// TIA Portal V17 export
// export: Created 2025-03-07T09:17:31.2731089Z, ExportSetting WithDefaults, DisplayName Totally Integrated Automation Portal, DisplayVersion V17 Update 8, DisplayName TIA Portal Openness, DisplayVersion V17 Update 8, DisplayName TIA Portal Version Control Interface, DisplayVersion V17, DisplayName SINAMICS Startdrive Advanced, DisplayVersion V17 SP2, DisplayName SINAMICS Startdrive G110M, G120, G120C, G120D, G120P, G115D, DisplayVersion V17 SP2, DisplayName SINAMICS Startdrive G130, G150, S120, S150, SINAMICS MV, S210, DisplayVersion V17 SP2, DisplayName STEP 7 Professional, DisplayVersion V17 Update 8, DisplayName SINUMERIK ONE STEP 7 Toolbox, DisplayVersion V17 Update 12, DisplayName SINUMERIK 840D sl STEP 7 Toolbox, DisplayVersion V17 Update 12, DisplayName STEP 7 Safety, DisplayVersion V17 Update 6, DisplayName WinCC Advanced, DisplayVersion V17 Update 8
FUNCTION "FC373_NCK_M_CH9_SPARE" : Void   // FC373, LAD
TITLE = Channel 1 data
{ S7_Optimized_Access := 'FALSE' }
AUTHOR : ETXETAR
VERSION : 1.0
// stored: AutoNumber false, IsIECCheckEnabled false, SetENOAutomatically false, UDAEnableTagReadback false
BEGIN

REGION Network 1: ACKNOWLEDGE M700-FIXTURE 4 CLAMP SEQUENCE (READ-IN DISABLE) / ACKNOWLEDGE M100-CLAMP SEQUENCE FIXTURE 1
   // NOTE: WHEN THERE IS NOT INDEXING TABLE AVAILABLE IN THE MACHINE DELETE 
   // DB2171.DBX5.0 AND DB2171.DBX2.0
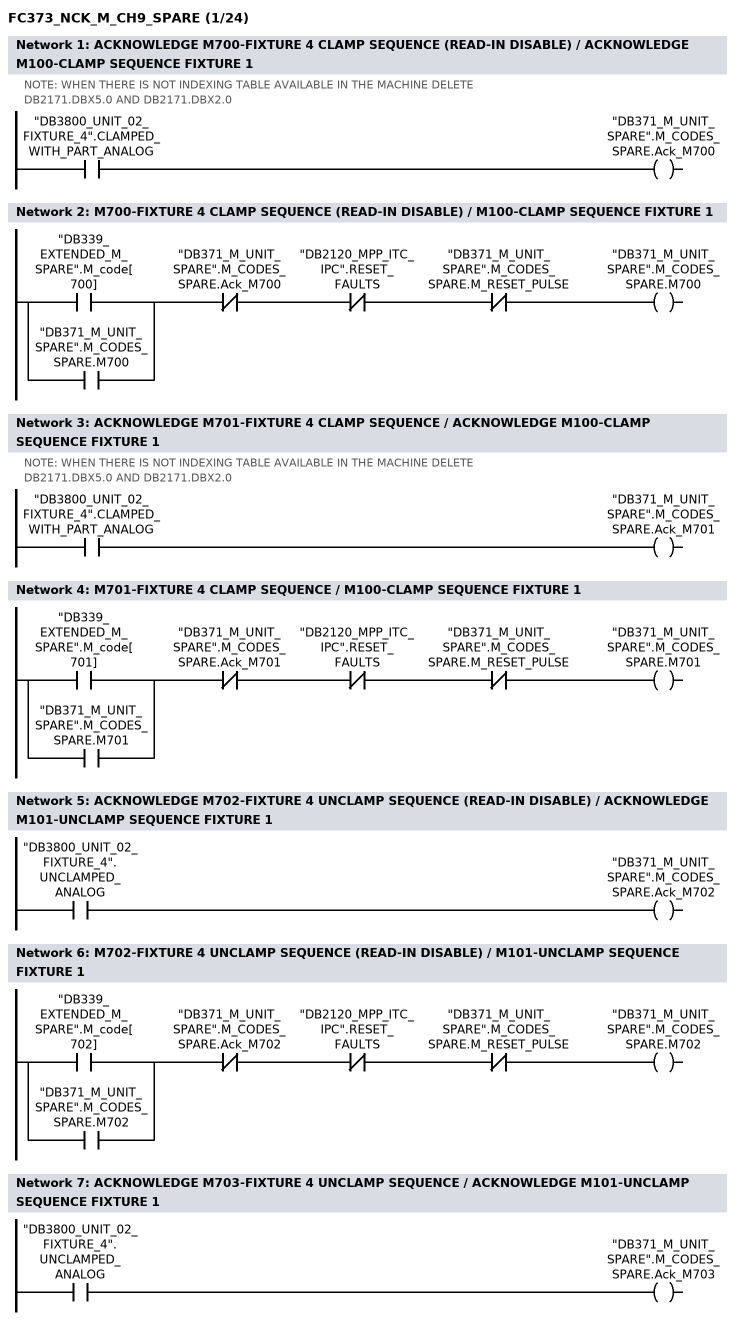
   RUNG wire#powerrail
      Contact( "DB3800_UNIT_02_FIXTURE_4".CLAMPED_WITH_PART_ANALOG )
      Coil( "DB371_M_UNIT_SPARE".M_CODES_SPARE.Ack_M700 )
   END_RUNG
   // the same network as SCL:
   "DB371_M_UNIT_SPARE".M_CODES_SPARE.Ack_M700 := "DB3800_UNIT_02_FIXTURE_4".CLAMPED_WITH_PART_ANALOG;
END_REGION

REGION Network 2: M700-FIXTURE 4 CLAMP SEQUENCE (READ-IN DISABLE) / M100-CLAMP SEQUENCE FIXTURE 1
   RUNG wire#powerrail
      Contact( "DB339_EXTENDED_M_SPARE".M_code[700] )
      wire#w1
      I_Contact( "DB371_M_UNIT_SPARE".M_CODES_SPARE.Ack_M700 )
      I_Contact( "DB2120_MPP_ITC_IPC".RESET_FAULTS )
      I_Contact( "DB371_M_UNIT_SPARE".M_CODES_SPARE.M_RESET_PULSE )
      Coil( "DB371_M_UNIT_SPARE".M_CODES_SPARE.M700 )
   END_RUNG
   RUNG wire#powerrail
      Contact( "DB371_M_UNIT_SPARE".M_CODES_SPARE.M700 )
   END_RUNG wire#w1
   // the same network as SCL:
   "DB371_M_UNIT_SPARE".M_CODES_SPARE.M700 := ("DB339_EXTENDED_M_SPARE".M_code[700] OR "DB371_M_UNIT_SPARE".M_CODES_SPARE.M700) AND NOT "DB371_M_UNIT_SPARE".M_CODES_SPARE.Ack_M700 AND NOT "DB2120_MPP_ITC_IPC".RESET_FAULTS AND NOT "DB371_M_UNIT_SPARE".M_CODES_SPARE.M_RESET_PULSE;
END_REGION

REGION Network 3: ACKNOWLEDGE M701-FIXTURE 4 CLAMP SEQUENCE / ACKNOWLEDGE M100-CLAMP SEQUENCE FIXTURE 1
   // NOTE: WHEN THERE IS NOT INDEXING TABLE AVAILABLE IN THE MACHINE DELETE 
   // DB2171.DBX5.0 AND DB2171.DBX2.0
   RUNG wire#powerrail
      Contact( "DB3800_UNIT_02_FIXTURE_4".CLAMPED_WITH_PART_ANALOG )
      Coil( "DB371_M_UNIT_SPARE".M_CODES_SPARE.Ack_M701 )
   END_RUNG
   // the same network as SCL:
   "DB371_M_UNIT_SPARE".M_CODES_SPARE.Ack_M701 := "DB3800_UNIT_02_FIXTURE_4".CLAMPED_WITH_PART_ANALOG;
END_REGION

REGION Network 4: M701-FIXTURE 4 CLAMP SEQUENCE / M100-CLAMP SEQUENCE FIXTURE 1
   RUNG wire#powerrail
      Contact( "DB339_EXTENDED_M_SPARE".M_code[701] )
      wire#w1
      I_Contact( "DB371_M_UNIT_SPARE".M_CODES_SPARE.Ack_M701 )
      I_Contact( "DB2120_MPP_ITC_IPC".RESET_FAULTS )
      I_Contact( "DB371_M_UNIT_SPARE".M_CODES_SPARE.M_RESET_PULSE )
      Coil( "DB371_M_UNIT_SPARE".M_CODES_SPARE.M701 )
   END_RUNG
   RUNG wire#powerrail
      Contact( "DB371_M_UNIT_SPARE".M_CODES_SPARE.M701 )
   END_RUNG wire#w1
   // the same network as SCL:
   "DB371_M_UNIT_SPARE".M_CODES_SPARE.M701 := ("DB339_EXTENDED_M_SPARE".M_code[701] OR "DB371_M_UNIT_SPARE".M_CODES_SPARE.M701) AND NOT "DB371_M_UNIT_SPARE".M_CODES_SPARE.Ack_M701 AND NOT "DB2120_MPP_ITC_IPC".RESET_FAULTS AND NOT "DB371_M_UNIT_SPARE".M_CODES_SPARE.M_RESET_PULSE;
END_REGION

REGION Network 5: ACKNOWLEDGE M702-FIXTURE 4 UNCLAMP SEQUENCE (READ-IN DISABLE) / ACKNOWLEDGE M101-UNCLAMP SEQUENCE FIXTURE 1
   RUNG wire#powerrail
      Contact( "DB3800_UNIT_02_FIXTURE_4".UNCLAMPED_ANALOG )
      Coil( "DB371_M_UNIT_SPARE".M_CODES_SPARE.Ack_M702 )
   END_RUNG
   // the same network as SCL:
   "DB371_M_UNIT_SPARE".M_CODES_SPARE.Ack_M702 := "DB3800_UNIT_02_FIXTURE_4".UNCLAMPED_ANALOG;
END_REGION

REGION Network 6: M702-FIXTURE 4 UNCLAMP SEQUENCE (READ-IN DISABLE) / M101-UNCLAMP SEQUENCE FIXTURE 1
   RUNG wire#powerrail
      Contact( "DB339_EXTENDED_M_SPARE".M_code[702] )
      wire#w1
      I_Contact( "DB371_M_UNIT_SPARE".M_CODES_SPARE.Ack_M702 )
      I_Contact( "DB2120_MPP_ITC_IPC".RESET_FAULTS )
      I_Contact( "DB371_M_UNIT_SPARE".M_CODES_SPARE.M_RESET_PULSE )
      Coil( "DB371_M_UNIT_SPARE".M_CODES_SPARE.M702 )
   END_RUNG
   RUNG wire#powerrail
      Contact( "DB371_M_UNIT_SPARE".M_CODES_SPARE.M702 )
   END_RUNG wire#w1
   // the same network as SCL:
   "DB371_M_UNIT_SPARE".M_CODES_SPARE.M702 := ("DB339_EXTENDED_M_SPARE".M_code[702] OR "DB371_M_UNIT_SPARE".M_CODES_SPARE.M702) AND NOT "DB371_M_UNIT_SPARE".M_CODES_SPARE.Ack_M702 AND NOT "DB2120_MPP_ITC_IPC".RESET_FAULTS AND NOT "DB371_M_UNIT_SPARE".M_CODES_SPARE.M_RESET_PULSE;
END_REGION

REGION Network 7: ACKNOWLEDGE M703-FIXTURE 4 UNCLAMP SEQUENCE / ACKNOWLEDGE M101-UNCLAMP SEQUENCE FIXTURE 1
   RUNG wire#powerrail
      Contact( "DB3800_UNIT_02_FIXTURE_4".UNCLAMPED_ANALOG )
      Coil( "DB371_M_UNIT_SPARE".M_CODES_SPARE.Ack_M703 )
   END_RUNG
   // the same network as SCL:
   "DB371_M_UNIT_SPARE".M_CODES_SPARE.Ack_M703 := "DB3800_UNIT_02_FIXTURE_4".UNCLAMPED_ANALOG;
END_REGION

REGION Network 8: M703-FIXTURE 4 UNCLAMP SEQUENCE / M101-UNCLAMP SEQUENCE FIXTURE 1
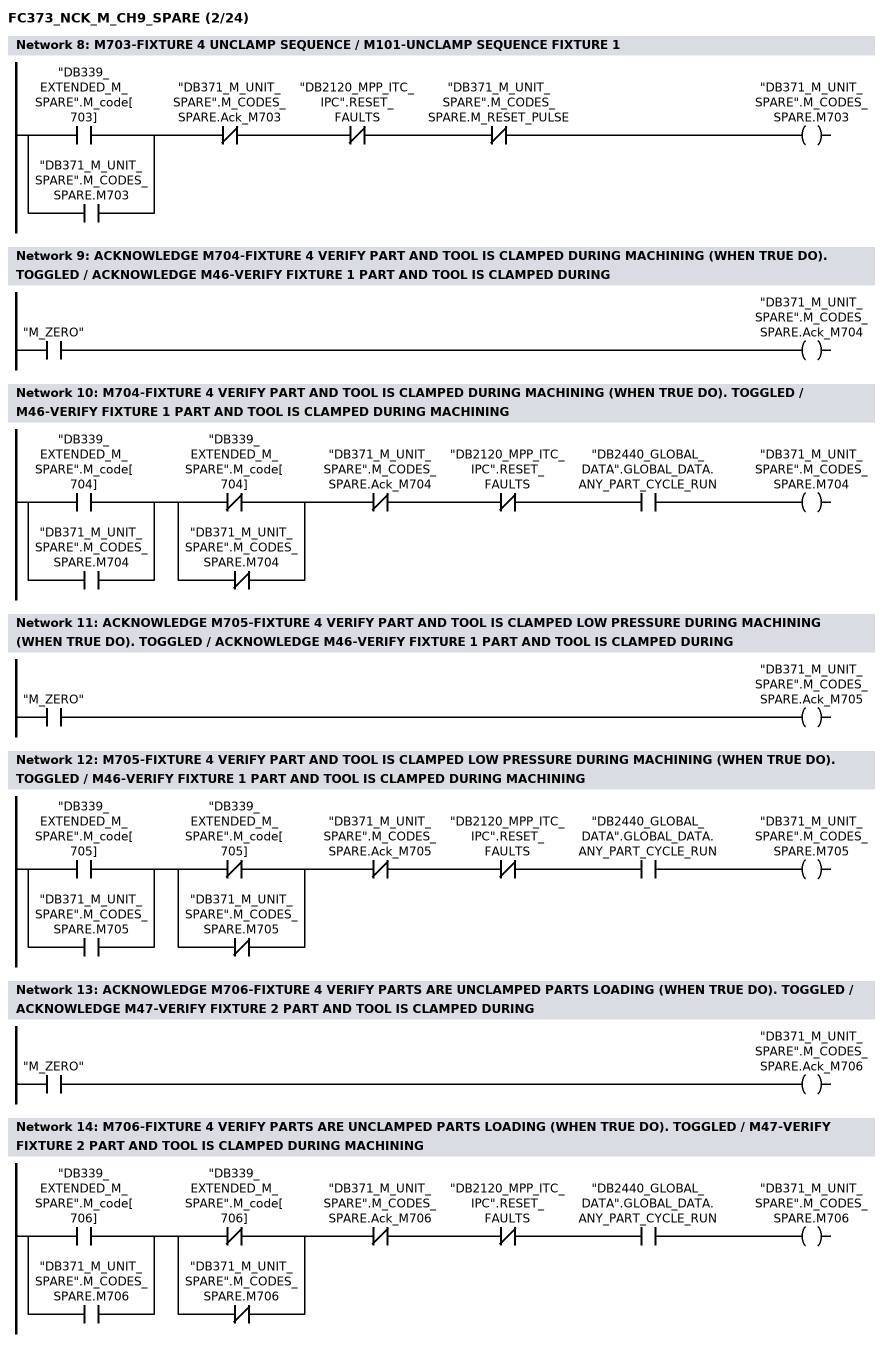
   RUNG wire#powerrail
      Contact( "DB339_EXTENDED_M_SPARE".M_code[703] )
      wire#w1
      I_Contact( "DB371_M_UNIT_SPARE".M_CODES_SPARE.Ack_M703 )
      I_Contact( "DB2120_MPP_ITC_IPC".RESET_FAULTS )
      I_Contact( "DB371_M_UNIT_SPARE".M_CODES_SPARE.M_RESET_PULSE )
      Coil( "DB371_M_UNIT_SPARE".M_CODES_SPARE.M703 )
   END_RUNG
   RUNG wire#powerrail
      Contact( "DB371_M_UNIT_SPARE".M_CODES_SPARE.M703 )
   END_RUNG wire#w1
   // the same network as SCL:
   "DB371_M_UNIT_SPARE".M_CODES_SPARE.M703 := ("DB339_EXTENDED_M_SPARE".M_code[703] OR "DB371_M_UNIT_SPARE".M_CODES_SPARE.M703) AND NOT "DB371_M_UNIT_SPARE".M_CODES_SPARE.Ack_M703 AND NOT "DB2120_MPP_ITC_IPC".RESET_FAULTS AND NOT "DB371_M_UNIT_SPARE".M_CODES_SPARE.M_RESET_PULSE;
END_REGION

REGION Network 9: ACKNOWLEDGE M704-FIXTURE 4 VERIFY PART AND TOOL IS CLAMPED DURING MACHINING (WHEN TRUE DO). TOGGLED / ACKNOWLEDGE M46-VERIFY FIXTURE 1 PART AND TOOL IS CLAMPED DURING
   RUNG wire#powerrail
      Contact( "M_ZERO" )
      Coil( "DB371_M_UNIT_SPARE".M_CODES_SPARE.Ack_M704 )
   END_RUNG
   // the same network as SCL:
   "DB371_M_UNIT_SPARE".M_CODES_SPARE.Ack_M704 := "M_ZERO";
END_REGION

REGION Network 10: M704-FIXTURE 4 VERIFY PART AND TOOL IS CLAMPED DURING MACHINING (WHEN TRUE DO). TOGGLED / M46-VERIFY FIXTURE 1 PART AND TOOL IS CLAMPED DURING MACHINING
   RUNG wire#powerrail
      Contact( "DB339_EXTENDED_M_SPARE".M_code[704] )
      wire#w1
      I_Contact( "DB339_EXTENDED_M_SPARE".M_code[704] )
      wire#w2
      I_Contact( "DB371_M_UNIT_SPARE".M_CODES_SPARE.Ack_M704 )
      I_Contact( "DB2120_MPP_ITC_IPC".RESET_FAULTS )
      Contact( "DB2440_GLOBAL_DATA".GLOBAL_DATA.ANY_PART_CYCLE_RUN )
      Coil( "DB371_M_UNIT_SPARE".M_CODES_SPARE.M704 )
   END_RUNG
   RUNG wire#powerrail
      Contact( "DB371_M_UNIT_SPARE".M_CODES_SPARE.M704 )
   END_RUNG wire#w1
   RUNG wire#w1
      I_Contact( "DB371_M_UNIT_SPARE".M_CODES_SPARE.M704 )
   END_RUNG wire#w2
   // the same network as SCL:
   "DB371_M_UNIT_SPARE".M_CODES_SPARE.M704 := ("DB339_EXTENDED_M_SPARE".M_code[704] OR "DB371_M_UNIT_SPARE".M_CODES_SPARE.M704) AND (NOT "DB339_EXTENDED_M_SPARE".M_code[704] OR NOT "DB371_M_UNIT_SPARE".M_CODES_SPARE.M704) AND NOT "DB371_M_UNIT_SPARE".M_CODES_SPARE.Ack_M704 AND NOT "DB2120_MPP_ITC_IPC".RESET_FAULTS AND "DB2440_GLOBAL_DATA".GLOBAL_DATA.ANY_PART_CYCLE_RUN;
END_REGION

REGION Network 11: ACKNOWLEDGE M705-FIXTURE 4 VERIFY PART AND TOOL IS CLAMPED LOW PRESSURE DURING MACHINING (WHEN TRUE DO). TOGGLED / ACKNOWLEDGE M46-VERIFY FIXTURE 1 PART AND TOOL IS CLAMPED DURING
   RUNG wire#powerrail
      Contact( "M_ZERO" )
      Coil( "DB371_M_UNIT_SPARE".M_CODES_SPARE.Ack_M705 )
   END_RUNG
   // the same network as SCL:
   "DB371_M_UNIT_SPARE".M_CODES_SPARE.Ack_M705 := "M_ZERO";
END_REGION

REGION Network 12: M705-FIXTURE 4 VERIFY PART AND TOOL IS CLAMPED LOW PRESSURE DURING MACHINING (WHEN TRUE DO). TOGGLED / M46-VERIFY FIXTURE 1 PART AND TOOL IS CLAMPED DURING MACHINING
   RUNG wire#powerrail
      Contact( "DB339_EXTENDED_M_SPARE".M_code[705] )
      wire#w1
      I_Contact( "DB339_EXTENDED_M_SPARE".M_code[705] )
      wire#w2
      I_Contact( "DB371_M_UNIT_SPARE".M_CODES_SPARE.Ack_M705 )
      I_Contact( "DB2120_MPP_ITC_IPC".RESET_FAULTS )
      Contact( "DB2440_GLOBAL_DATA".GLOBAL_DATA.ANY_PART_CYCLE_RUN )
      Coil( "DB371_M_UNIT_SPARE".M_CODES_SPARE.M705 )
   END_RUNG
   RUNG wire#powerrail
      Contact( "DB371_M_UNIT_SPARE".M_CODES_SPARE.M705 )
   END_RUNG wire#w1
   RUNG wire#w1
      I_Contact( "DB371_M_UNIT_SPARE".M_CODES_SPARE.M705 )
   END_RUNG wire#w2
   // the same network as SCL:
   "DB371_M_UNIT_SPARE".M_CODES_SPARE.M705 := ("DB339_EXTENDED_M_SPARE".M_code[705] OR "DB371_M_UNIT_SPARE".M_CODES_SPARE.M705) AND (NOT "DB339_EXTENDED_M_SPARE".M_code[705] OR NOT "DB371_M_UNIT_SPARE".M_CODES_SPARE.M705) AND NOT "DB371_M_UNIT_SPARE".M_CODES_SPARE.Ack_M705 AND NOT "DB2120_MPP_ITC_IPC".RESET_FAULTS AND "DB2440_GLOBAL_DATA".GLOBAL_DATA.ANY_PART_CYCLE_RUN;
END_REGION

REGION Network 13: ACKNOWLEDGE M706-FIXTURE 4 VERIFY PARTS ARE UNCLAMPED PARTS LOADING (WHEN TRUE DO). TOGGLED / ACKNOWLEDGE M47-VERIFY FIXTURE 2 PART AND TOOL IS CLAMPED DURING
   RUNG wire#powerrail
      Contact( "M_ZERO" )
      Coil( "DB371_M_UNIT_SPARE".M_CODES_SPARE.Ack_M706 )
   END_RUNG
   // the same network as SCL:
   "DB371_M_UNIT_SPARE".M_CODES_SPARE.Ack_M706 := "M_ZERO";
END_REGION

REGION Network 14: M706-FIXTURE 4 VERIFY PARTS ARE UNCLAMPED PARTS LOADING (WHEN TRUE DO). TOGGLED / M47-VERIFY FIXTURE 2 PART AND TOOL IS CLAMPED DURING MACHINING
   RUNG wire#powerrail
      Contact( "DB339_EXTENDED_M_SPARE".M_code[706] )
      wire#w1
      I_Contact( "DB339_EXTENDED_M_SPARE".M_code[706] )
      wire#w2
      I_Contact( "DB371_M_UNIT_SPARE".M_CODES_SPARE.Ack_M706 )
      I_Contact( "DB2120_MPP_ITC_IPC".RESET_FAULTS )
      Contact( "DB2440_GLOBAL_DATA".GLOBAL_DATA.ANY_PART_CYCLE_RUN )
      Coil( "DB371_M_UNIT_SPARE".M_CODES_SPARE.M706 )
   END_RUNG
   RUNG wire#powerrail
      Contact( "DB371_M_UNIT_SPARE".M_CODES_SPARE.M706 )
   END_RUNG wire#w1
   RUNG wire#w1
      I_Contact( "DB371_M_UNIT_SPARE".M_CODES_SPARE.M706 )
   END_RUNG wire#w2
   // the same network as SCL:
   "DB371_M_UNIT_SPARE".M_CODES_SPARE.M706 := ("DB339_EXTENDED_M_SPARE".M_code[706] OR "DB371_M_UNIT_SPARE".M_CODES_SPARE.M706) AND (NOT "DB339_EXTENDED_M_SPARE".M_code[706] OR NOT "DB371_M_UNIT_SPARE".M_CODES_SPARE.M706) AND NOT "DB371_M_UNIT_SPARE".M_CODES_SPARE.Ack_M706 AND NOT "DB2120_MPP_ITC_IPC".RESET_FAULTS AND "DB2440_GLOBAL_DATA".GLOBAL_DATA.ANY_PART_CYCLE_RUN;
END_REGION

REGION Network 15: ACKNOWLEDGE M707-FIXTURE 4 VERIFY FIXTURE REMAINS CLAMPED
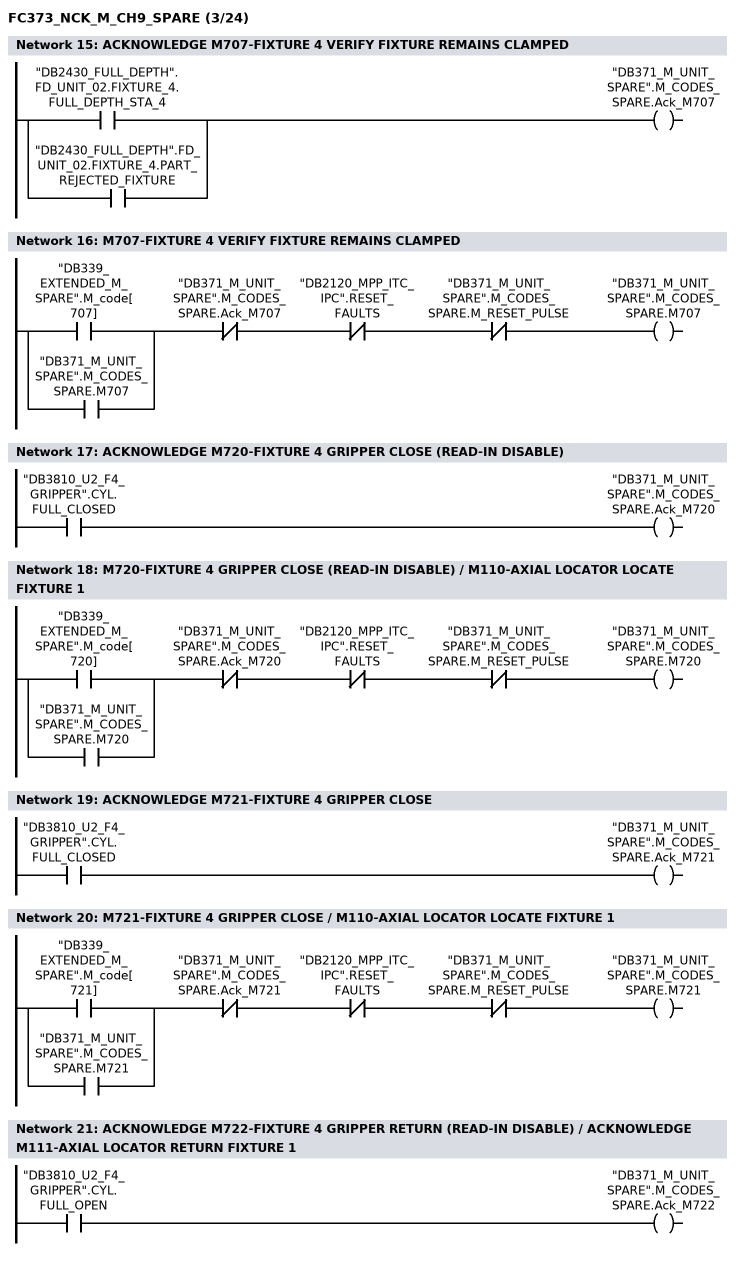
   RUNG wire#powerrail
      Contact( "DB2430_FULL_DEPTH".FD_UNIT_02.FIXTURE_4.FULL_DEPTH_STA_4 )
      wire#w1
      Coil( "DB371_M_UNIT_SPARE".M_CODES_SPARE.Ack_M707 )
   END_RUNG
   RUNG wire#powerrail
      Contact( "DB2430_FULL_DEPTH".FD_UNIT_02.FIXTURE_4.PART_REJECTED_FIXTURE )
   END_RUNG wire#w1
   // the same network as SCL:
   "DB371_M_UNIT_SPARE".M_CODES_SPARE.Ack_M707 := "DB2430_FULL_DEPTH".FD_UNIT_02.FIXTURE_4.FULL_DEPTH_STA_4 OR "DB2430_FULL_DEPTH".FD_UNIT_02.FIXTURE_4.PART_REJECTED_FIXTURE;
END_REGION

REGION Network 16: M707-FIXTURE 4 VERIFY FIXTURE REMAINS CLAMPED
   RUNG wire#powerrail
      Contact( "DB339_EXTENDED_M_SPARE".M_code[707] )
      wire#w1
      I_Contact( "DB371_M_UNIT_SPARE".M_CODES_SPARE.Ack_M707 )
      I_Contact( "DB2120_MPP_ITC_IPC".RESET_FAULTS )
      I_Contact( "DB371_M_UNIT_SPARE".M_CODES_SPARE.M_RESET_PULSE )
      Coil( "DB371_M_UNIT_SPARE".M_CODES_SPARE.M707 )
   END_RUNG
   RUNG wire#powerrail
      Contact( "DB371_M_UNIT_SPARE".M_CODES_SPARE.M707 )
   END_RUNG wire#w1
   // the same network as SCL:
   "DB371_M_UNIT_SPARE".M_CODES_SPARE.M707 := ("DB339_EXTENDED_M_SPARE".M_code[707] OR "DB371_M_UNIT_SPARE".M_CODES_SPARE.M707) AND NOT "DB371_M_UNIT_SPARE".M_CODES_SPARE.Ack_M707 AND NOT "DB2120_MPP_ITC_IPC".RESET_FAULTS AND NOT "DB371_M_UNIT_SPARE".M_CODES_SPARE.M_RESET_PULSE;
END_REGION

REGION Network 17: ACKNOWLEDGE M720-FIXTURE 4 GRIPPER CLOSE (READ-IN DISABLE)
   RUNG wire#powerrail
      Contact( "DB3810_U2_F4_GRIPPER".CYL.FULL_CLOSED )
      Coil( "DB371_M_UNIT_SPARE".M_CODES_SPARE.Ack_M720 )
   END_RUNG
   // the same network as SCL:
   "DB371_M_UNIT_SPARE".M_CODES_SPARE.Ack_M720 := "DB3810_U2_F4_GRIPPER".CYL.FULL_CLOSED;
END_REGION

REGION Network 18: M720-FIXTURE 4 GRIPPER CLOSE (READ-IN DISABLE) / M110-AXIAL LOCATOR LOCATE FIXTURE 1
   RUNG wire#powerrail
      Contact( "DB339_EXTENDED_M_SPARE".M_code[720] )
      wire#w1
      I_Contact( "DB371_M_UNIT_SPARE".M_CODES_SPARE.Ack_M720 )
      I_Contact( "DB2120_MPP_ITC_IPC".RESET_FAULTS )
      I_Contact( "DB371_M_UNIT_SPARE".M_CODES_SPARE.M_RESET_PULSE )
      Coil( "DB371_M_UNIT_SPARE".M_CODES_SPARE.M720 )
   END_RUNG
   RUNG wire#powerrail
      Contact( "DB371_M_UNIT_SPARE".M_CODES_SPARE.M720 )
   END_RUNG wire#w1
   // the same network as SCL:
   "DB371_M_UNIT_SPARE".M_CODES_SPARE.M720 := ("DB339_EXTENDED_M_SPARE".M_code[720] OR "DB371_M_UNIT_SPARE".M_CODES_SPARE.M720) AND NOT "DB371_M_UNIT_SPARE".M_CODES_SPARE.Ack_M720 AND NOT "DB2120_MPP_ITC_IPC".RESET_FAULTS AND NOT "DB371_M_UNIT_SPARE".M_CODES_SPARE.M_RESET_PULSE;
END_REGION

REGION Network 19: ACKNOWLEDGE M721-FIXTURE 4 GRIPPER CLOSE
   RUNG wire#powerrail
      Contact( "DB3810_U2_F4_GRIPPER".CYL.FULL_CLOSED )
      Coil( "DB371_M_UNIT_SPARE".M_CODES_SPARE.Ack_M721 )
   END_RUNG
   // the same network as SCL:
   "DB371_M_UNIT_SPARE".M_CODES_SPARE.Ack_M721 := "DB3810_U2_F4_GRIPPER".CYL.FULL_CLOSED;
END_REGION

REGION Network 20: M721-FIXTURE 4 GRIPPER CLOSE / M110-AXIAL LOCATOR LOCATE FIXTURE 1
   RUNG wire#powerrail
      Contact( "DB339_EXTENDED_M_SPARE".M_code[721] )
      wire#w1
      I_Contact( "DB371_M_UNIT_SPARE".M_CODES_SPARE.Ack_M721 )
      I_Contact( "DB2120_MPP_ITC_IPC".RESET_FAULTS )
      I_Contact( "DB371_M_UNIT_SPARE".M_CODES_SPARE.M_RESET_PULSE )
      Coil( "DB371_M_UNIT_SPARE".M_CODES_SPARE.M721 )
   END_RUNG
   RUNG wire#powerrail
      Contact( "DB371_M_UNIT_SPARE".M_CODES_SPARE.M721 )
   END_RUNG wire#w1
   // the same network as SCL:
   "DB371_M_UNIT_SPARE".M_CODES_SPARE.M721 := ("DB339_EXTENDED_M_SPARE".M_code[721] OR "DB371_M_UNIT_SPARE".M_CODES_SPARE.M721) AND NOT "DB371_M_UNIT_SPARE".M_CODES_SPARE.Ack_M721 AND NOT "DB2120_MPP_ITC_IPC".RESET_FAULTS AND NOT "DB371_M_UNIT_SPARE".M_CODES_SPARE.M_RESET_PULSE;
END_REGION

REGION Network 21: ACKNOWLEDGE M722-FIXTURE 4 GRIPPER RETURN (READ-IN DISABLE) / ACKNOWLEDGE M111-AXIAL LOCATOR RETURN FIXTURE 1
   RUNG wire#powerrail
      Contact( "DB3810_U2_F4_GRIPPER".CYL.FULL_OPEN )
      Coil( "DB371_M_UNIT_SPARE".M_CODES_SPARE.Ack_M722 )
   END_RUNG
   // the same network as SCL:
   "DB371_M_UNIT_SPARE".M_CODES_SPARE.Ack_M722 := "DB3810_U2_F4_GRIPPER".CYL.FULL_OPEN;
END_REGION

REGION Network 22: M722-FIXTURE 4 GRIPPER RETURN (READ-IN DISABLE) / M111-AXIAL LOCATOR RETURN FIXTURE 1
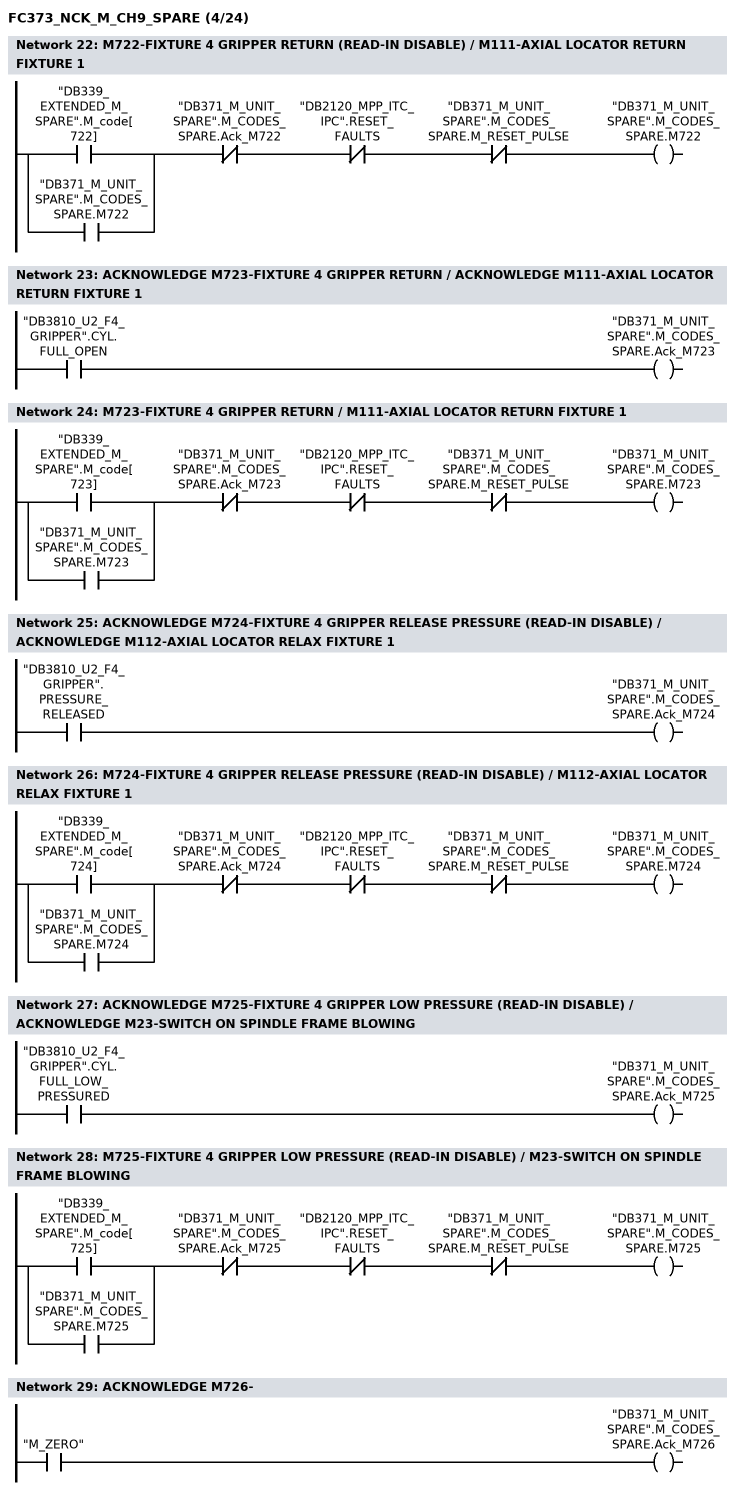
   RUNG wire#powerrail
      Contact( "DB339_EXTENDED_M_SPARE".M_code[722] )
      wire#w1
      I_Contact( "DB371_M_UNIT_SPARE".M_CODES_SPARE.Ack_M722 )
      I_Contact( "DB2120_MPP_ITC_IPC".RESET_FAULTS )
      I_Contact( "DB371_M_UNIT_SPARE".M_CODES_SPARE.M_RESET_PULSE )
      Coil( "DB371_M_UNIT_SPARE".M_CODES_SPARE.M722 )
   END_RUNG
   RUNG wire#powerrail
      Contact( "DB371_M_UNIT_SPARE".M_CODES_SPARE.M722 )
   END_RUNG wire#w1
   // the same network as SCL:
   "DB371_M_UNIT_SPARE".M_CODES_SPARE.M722 := ("DB339_EXTENDED_M_SPARE".M_code[722] OR "DB371_M_UNIT_SPARE".M_CODES_SPARE.M722) AND NOT "DB371_M_UNIT_SPARE".M_CODES_SPARE.Ack_M722 AND NOT "DB2120_MPP_ITC_IPC".RESET_FAULTS AND NOT "DB371_M_UNIT_SPARE".M_CODES_SPARE.M_RESET_PULSE;
END_REGION

REGION Network 23: ACKNOWLEDGE M723-FIXTURE 4 GRIPPER RETURN / ACKNOWLEDGE M111-AXIAL LOCATOR RETURN FIXTURE 1
   RUNG wire#powerrail
      Contact( "DB3810_U2_F4_GRIPPER".CYL.FULL_OPEN )
      Coil( "DB371_M_UNIT_SPARE".M_CODES_SPARE.Ack_M723 )
   END_RUNG
   // the same network as SCL:
   "DB371_M_UNIT_SPARE".M_CODES_SPARE.Ack_M723 := "DB3810_U2_F4_GRIPPER".CYL.FULL_OPEN;
END_REGION

REGION Network 24: M723-FIXTURE 4 GRIPPER RETURN / M111-AXIAL LOCATOR RETURN FIXTURE 1
   RUNG wire#powerrail
      Contact( "DB339_EXTENDED_M_SPARE".M_code[723] )
      wire#w1
      I_Contact( "DB371_M_UNIT_SPARE".M_CODES_SPARE.Ack_M723 )
      I_Contact( "DB2120_MPP_ITC_IPC".RESET_FAULTS )
      I_Contact( "DB371_M_UNIT_SPARE".M_CODES_SPARE.M_RESET_PULSE )
      Coil( "DB371_M_UNIT_SPARE".M_CODES_SPARE.M723 )
   END_RUNG
   RUNG wire#powerrail
      Contact( "DB371_M_UNIT_SPARE".M_CODES_SPARE.M723 )
   END_RUNG wire#w1
   // the same network as SCL:
   "DB371_M_UNIT_SPARE".M_CODES_SPARE.M723 := ("DB339_EXTENDED_M_SPARE".M_code[723] OR "DB371_M_UNIT_SPARE".M_CODES_SPARE.M723) AND NOT "DB371_M_UNIT_SPARE".M_CODES_SPARE.Ack_M723 AND NOT "DB2120_MPP_ITC_IPC".RESET_FAULTS AND NOT "DB371_M_UNIT_SPARE".M_CODES_SPARE.M_RESET_PULSE;
END_REGION

REGION Network 25: ACKNOWLEDGE M724-FIXTURE 4 GRIPPER RELEASE PRESSURE (READ-IN DISABLE) / ACKNOWLEDGE M112-AXIAL LOCATOR RELAX FIXTURE 1
   RUNG wire#powerrail
      Contact( "DB3810_U2_F4_GRIPPER".PRESSURE_RELEASED )
      Coil( "DB371_M_UNIT_SPARE".M_CODES_SPARE.Ack_M724 )
   END_RUNG
   // the same network as SCL:
   "DB371_M_UNIT_SPARE".M_CODES_SPARE.Ack_M724 := "DB3810_U2_F4_GRIPPER".PRESSURE_RELEASED;
END_REGION

REGION Network 26: M724-FIXTURE 4 GRIPPER RELEASE PRESSURE (READ-IN DISABLE) / M112-AXIAL LOCATOR RELAX FIXTURE 1
   RUNG wire#powerrail
      Contact( "DB339_EXTENDED_M_SPARE".M_code[724] )
      wire#w1
      I_Contact( "DB371_M_UNIT_SPARE".M_CODES_SPARE.Ack_M724 )
      I_Contact( "DB2120_MPP_ITC_IPC".RESET_FAULTS )
      I_Contact( "DB371_M_UNIT_SPARE".M_CODES_SPARE.M_RESET_PULSE )
      Coil( "DB371_M_UNIT_SPARE".M_CODES_SPARE.M724 )
   END_RUNG
   RUNG wire#powerrail
      Contact( "DB371_M_UNIT_SPARE".M_CODES_SPARE.M724 )
   END_RUNG wire#w1
   // the same network as SCL:
   "DB371_M_UNIT_SPARE".M_CODES_SPARE.M724 := ("DB339_EXTENDED_M_SPARE".M_code[724] OR "DB371_M_UNIT_SPARE".M_CODES_SPARE.M724) AND NOT "DB371_M_UNIT_SPARE".M_CODES_SPARE.Ack_M724 AND NOT "DB2120_MPP_ITC_IPC".RESET_FAULTS AND NOT "DB371_M_UNIT_SPARE".M_CODES_SPARE.M_RESET_PULSE;
END_REGION

REGION Network 27: ACKNOWLEDGE M725-FIXTURE 4 GRIPPER LOW PRESSURE (READ-IN DISABLE) / ACKNOWLEDGE M23-SWITCH ON SPINDLE FRAME BLOWING
   RUNG wire#powerrail
      Contact( "DB3810_U2_F4_GRIPPER".CYL.FULL_LOW_PRESSURED )
      Coil( "DB371_M_UNIT_SPARE".M_CODES_SPARE.Ack_M725 )
   END_RUNG
   // the same network as SCL:
   "DB371_M_UNIT_SPARE".M_CODES_SPARE.Ack_M725 := "DB3810_U2_F4_GRIPPER".CYL.FULL_LOW_PRESSURED;
END_REGION

REGION Network 28: M725-FIXTURE 4 GRIPPER LOW PRESSURE (READ-IN DISABLE) / M23-SWITCH ON SPINDLE FRAME BLOWING
   RUNG wire#powerrail
      Contact( "DB339_EXTENDED_M_SPARE".M_code[725] )
      wire#w1
      I_Contact( "DB371_M_UNIT_SPARE".M_CODES_SPARE.Ack_M725 )
      I_Contact( "DB2120_MPP_ITC_IPC".RESET_FAULTS )
      I_Contact( "DB371_M_UNIT_SPARE".M_CODES_SPARE.M_RESET_PULSE )
      Coil( "DB371_M_UNIT_SPARE".M_CODES_SPARE.M725 )
   END_RUNG
   RUNG wire#powerrail
      Contact( "DB371_M_UNIT_SPARE".M_CODES_SPARE.M725 )
   END_RUNG wire#w1
   // the same network as SCL:
   "DB371_M_UNIT_SPARE".M_CODES_SPARE.M725 := ("DB339_EXTENDED_M_SPARE".M_code[725] OR "DB371_M_UNIT_SPARE".M_CODES_SPARE.M725) AND NOT "DB371_M_UNIT_SPARE".M_CODES_SPARE.Ack_M725 AND NOT "DB2120_MPP_ITC_IPC".RESET_FAULTS AND NOT "DB371_M_UNIT_SPARE".M_CODES_SPARE.M_RESET_PULSE;
END_REGION

REGION Network 29: ACKNOWLEDGE M726-
   RUNG wire#powerrail
      Contact( "M_ZERO" )
      Coil( "DB371_M_UNIT_SPARE".M_CODES_SPARE.Ack_M726 )
   END_RUNG
   // the same network as SCL:
   "DB371_M_UNIT_SPARE".M_CODES_SPARE.Ack_M726 := "M_ZERO";
END_REGION

REGION Network 30: M726-
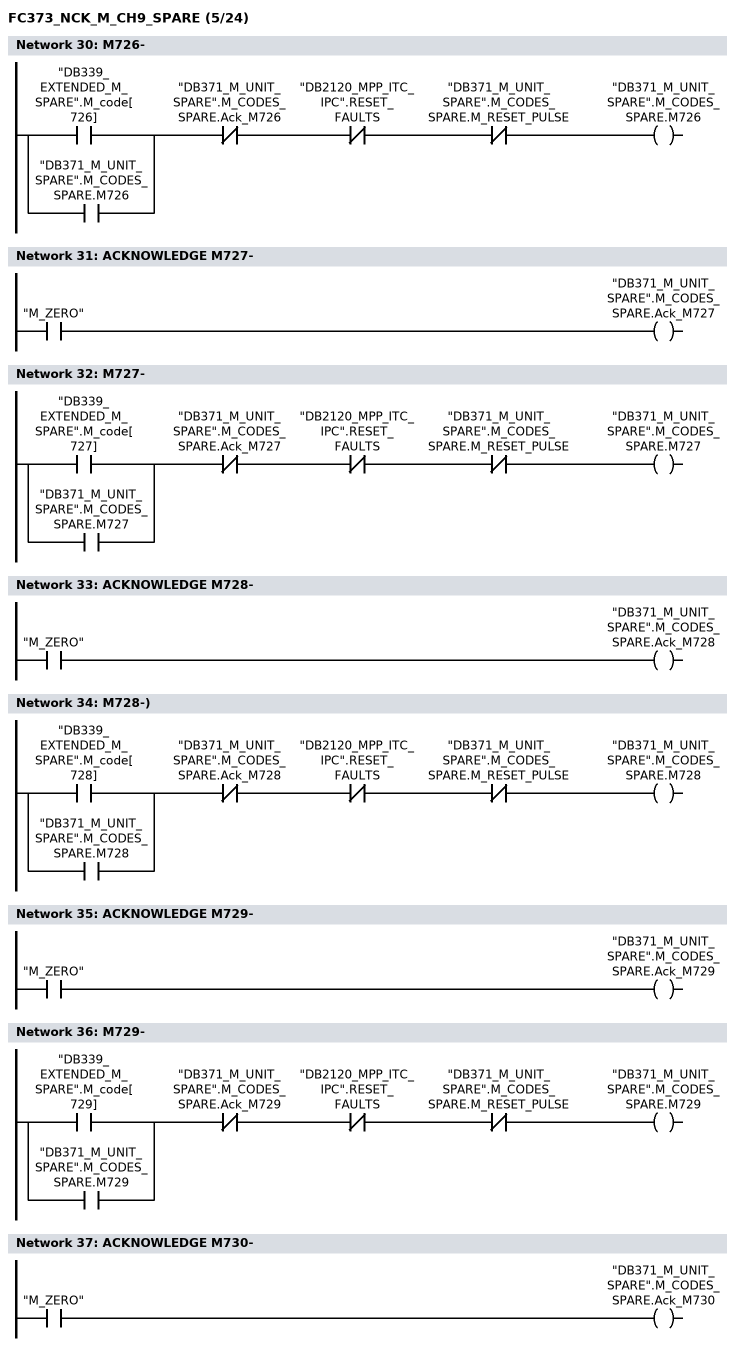
   RUNG wire#powerrail
      Contact( "DB339_EXTENDED_M_SPARE".M_code[726] )
      wire#w1
      I_Contact( "DB371_M_UNIT_SPARE".M_CODES_SPARE.Ack_M726 )
      I_Contact( "DB2120_MPP_ITC_IPC".RESET_FAULTS )
      I_Contact( "DB371_M_UNIT_SPARE".M_CODES_SPARE.M_RESET_PULSE )
      Coil( "DB371_M_UNIT_SPARE".M_CODES_SPARE.M726 )
   END_RUNG
   RUNG wire#powerrail
      Contact( "DB371_M_UNIT_SPARE".M_CODES_SPARE.M726 )
   END_RUNG wire#w1
   // the same network as SCL:
   "DB371_M_UNIT_SPARE".M_CODES_SPARE.M726 := ("DB339_EXTENDED_M_SPARE".M_code[726] OR "DB371_M_UNIT_SPARE".M_CODES_SPARE.M726) AND NOT "DB371_M_UNIT_SPARE".M_CODES_SPARE.Ack_M726 AND NOT "DB2120_MPP_ITC_IPC".RESET_FAULTS AND NOT "DB371_M_UNIT_SPARE".M_CODES_SPARE.M_RESET_PULSE;
END_REGION

REGION Network 31: ACKNOWLEDGE M727-
   RUNG wire#powerrail
      Contact( "M_ZERO" )
      Coil( "DB371_M_UNIT_SPARE".M_CODES_SPARE.Ack_M727 )
   END_RUNG
   // the same network as SCL:
   "DB371_M_UNIT_SPARE".M_CODES_SPARE.Ack_M727 := "M_ZERO";
END_REGION

REGION Network 32: M727-
   RUNG wire#powerrail
      Contact( "DB339_EXTENDED_M_SPARE".M_code[727] )
      wire#w1
      I_Contact( "DB371_M_UNIT_SPARE".M_CODES_SPARE.Ack_M727 )
      I_Contact( "DB2120_MPP_ITC_IPC".RESET_FAULTS )
      I_Contact( "DB371_M_UNIT_SPARE".M_CODES_SPARE.M_RESET_PULSE )
      Coil( "DB371_M_UNIT_SPARE".M_CODES_SPARE.M727 )
   END_RUNG
   RUNG wire#powerrail
      Contact( "DB371_M_UNIT_SPARE".M_CODES_SPARE.M727 )
   END_RUNG wire#w1
   // the same network as SCL:
   "DB371_M_UNIT_SPARE".M_CODES_SPARE.M727 := ("DB339_EXTENDED_M_SPARE".M_code[727] OR "DB371_M_UNIT_SPARE".M_CODES_SPARE.M727) AND NOT "DB371_M_UNIT_SPARE".M_CODES_SPARE.Ack_M727 AND NOT "DB2120_MPP_ITC_IPC".RESET_FAULTS AND NOT "DB371_M_UNIT_SPARE".M_CODES_SPARE.M_RESET_PULSE;
END_REGION

REGION Network 33: ACKNOWLEDGE M728-
   RUNG wire#powerrail
      Contact( "M_ZERO" )
      Coil( "DB371_M_UNIT_SPARE".M_CODES_SPARE.Ack_M728 )
   END_RUNG
   // the same network as SCL:
   "DB371_M_UNIT_SPARE".M_CODES_SPARE.Ack_M728 := "M_ZERO";
END_REGION

REGION Network 34: M728-)
   RUNG wire#powerrail
      Contact( "DB339_EXTENDED_M_SPARE".M_code[728] )
      wire#w1
      I_Contact( "DB371_M_UNIT_SPARE".M_CODES_SPARE.Ack_M728 )
      I_Contact( "DB2120_MPP_ITC_IPC".RESET_FAULTS )
      I_Contact( "DB371_M_UNIT_SPARE".M_CODES_SPARE.M_RESET_PULSE )
      Coil( "DB371_M_UNIT_SPARE".M_CODES_SPARE.M728 )
   END_RUNG
   RUNG wire#powerrail
      Contact( "DB371_M_UNIT_SPARE".M_CODES_SPARE.M728 )
   END_RUNG wire#w1
   // the same network as SCL:
   "DB371_M_UNIT_SPARE".M_CODES_SPARE.M728 := ("DB339_EXTENDED_M_SPARE".M_code[728] OR "DB371_M_UNIT_SPARE".M_CODES_SPARE.M728) AND NOT "DB371_M_UNIT_SPARE".M_CODES_SPARE.Ack_M728 AND NOT "DB2120_MPP_ITC_IPC".RESET_FAULTS AND NOT "DB371_M_UNIT_SPARE".M_CODES_SPARE.M_RESET_PULSE;
END_REGION

REGION Network 35: ACKNOWLEDGE M729-
   RUNG wire#powerrail
      Contact( "M_ZERO" )
      Coil( "DB371_M_UNIT_SPARE".M_CODES_SPARE.Ack_M729 )
   END_RUNG
   // the same network as SCL:
   "DB371_M_UNIT_SPARE".M_CODES_SPARE.Ack_M729 := "M_ZERO";
END_REGION

REGION Network 36: M729-
   RUNG wire#powerrail
      Contact( "DB339_EXTENDED_M_SPARE".M_code[729] )
      wire#w1
      I_Contact( "DB371_M_UNIT_SPARE".M_CODES_SPARE.Ack_M729 )
      I_Contact( "DB2120_MPP_ITC_IPC".RESET_FAULTS )
      I_Contact( "DB371_M_UNIT_SPARE".M_CODES_SPARE.M_RESET_PULSE )
      Coil( "DB371_M_UNIT_SPARE".M_CODES_SPARE.M729 )
   END_RUNG
   RUNG wire#powerrail
      Contact( "DB371_M_UNIT_SPARE".M_CODES_SPARE.M729 )
   END_RUNG wire#w1
   // the same network as SCL:
   "DB371_M_UNIT_SPARE".M_CODES_SPARE.M729 := ("DB339_EXTENDED_M_SPARE".M_code[729] OR "DB371_M_UNIT_SPARE".M_CODES_SPARE.M729) AND NOT "DB371_M_UNIT_SPARE".M_CODES_SPARE.Ack_M729 AND NOT "DB2120_MPP_ITC_IPC".RESET_FAULTS AND NOT "DB371_M_UNIT_SPARE".M_CODES_SPARE.M_RESET_PULSE;
END_REGION

REGION Network 37: ACKNOWLEDGE M730-
   RUNG wire#powerrail
      Contact( "M_ZERO" )
      Coil( "DB371_M_UNIT_SPARE".M_CODES_SPARE.Ack_M730 )
   END_RUNG
   // the same network as SCL:
   "DB371_M_UNIT_SPARE".M_CODES_SPARE.Ack_M730 := "M_ZERO";
END_REGION

REGION Network 38: M730-
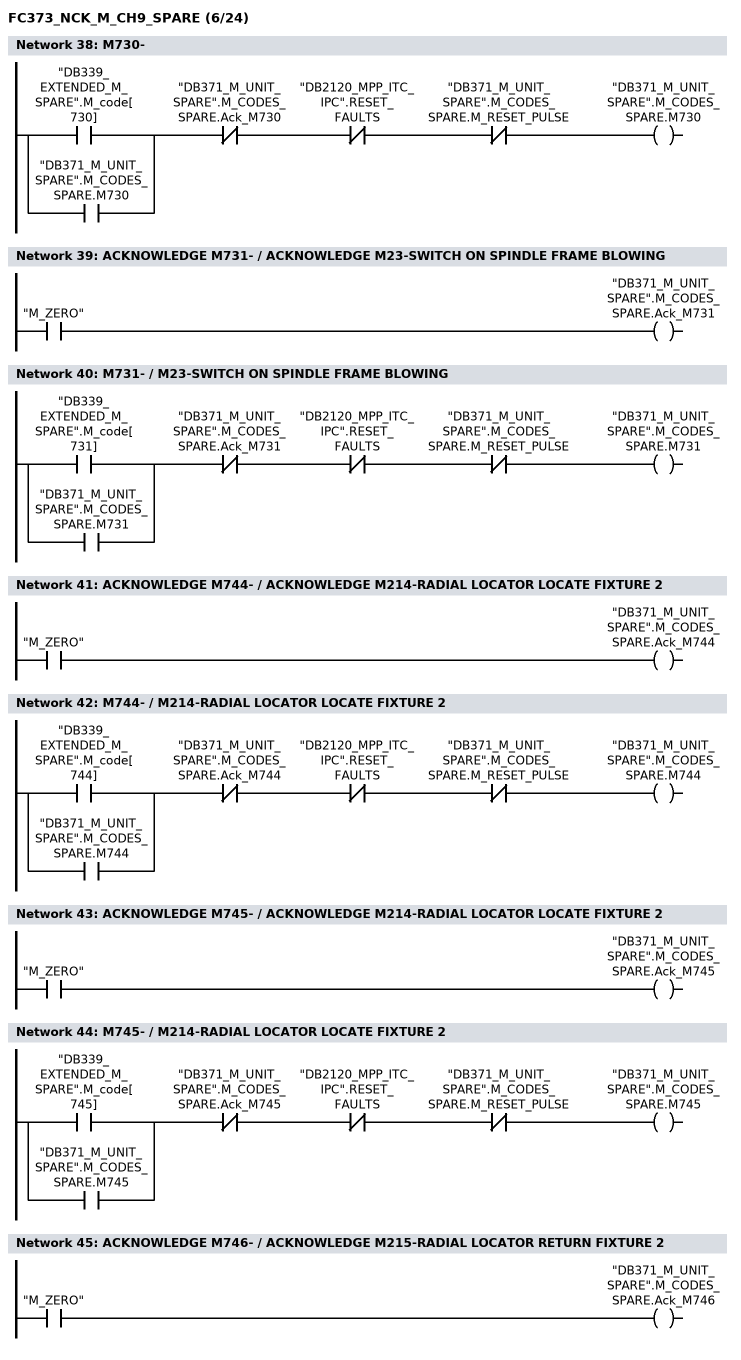
   RUNG wire#powerrail
      Contact( "DB339_EXTENDED_M_SPARE".M_code[730] )
      wire#w1
      I_Contact( "DB371_M_UNIT_SPARE".M_CODES_SPARE.Ack_M730 )
      I_Contact( "DB2120_MPP_ITC_IPC".RESET_FAULTS )
      I_Contact( "DB371_M_UNIT_SPARE".M_CODES_SPARE.M_RESET_PULSE )
      Coil( "DB371_M_UNIT_SPARE".M_CODES_SPARE.M730 )
   END_RUNG
   RUNG wire#powerrail
      Contact( "DB371_M_UNIT_SPARE".M_CODES_SPARE.M730 )
   END_RUNG wire#w1
   // the same network as SCL:
   "DB371_M_UNIT_SPARE".M_CODES_SPARE.M730 := ("DB339_EXTENDED_M_SPARE".M_code[730] OR "DB371_M_UNIT_SPARE".M_CODES_SPARE.M730) AND NOT "DB371_M_UNIT_SPARE".M_CODES_SPARE.Ack_M730 AND NOT "DB2120_MPP_ITC_IPC".RESET_FAULTS AND NOT "DB371_M_UNIT_SPARE".M_CODES_SPARE.M_RESET_PULSE;
END_REGION

REGION Network 39: ACKNOWLEDGE M731- / ACKNOWLEDGE M23-SWITCH ON SPINDLE FRAME BLOWING
   RUNG wire#powerrail
      Contact( "M_ZERO" )
      Coil( "DB371_M_UNIT_SPARE".M_CODES_SPARE.Ack_M731 )
   END_RUNG
   // the same network as SCL:
   "DB371_M_UNIT_SPARE".M_CODES_SPARE.Ack_M731 := "M_ZERO";
END_REGION

REGION Network 40: M731- / M23-SWITCH ON SPINDLE FRAME BLOWING
   RUNG wire#powerrail
      Contact( "DB339_EXTENDED_M_SPARE".M_code[731] )
      wire#w1
      I_Contact( "DB371_M_UNIT_SPARE".M_CODES_SPARE.Ack_M731 )
      I_Contact( "DB2120_MPP_ITC_IPC".RESET_FAULTS )
      I_Contact( "DB371_M_UNIT_SPARE".M_CODES_SPARE.M_RESET_PULSE )
      Coil( "DB371_M_UNIT_SPARE".M_CODES_SPARE.M731 )
   END_RUNG
   RUNG wire#powerrail
      Contact( "DB371_M_UNIT_SPARE".M_CODES_SPARE.M731 )
   END_RUNG wire#w1
   // the same network as SCL:
   "DB371_M_UNIT_SPARE".M_CODES_SPARE.M731 := ("DB339_EXTENDED_M_SPARE".M_code[731] OR "DB371_M_UNIT_SPARE".M_CODES_SPARE.M731) AND NOT "DB371_M_UNIT_SPARE".M_CODES_SPARE.Ack_M731 AND NOT "DB2120_MPP_ITC_IPC".RESET_FAULTS AND NOT "DB371_M_UNIT_SPARE".M_CODES_SPARE.M_RESET_PULSE;
END_REGION

REGION Network 41: ACKNOWLEDGE M744- / ACKNOWLEDGE M214-RADIAL LOCATOR LOCATE FIXTURE 2
   RUNG wire#powerrail
      Contact( "M_ZERO" )
      Coil( "DB371_M_UNIT_SPARE".M_CODES_SPARE.Ack_M744 )
   END_RUNG
   // the same network as SCL:
   "DB371_M_UNIT_SPARE".M_CODES_SPARE.Ack_M744 := "M_ZERO";
END_REGION

REGION Network 42: M744- / M214-RADIAL LOCATOR LOCATE FIXTURE 2
   RUNG wire#powerrail
      Contact( "DB339_EXTENDED_M_SPARE".M_code[744] )
      wire#w1
      I_Contact( "DB371_M_UNIT_SPARE".M_CODES_SPARE.Ack_M744 )
      I_Contact( "DB2120_MPP_ITC_IPC".RESET_FAULTS )
      I_Contact( "DB371_M_UNIT_SPARE".M_CODES_SPARE.M_RESET_PULSE )
      Coil( "DB371_M_UNIT_SPARE".M_CODES_SPARE.M744 )
   END_RUNG
   RUNG wire#powerrail
      Contact( "DB371_M_UNIT_SPARE".M_CODES_SPARE.M744 )
   END_RUNG wire#w1
   // the same network as SCL:
   "DB371_M_UNIT_SPARE".M_CODES_SPARE.M744 := ("DB339_EXTENDED_M_SPARE".M_code[744] OR "DB371_M_UNIT_SPARE".M_CODES_SPARE.M744) AND NOT "DB371_M_UNIT_SPARE".M_CODES_SPARE.Ack_M744 AND NOT "DB2120_MPP_ITC_IPC".RESET_FAULTS AND NOT "DB371_M_UNIT_SPARE".M_CODES_SPARE.M_RESET_PULSE;
END_REGION

REGION Network 43: ACKNOWLEDGE M745- / ACKNOWLEDGE M214-RADIAL LOCATOR LOCATE FIXTURE 2
   RUNG wire#powerrail
      Contact( "M_ZERO" )
      Coil( "DB371_M_UNIT_SPARE".M_CODES_SPARE.Ack_M745 )
   END_RUNG
   // the same network as SCL:
   "DB371_M_UNIT_SPARE".M_CODES_SPARE.Ack_M745 := "M_ZERO";
END_REGION

REGION Network 44: M745- / M214-RADIAL LOCATOR LOCATE FIXTURE 2
   RUNG wire#powerrail
      Contact( "DB339_EXTENDED_M_SPARE".M_code[745] )
      wire#w1
      I_Contact( "DB371_M_UNIT_SPARE".M_CODES_SPARE.Ack_M745 )
      I_Contact( "DB2120_MPP_ITC_IPC".RESET_FAULTS )
      I_Contact( "DB371_M_UNIT_SPARE".M_CODES_SPARE.M_RESET_PULSE )
      Coil( "DB371_M_UNIT_SPARE".M_CODES_SPARE.M745 )
   END_RUNG
   RUNG wire#powerrail
      Contact( "DB371_M_UNIT_SPARE".M_CODES_SPARE.M745 )
   END_RUNG wire#w1
   // the same network as SCL:
   "DB371_M_UNIT_SPARE".M_CODES_SPARE.M745 := ("DB339_EXTENDED_M_SPARE".M_code[745] OR "DB371_M_UNIT_SPARE".M_CODES_SPARE.M745) AND NOT "DB371_M_UNIT_SPARE".M_CODES_SPARE.Ack_M745 AND NOT "DB2120_MPP_ITC_IPC".RESET_FAULTS AND NOT "DB371_M_UNIT_SPARE".M_CODES_SPARE.M_RESET_PULSE;
END_REGION

REGION Network 45: ACKNOWLEDGE M746- / ACKNOWLEDGE M215-RADIAL LOCATOR RETURN FIXTURE 2
   RUNG wire#powerrail
      Contact( "M_ZERO" )
      Coil( "DB371_M_UNIT_SPARE".M_CODES_SPARE.Ack_M746 )
   END_RUNG
   // the same network as SCL:
   "DB371_M_UNIT_SPARE".M_CODES_SPARE.Ack_M746 := "M_ZERO";
END_REGION

REGION Network 46: M746- / M215-RADIAL LOCATOR RETURN FIXTURE 2
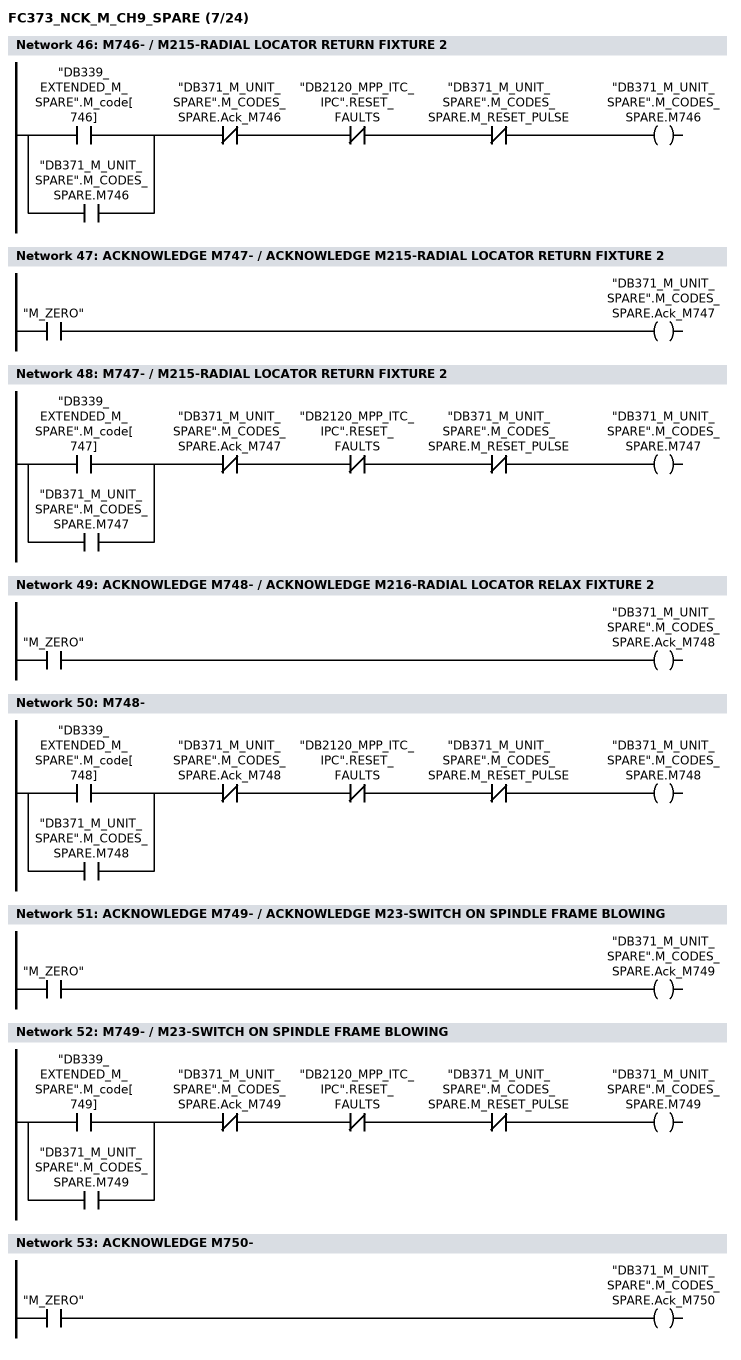
   RUNG wire#powerrail
      Contact( "DB339_EXTENDED_M_SPARE".M_code[746] )
      wire#w1
      I_Contact( "DB371_M_UNIT_SPARE".M_CODES_SPARE.Ack_M746 )
      I_Contact( "DB2120_MPP_ITC_IPC".RESET_FAULTS )
      I_Contact( "DB371_M_UNIT_SPARE".M_CODES_SPARE.M_RESET_PULSE )
      Coil( "DB371_M_UNIT_SPARE".M_CODES_SPARE.M746 )
   END_RUNG
   RUNG wire#powerrail
      Contact( "DB371_M_UNIT_SPARE".M_CODES_SPARE.M746 )
   END_RUNG wire#w1
   // the same network as SCL:
   "DB371_M_UNIT_SPARE".M_CODES_SPARE.M746 := ("DB339_EXTENDED_M_SPARE".M_code[746] OR "DB371_M_UNIT_SPARE".M_CODES_SPARE.M746) AND NOT "DB371_M_UNIT_SPARE".M_CODES_SPARE.Ack_M746 AND NOT "DB2120_MPP_ITC_IPC".RESET_FAULTS AND NOT "DB371_M_UNIT_SPARE".M_CODES_SPARE.M_RESET_PULSE;
END_REGION

REGION Network 47: ACKNOWLEDGE M747- / ACKNOWLEDGE M215-RADIAL LOCATOR RETURN FIXTURE 2
   RUNG wire#powerrail
      Contact( "M_ZERO" )
      Coil( "DB371_M_UNIT_SPARE".M_CODES_SPARE.Ack_M747 )
   END_RUNG
   // the same network as SCL:
   "DB371_M_UNIT_SPARE".M_CODES_SPARE.Ack_M747 := "M_ZERO";
END_REGION

REGION Network 48: M747- / M215-RADIAL LOCATOR RETURN FIXTURE 2
   RUNG wire#powerrail
      Contact( "DB339_EXTENDED_M_SPARE".M_code[747] )
      wire#w1
      I_Contact( "DB371_M_UNIT_SPARE".M_CODES_SPARE.Ack_M747 )
      I_Contact( "DB2120_MPP_ITC_IPC".RESET_FAULTS )
      I_Contact( "DB371_M_UNIT_SPARE".M_CODES_SPARE.M_RESET_PULSE )
      Coil( "DB371_M_UNIT_SPARE".M_CODES_SPARE.M747 )
   END_RUNG
   RUNG wire#powerrail
      Contact( "DB371_M_UNIT_SPARE".M_CODES_SPARE.M747 )
   END_RUNG wire#w1
   // the same network as SCL:
   "DB371_M_UNIT_SPARE".M_CODES_SPARE.M747 := ("DB339_EXTENDED_M_SPARE".M_code[747] OR "DB371_M_UNIT_SPARE".M_CODES_SPARE.M747) AND NOT "DB371_M_UNIT_SPARE".M_CODES_SPARE.Ack_M747 AND NOT "DB2120_MPP_ITC_IPC".RESET_FAULTS AND NOT "DB371_M_UNIT_SPARE".M_CODES_SPARE.M_RESET_PULSE;
END_REGION

REGION Network 49: ACKNOWLEDGE M748- / ACKNOWLEDGE M216-RADIAL LOCATOR RELAX FIXTURE 2
   RUNG wire#powerrail
      Contact( "M_ZERO" )
      Coil( "DB371_M_UNIT_SPARE".M_CODES_SPARE.Ack_M748 )
   END_RUNG
   // the same network as SCL:
   "DB371_M_UNIT_SPARE".M_CODES_SPARE.Ack_M748 := "M_ZERO";
END_REGION

REGION Network 50: M748-
   RUNG wire#powerrail
      Contact( "DB339_EXTENDED_M_SPARE".M_code[748] )
      wire#w1
      I_Contact( "DB371_M_UNIT_SPARE".M_CODES_SPARE.Ack_M748 )
      I_Contact( "DB2120_MPP_ITC_IPC".RESET_FAULTS )
      I_Contact( "DB371_M_UNIT_SPARE".M_CODES_SPARE.M_RESET_PULSE )
      Coil( "DB371_M_UNIT_SPARE".M_CODES_SPARE.M748 )
   END_RUNG
   RUNG wire#powerrail
      Contact( "DB371_M_UNIT_SPARE".M_CODES_SPARE.M748 )
   END_RUNG wire#w1
   // the same network as SCL:
   "DB371_M_UNIT_SPARE".M_CODES_SPARE.M748 := ("DB339_EXTENDED_M_SPARE".M_code[748] OR "DB371_M_UNIT_SPARE".M_CODES_SPARE.M748) AND NOT "DB371_M_UNIT_SPARE".M_CODES_SPARE.Ack_M748 AND NOT "DB2120_MPP_ITC_IPC".RESET_FAULTS AND NOT "DB371_M_UNIT_SPARE".M_CODES_SPARE.M_RESET_PULSE;
END_REGION

REGION Network 51: ACKNOWLEDGE M749- / ACKNOWLEDGE M23-SWITCH ON SPINDLE FRAME BLOWING
   RUNG wire#powerrail
      Contact( "M_ZERO" )
      Coil( "DB371_M_UNIT_SPARE".M_CODES_SPARE.Ack_M749 )
   END_RUNG
   // the same network as SCL:
   "DB371_M_UNIT_SPARE".M_CODES_SPARE.Ack_M749 := "M_ZERO";
END_REGION

REGION Network 52: M749- / M23-SWITCH ON SPINDLE FRAME BLOWING
   RUNG wire#powerrail
      Contact( "DB339_EXTENDED_M_SPARE".M_code[749] )
      wire#w1
      I_Contact( "DB371_M_UNIT_SPARE".M_CODES_SPARE.Ack_M749 )
      I_Contact( "DB2120_MPP_ITC_IPC".RESET_FAULTS )
      I_Contact( "DB371_M_UNIT_SPARE".M_CODES_SPARE.M_RESET_PULSE )
      Coil( "DB371_M_UNIT_SPARE".M_CODES_SPARE.M749 )
   END_RUNG
   RUNG wire#powerrail
      Contact( "DB371_M_UNIT_SPARE".M_CODES_SPARE.M749 )
   END_RUNG wire#w1
   // the same network as SCL:
   "DB371_M_UNIT_SPARE".M_CODES_SPARE.M749 := ("DB339_EXTENDED_M_SPARE".M_code[749] OR "DB371_M_UNIT_SPARE".M_CODES_SPARE.M749) AND NOT "DB371_M_UNIT_SPARE".M_CODES_SPARE.Ack_M749 AND NOT "DB2120_MPP_ITC_IPC".RESET_FAULTS AND NOT "DB371_M_UNIT_SPARE".M_CODES_SPARE.M_RESET_PULSE;
END_REGION

REGION Network 53: ACKNOWLEDGE M750-
   RUNG wire#powerrail
      Contact( "M_ZERO" )
      Coil( "DB371_M_UNIT_SPARE".M_CODES_SPARE.Ack_M750 )
   END_RUNG
   // the same network as SCL:
   "DB371_M_UNIT_SPARE".M_CODES_SPARE.Ack_M750 := "M_ZERO";
END_REGION

REGION Network 54: M750-
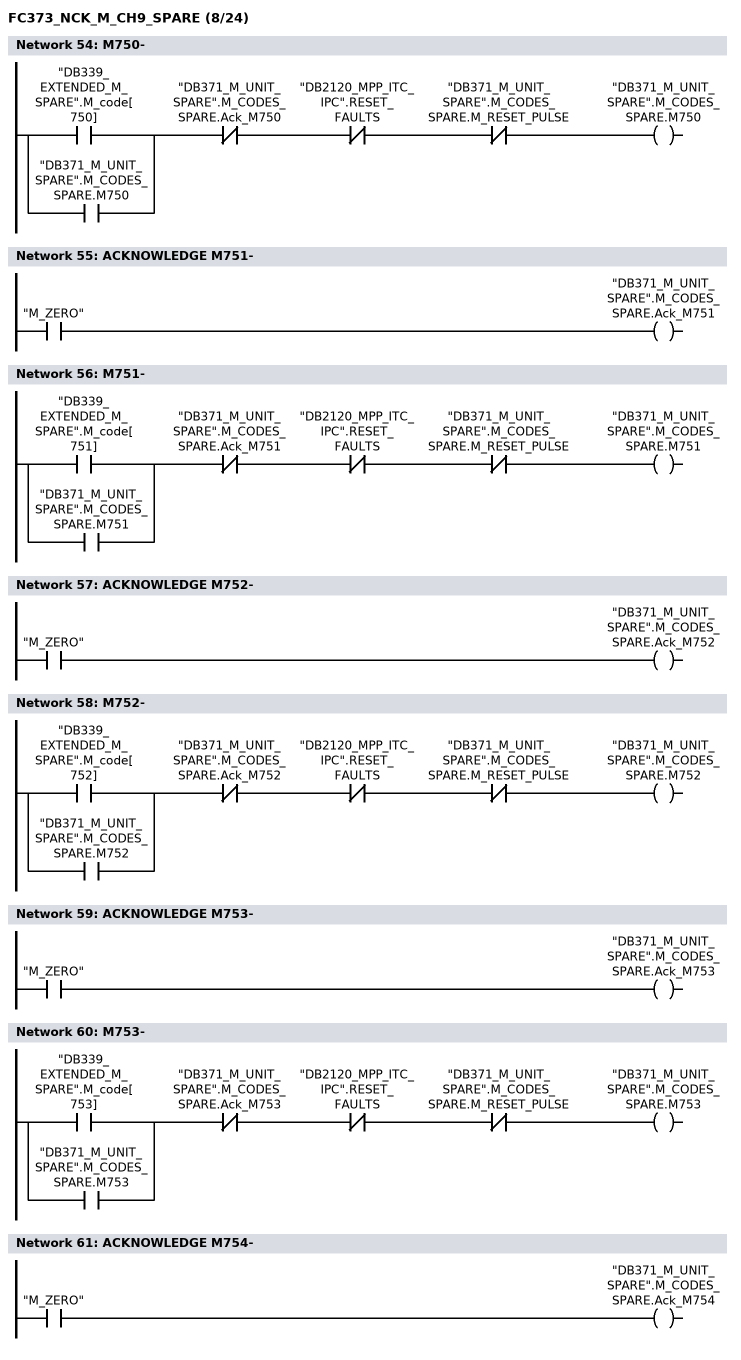
   RUNG wire#powerrail
      Contact( "DB339_EXTENDED_M_SPARE".M_code[750] )
      wire#w1
      I_Contact( "DB371_M_UNIT_SPARE".M_CODES_SPARE.Ack_M750 )
      I_Contact( "DB2120_MPP_ITC_IPC".RESET_FAULTS )
      I_Contact( "DB371_M_UNIT_SPARE".M_CODES_SPARE.M_RESET_PULSE )
      Coil( "DB371_M_UNIT_SPARE".M_CODES_SPARE.M750 )
   END_RUNG
   RUNG wire#powerrail
      Contact( "DB371_M_UNIT_SPARE".M_CODES_SPARE.M750 )
   END_RUNG wire#w1
   // the same network as SCL:
   "DB371_M_UNIT_SPARE".M_CODES_SPARE.M750 := ("DB339_EXTENDED_M_SPARE".M_code[750] OR "DB371_M_UNIT_SPARE".M_CODES_SPARE.M750) AND NOT "DB371_M_UNIT_SPARE".M_CODES_SPARE.Ack_M750 AND NOT "DB2120_MPP_ITC_IPC".RESET_FAULTS AND NOT "DB371_M_UNIT_SPARE".M_CODES_SPARE.M_RESET_PULSE;
END_REGION

REGION Network 55: ACKNOWLEDGE M751-
   RUNG wire#powerrail
      Contact( "M_ZERO" )
      Coil( "DB371_M_UNIT_SPARE".M_CODES_SPARE.Ack_M751 )
   END_RUNG
   // the same network as SCL:
   "DB371_M_UNIT_SPARE".M_CODES_SPARE.Ack_M751 := "M_ZERO";
END_REGION

REGION Network 56: M751-
   RUNG wire#powerrail
      Contact( "DB339_EXTENDED_M_SPARE".M_code[751] )
      wire#w1
      I_Contact( "DB371_M_UNIT_SPARE".M_CODES_SPARE.Ack_M751 )
      I_Contact( "DB2120_MPP_ITC_IPC".RESET_FAULTS )
      I_Contact( "DB371_M_UNIT_SPARE".M_CODES_SPARE.M_RESET_PULSE )
      Coil( "DB371_M_UNIT_SPARE".M_CODES_SPARE.M751 )
   END_RUNG
   RUNG wire#powerrail
      Contact( "DB371_M_UNIT_SPARE".M_CODES_SPARE.M751 )
   END_RUNG wire#w1
   // the same network as SCL:
   "DB371_M_UNIT_SPARE".M_CODES_SPARE.M751 := ("DB339_EXTENDED_M_SPARE".M_code[751] OR "DB371_M_UNIT_SPARE".M_CODES_SPARE.M751) AND NOT "DB371_M_UNIT_SPARE".M_CODES_SPARE.Ack_M751 AND NOT "DB2120_MPP_ITC_IPC".RESET_FAULTS AND NOT "DB371_M_UNIT_SPARE".M_CODES_SPARE.M_RESET_PULSE;
END_REGION

REGION Network 57: ACKNOWLEDGE M752-
   RUNG wire#powerrail
      Contact( "M_ZERO" )
      Coil( "DB371_M_UNIT_SPARE".M_CODES_SPARE.Ack_M752 )
   END_RUNG
   // the same network as SCL:
   "DB371_M_UNIT_SPARE".M_CODES_SPARE.Ack_M752 := "M_ZERO";
END_REGION

REGION Network 58: M752-
   RUNG wire#powerrail
      Contact( "DB339_EXTENDED_M_SPARE".M_code[752] )
      wire#w1
      I_Contact( "DB371_M_UNIT_SPARE".M_CODES_SPARE.Ack_M752 )
      I_Contact( "DB2120_MPP_ITC_IPC".RESET_FAULTS )
      I_Contact( "DB371_M_UNIT_SPARE".M_CODES_SPARE.M_RESET_PULSE )
      Coil( "DB371_M_UNIT_SPARE".M_CODES_SPARE.M752 )
   END_RUNG
   RUNG wire#powerrail
      Contact( "DB371_M_UNIT_SPARE".M_CODES_SPARE.M752 )
   END_RUNG wire#w1
   // the same network as SCL:
   "DB371_M_UNIT_SPARE".M_CODES_SPARE.M752 := ("DB339_EXTENDED_M_SPARE".M_code[752] OR "DB371_M_UNIT_SPARE".M_CODES_SPARE.M752) AND NOT "DB371_M_UNIT_SPARE".M_CODES_SPARE.Ack_M752 AND NOT "DB2120_MPP_ITC_IPC".RESET_FAULTS AND NOT "DB371_M_UNIT_SPARE".M_CODES_SPARE.M_RESET_PULSE;
END_REGION

REGION Network 59: ACKNOWLEDGE M753-
   RUNG wire#powerrail
      Contact( "M_ZERO" )
      Coil( "DB371_M_UNIT_SPARE".M_CODES_SPARE.Ack_M753 )
   END_RUNG
   // the same network as SCL:
   "DB371_M_UNIT_SPARE".M_CODES_SPARE.Ack_M753 := "M_ZERO";
END_REGION

REGION Network 60: M753-
   RUNG wire#powerrail
      Contact( "DB339_EXTENDED_M_SPARE".M_code[753] )
      wire#w1
      I_Contact( "DB371_M_UNIT_SPARE".M_CODES_SPARE.Ack_M753 )
      I_Contact( "DB2120_MPP_ITC_IPC".RESET_FAULTS )
      I_Contact( "DB371_M_UNIT_SPARE".M_CODES_SPARE.M_RESET_PULSE )
      Coil( "DB371_M_UNIT_SPARE".M_CODES_SPARE.M753 )
   END_RUNG
   RUNG wire#powerrail
      Contact( "DB371_M_UNIT_SPARE".M_CODES_SPARE.M753 )
   END_RUNG wire#w1
   // the same network as SCL:
   "DB371_M_UNIT_SPARE".M_CODES_SPARE.M753 := ("DB339_EXTENDED_M_SPARE".M_code[753] OR "DB371_M_UNIT_SPARE".M_CODES_SPARE.M753) AND NOT "DB371_M_UNIT_SPARE".M_CODES_SPARE.Ack_M753 AND NOT "DB2120_MPP_ITC_IPC".RESET_FAULTS AND NOT "DB371_M_UNIT_SPARE".M_CODES_SPARE.M_RESET_PULSE;
END_REGION

REGION Network 61: ACKNOWLEDGE M754-
   RUNG wire#powerrail
      Contact( "M_ZERO" )
      Coil( "DB371_M_UNIT_SPARE".M_CODES_SPARE.Ack_M754 )
   END_RUNG
   // the same network as SCL:
   "DB371_M_UNIT_SPARE".M_CODES_SPARE.Ack_M754 := "M_ZERO";
END_REGION

REGION Network 62: M754-
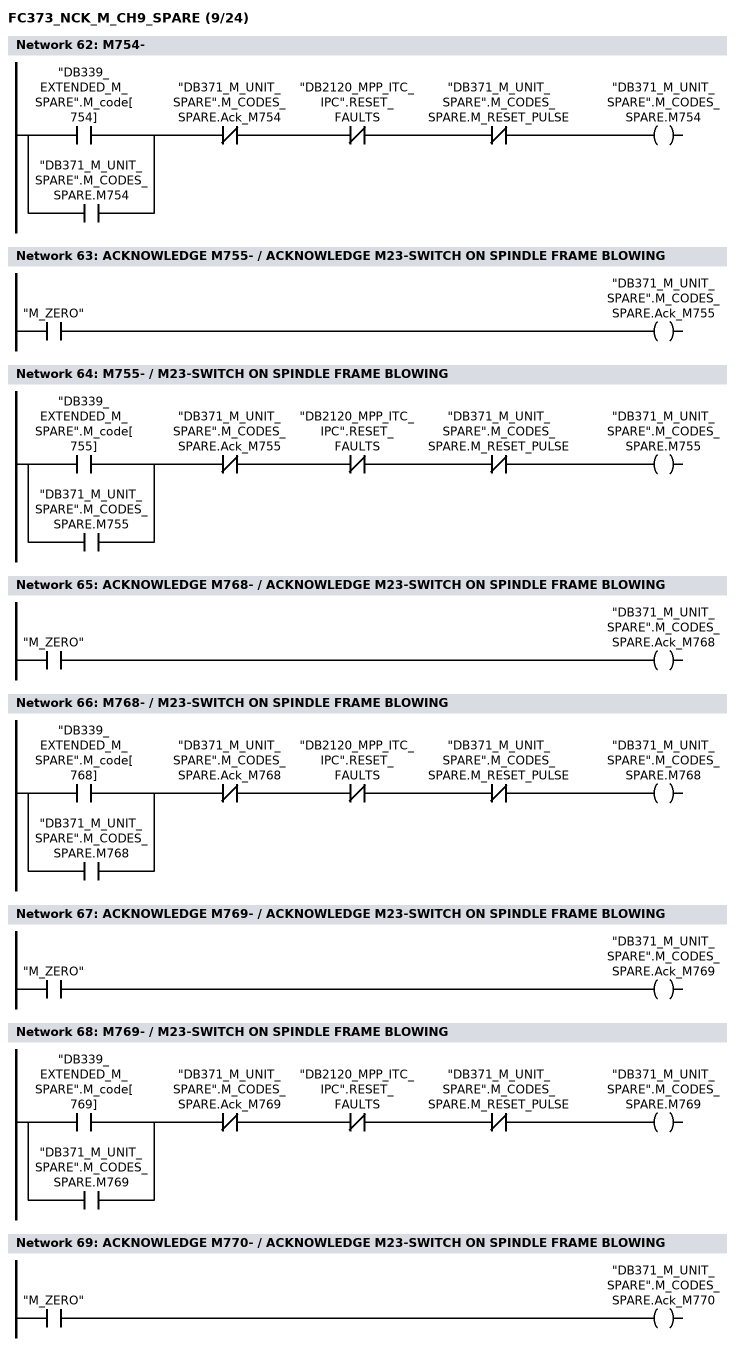
   RUNG wire#powerrail
      Contact( "DB339_EXTENDED_M_SPARE".M_code[754] )
      wire#w1
      I_Contact( "DB371_M_UNIT_SPARE".M_CODES_SPARE.Ack_M754 )
      I_Contact( "DB2120_MPP_ITC_IPC".RESET_FAULTS )
      I_Contact( "DB371_M_UNIT_SPARE".M_CODES_SPARE.M_RESET_PULSE )
      Coil( "DB371_M_UNIT_SPARE".M_CODES_SPARE.M754 )
   END_RUNG
   RUNG wire#powerrail
      Contact( "DB371_M_UNIT_SPARE".M_CODES_SPARE.M754 )
   END_RUNG wire#w1
   // the same network as SCL:
   "DB371_M_UNIT_SPARE".M_CODES_SPARE.M754 := ("DB339_EXTENDED_M_SPARE".M_code[754] OR "DB371_M_UNIT_SPARE".M_CODES_SPARE.M754) AND NOT "DB371_M_UNIT_SPARE".M_CODES_SPARE.Ack_M754 AND NOT "DB2120_MPP_ITC_IPC".RESET_FAULTS AND NOT "DB371_M_UNIT_SPARE".M_CODES_SPARE.M_RESET_PULSE;
END_REGION

REGION Network 63: ACKNOWLEDGE M755- / ACKNOWLEDGE M23-SWITCH ON SPINDLE FRAME BLOWING
   RUNG wire#powerrail
      Contact( "M_ZERO" )
      Coil( "DB371_M_UNIT_SPARE".M_CODES_SPARE.Ack_M755 )
   END_RUNG
   // the same network as SCL:
   "DB371_M_UNIT_SPARE".M_CODES_SPARE.Ack_M755 := "M_ZERO";
END_REGION

REGION Network 64: M755- / M23-SWITCH ON SPINDLE FRAME BLOWING
   RUNG wire#powerrail
      Contact( "DB339_EXTENDED_M_SPARE".M_code[755] )
      wire#w1
      I_Contact( "DB371_M_UNIT_SPARE".M_CODES_SPARE.Ack_M755 )
      I_Contact( "DB2120_MPP_ITC_IPC".RESET_FAULTS )
      I_Contact( "DB371_M_UNIT_SPARE".M_CODES_SPARE.M_RESET_PULSE )
      Coil( "DB371_M_UNIT_SPARE".M_CODES_SPARE.M755 )
   END_RUNG
   RUNG wire#powerrail
      Contact( "DB371_M_UNIT_SPARE".M_CODES_SPARE.M755 )
   END_RUNG wire#w1
   // the same network as SCL:
   "DB371_M_UNIT_SPARE".M_CODES_SPARE.M755 := ("DB339_EXTENDED_M_SPARE".M_code[755] OR "DB371_M_UNIT_SPARE".M_CODES_SPARE.M755) AND NOT "DB371_M_UNIT_SPARE".M_CODES_SPARE.Ack_M755 AND NOT "DB2120_MPP_ITC_IPC".RESET_FAULTS AND NOT "DB371_M_UNIT_SPARE".M_CODES_SPARE.M_RESET_PULSE;
END_REGION

REGION Network 65: ACKNOWLEDGE M768- / ACKNOWLEDGE M23-SWITCH ON SPINDLE FRAME BLOWING
   RUNG wire#powerrail
      Contact( "M_ZERO" )
      Coil( "DB371_M_UNIT_SPARE".M_CODES_SPARE.Ack_M768 )
   END_RUNG
   // the same network as SCL:
   "DB371_M_UNIT_SPARE".M_CODES_SPARE.Ack_M768 := "M_ZERO";
END_REGION

REGION Network 66: M768- / M23-SWITCH ON SPINDLE FRAME BLOWING
   RUNG wire#powerrail
      Contact( "DB339_EXTENDED_M_SPARE".M_code[768] )
      wire#w1
      I_Contact( "DB371_M_UNIT_SPARE".M_CODES_SPARE.Ack_M768 )
      I_Contact( "DB2120_MPP_ITC_IPC".RESET_FAULTS )
      I_Contact( "DB371_M_UNIT_SPARE".M_CODES_SPARE.M_RESET_PULSE )
      Coil( "DB371_M_UNIT_SPARE".M_CODES_SPARE.M768 )
   END_RUNG
   RUNG wire#powerrail
      Contact( "DB371_M_UNIT_SPARE".M_CODES_SPARE.M768 )
   END_RUNG wire#w1
   // the same network as SCL:
   "DB371_M_UNIT_SPARE".M_CODES_SPARE.M768 := ("DB339_EXTENDED_M_SPARE".M_code[768] OR "DB371_M_UNIT_SPARE".M_CODES_SPARE.M768) AND NOT "DB371_M_UNIT_SPARE".M_CODES_SPARE.Ack_M768 AND NOT "DB2120_MPP_ITC_IPC".RESET_FAULTS AND NOT "DB371_M_UNIT_SPARE".M_CODES_SPARE.M_RESET_PULSE;
END_REGION

REGION Network 67: ACKNOWLEDGE M769- / ACKNOWLEDGE M23-SWITCH ON SPINDLE FRAME BLOWING
   RUNG wire#powerrail
      Contact( "M_ZERO" )
      Coil( "DB371_M_UNIT_SPARE".M_CODES_SPARE.Ack_M769 )
   END_RUNG
   // the same network as SCL:
   "DB371_M_UNIT_SPARE".M_CODES_SPARE.Ack_M769 := "M_ZERO";
END_REGION

REGION Network 68: M769- / M23-SWITCH ON SPINDLE FRAME BLOWING
   RUNG wire#powerrail
      Contact( "DB339_EXTENDED_M_SPARE".M_code[769] )
      wire#w1
      I_Contact( "DB371_M_UNIT_SPARE".M_CODES_SPARE.Ack_M769 )
      I_Contact( "DB2120_MPP_ITC_IPC".RESET_FAULTS )
      I_Contact( "DB371_M_UNIT_SPARE".M_CODES_SPARE.M_RESET_PULSE )
      Coil( "DB371_M_UNIT_SPARE".M_CODES_SPARE.M769 )
   END_RUNG
   RUNG wire#powerrail
      Contact( "DB371_M_UNIT_SPARE".M_CODES_SPARE.M769 )
   END_RUNG wire#w1
   // the same network as SCL:
   "DB371_M_UNIT_SPARE".M_CODES_SPARE.M769 := ("DB339_EXTENDED_M_SPARE".M_code[769] OR "DB371_M_UNIT_SPARE".M_CODES_SPARE.M769) AND NOT "DB371_M_UNIT_SPARE".M_CODES_SPARE.Ack_M769 AND NOT "DB2120_MPP_ITC_IPC".RESET_FAULTS AND NOT "DB371_M_UNIT_SPARE".M_CODES_SPARE.M_RESET_PULSE;
END_REGION

REGION Network 69: ACKNOWLEDGE M770- / ACKNOWLEDGE M23-SWITCH ON SPINDLE FRAME BLOWING
   RUNG wire#powerrail
      Contact( "M_ZERO" )
      Coil( "DB371_M_UNIT_SPARE".M_CODES_SPARE.Ack_M770 )
   END_RUNG
   // the same network as SCL:
   "DB371_M_UNIT_SPARE".M_CODES_SPARE.Ack_M770 := "M_ZERO";
END_REGION

REGION Network 70: M770- / M23-SWITCH ON SPINDLE FRAME BLOWING
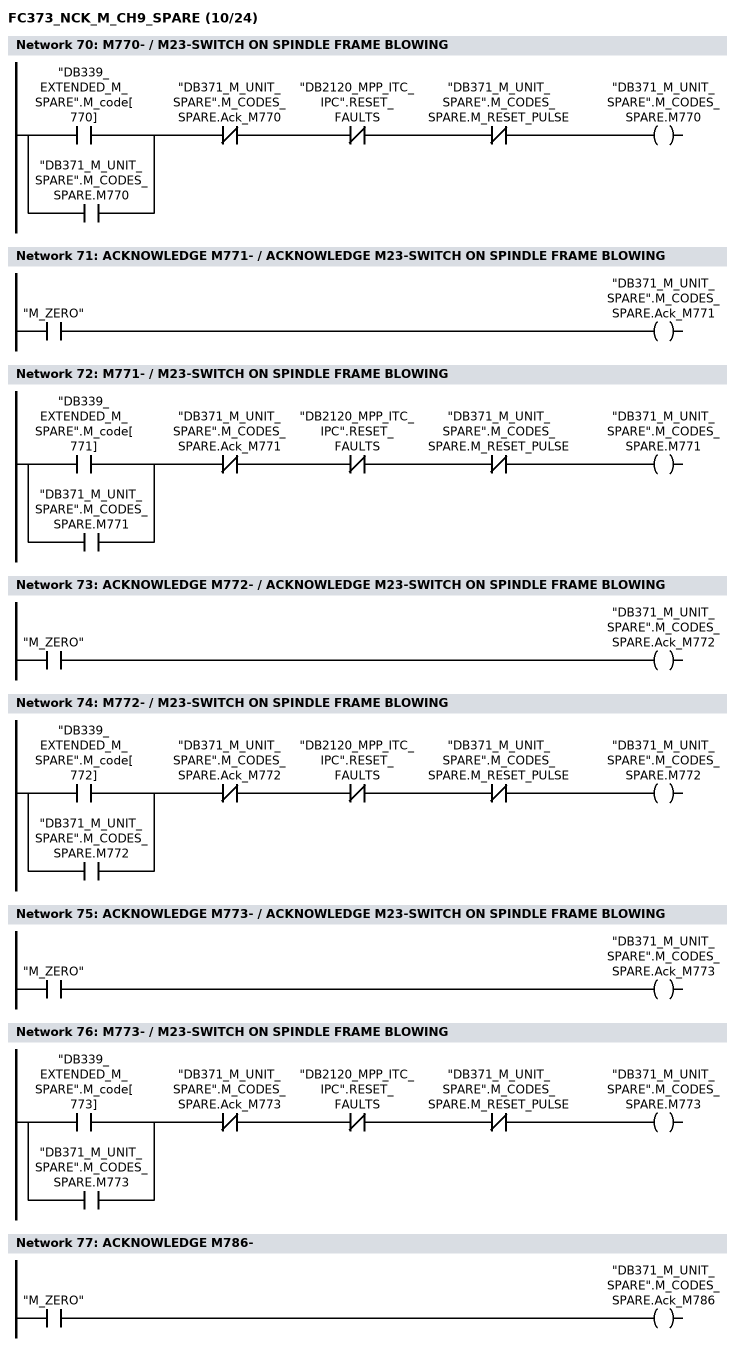
   RUNG wire#powerrail
      Contact( "DB339_EXTENDED_M_SPARE".M_code[770] )
      wire#w1
      I_Contact( "DB371_M_UNIT_SPARE".M_CODES_SPARE.Ack_M770 )
      I_Contact( "DB2120_MPP_ITC_IPC".RESET_FAULTS )
      I_Contact( "DB371_M_UNIT_SPARE".M_CODES_SPARE.M_RESET_PULSE )
      Coil( "DB371_M_UNIT_SPARE".M_CODES_SPARE.M770 )
   END_RUNG
   RUNG wire#powerrail
      Contact( "DB371_M_UNIT_SPARE".M_CODES_SPARE.M770 )
   END_RUNG wire#w1
   // the same network as SCL:
   "DB371_M_UNIT_SPARE".M_CODES_SPARE.M770 := ("DB339_EXTENDED_M_SPARE".M_code[770] OR "DB371_M_UNIT_SPARE".M_CODES_SPARE.M770) AND NOT "DB371_M_UNIT_SPARE".M_CODES_SPARE.Ack_M770 AND NOT "DB2120_MPP_ITC_IPC".RESET_FAULTS AND NOT "DB371_M_UNIT_SPARE".M_CODES_SPARE.M_RESET_PULSE;
END_REGION

REGION Network 71: ACKNOWLEDGE M771- / ACKNOWLEDGE M23-SWITCH ON SPINDLE FRAME BLOWING
   RUNG wire#powerrail
      Contact( "M_ZERO" )
      Coil( "DB371_M_UNIT_SPARE".M_CODES_SPARE.Ack_M771 )
   END_RUNG
   // the same network as SCL:
   "DB371_M_UNIT_SPARE".M_CODES_SPARE.Ack_M771 := "M_ZERO";
END_REGION

REGION Network 72: M771- / M23-SWITCH ON SPINDLE FRAME BLOWING
   RUNG wire#powerrail
      Contact( "DB339_EXTENDED_M_SPARE".M_code[771] )
      wire#w1
      I_Contact( "DB371_M_UNIT_SPARE".M_CODES_SPARE.Ack_M771 )
      I_Contact( "DB2120_MPP_ITC_IPC".RESET_FAULTS )
      I_Contact( "DB371_M_UNIT_SPARE".M_CODES_SPARE.M_RESET_PULSE )
      Coil( "DB371_M_UNIT_SPARE".M_CODES_SPARE.M771 )
   END_RUNG
   RUNG wire#powerrail
      Contact( "DB371_M_UNIT_SPARE".M_CODES_SPARE.M771 )
   END_RUNG wire#w1
   // the same network as SCL:
   "DB371_M_UNIT_SPARE".M_CODES_SPARE.M771 := ("DB339_EXTENDED_M_SPARE".M_code[771] OR "DB371_M_UNIT_SPARE".M_CODES_SPARE.M771) AND NOT "DB371_M_UNIT_SPARE".M_CODES_SPARE.Ack_M771 AND NOT "DB2120_MPP_ITC_IPC".RESET_FAULTS AND NOT "DB371_M_UNIT_SPARE".M_CODES_SPARE.M_RESET_PULSE;
END_REGION

REGION Network 73: ACKNOWLEDGE M772- / ACKNOWLEDGE M23-SWITCH ON SPINDLE FRAME BLOWING
   RUNG wire#powerrail
      Contact( "M_ZERO" )
      Coil( "DB371_M_UNIT_SPARE".M_CODES_SPARE.Ack_M772 )
   END_RUNG
   // the same network as SCL:
   "DB371_M_UNIT_SPARE".M_CODES_SPARE.Ack_M772 := "M_ZERO";
END_REGION

REGION Network 74: M772- / M23-SWITCH ON SPINDLE FRAME BLOWING
   RUNG wire#powerrail
      Contact( "DB339_EXTENDED_M_SPARE".M_code[772] )
      wire#w1
      I_Contact( "DB371_M_UNIT_SPARE".M_CODES_SPARE.Ack_M772 )
      I_Contact( "DB2120_MPP_ITC_IPC".RESET_FAULTS )
      I_Contact( "DB371_M_UNIT_SPARE".M_CODES_SPARE.M_RESET_PULSE )
      Coil( "DB371_M_UNIT_SPARE".M_CODES_SPARE.M772 )
   END_RUNG
   RUNG wire#powerrail
      Contact( "DB371_M_UNIT_SPARE".M_CODES_SPARE.M772 )
   END_RUNG wire#w1
   // the same network as SCL:
   "DB371_M_UNIT_SPARE".M_CODES_SPARE.M772 := ("DB339_EXTENDED_M_SPARE".M_code[772] OR "DB371_M_UNIT_SPARE".M_CODES_SPARE.M772) AND NOT "DB371_M_UNIT_SPARE".M_CODES_SPARE.Ack_M772 AND NOT "DB2120_MPP_ITC_IPC".RESET_FAULTS AND NOT "DB371_M_UNIT_SPARE".M_CODES_SPARE.M_RESET_PULSE;
END_REGION

REGION Network 75: ACKNOWLEDGE M773- / ACKNOWLEDGE M23-SWITCH ON SPINDLE FRAME BLOWING
   RUNG wire#powerrail
      Contact( "M_ZERO" )
      Coil( "DB371_M_UNIT_SPARE".M_CODES_SPARE.Ack_M773 )
   END_RUNG
   // the same network as SCL:
   "DB371_M_UNIT_SPARE".M_CODES_SPARE.Ack_M773 := "M_ZERO";
END_REGION

REGION Network 76: M773- / M23-SWITCH ON SPINDLE FRAME BLOWING
   RUNG wire#powerrail
      Contact( "DB339_EXTENDED_M_SPARE".M_code[773] )
      wire#w1
      I_Contact( "DB371_M_UNIT_SPARE".M_CODES_SPARE.Ack_M773 )
      I_Contact( "DB2120_MPP_ITC_IPC".RESET_FAULTS )
      I_Contact( "DB371_M_UNIT_SPARE".M_CODES_SPARE.M_RESET_PULSE )
      Coil( "DB371_M_UNIT_SPARE".M_CODES_SPARE.M773 )
   END_RUNG
   RUNG wire#powerrail
      Contact( "DB371_M_UNIT_SPARE".M_CODES_SPARE.M773 )
   END_RUNG wire#w1
   // the same network as SCL:
   "DB371_M_UNIT_SPARE".M_CODES_SPARE.M773 := ("DB339_EXTENDED_M_SPARE".M_code[773] OR "DB371_M_UNIT_SPARE".M_CODES_SPARE.M773) AND NOT "DB371_M_UNIT_SPARE".M_CODES_SPARE.Ack_M773 AND NOT "DB2120_MPP_ITC_IPC".RESET_FAULTS AND NOT "DB371_M_UNIT_SPARE".M_CODES_SPARE.M_RESET_PULSE;
END_REGION

REGION Network 77: ACKNOWLEDGE M786-
   RUNG wire#powerrail
      Contact( "M_ZERO" )
      Coil( "DB371_M_UNIT_SPARE".M_CODES_SPARE.Ack_M786 )
   END_RUNG
   // the same network as SCL:
   "DB371_M_UNIT_SPARE".M_CODES_SPARE.Ack_M786 := "M_ZERO";
END_REGION

REGION Network 78: M786-
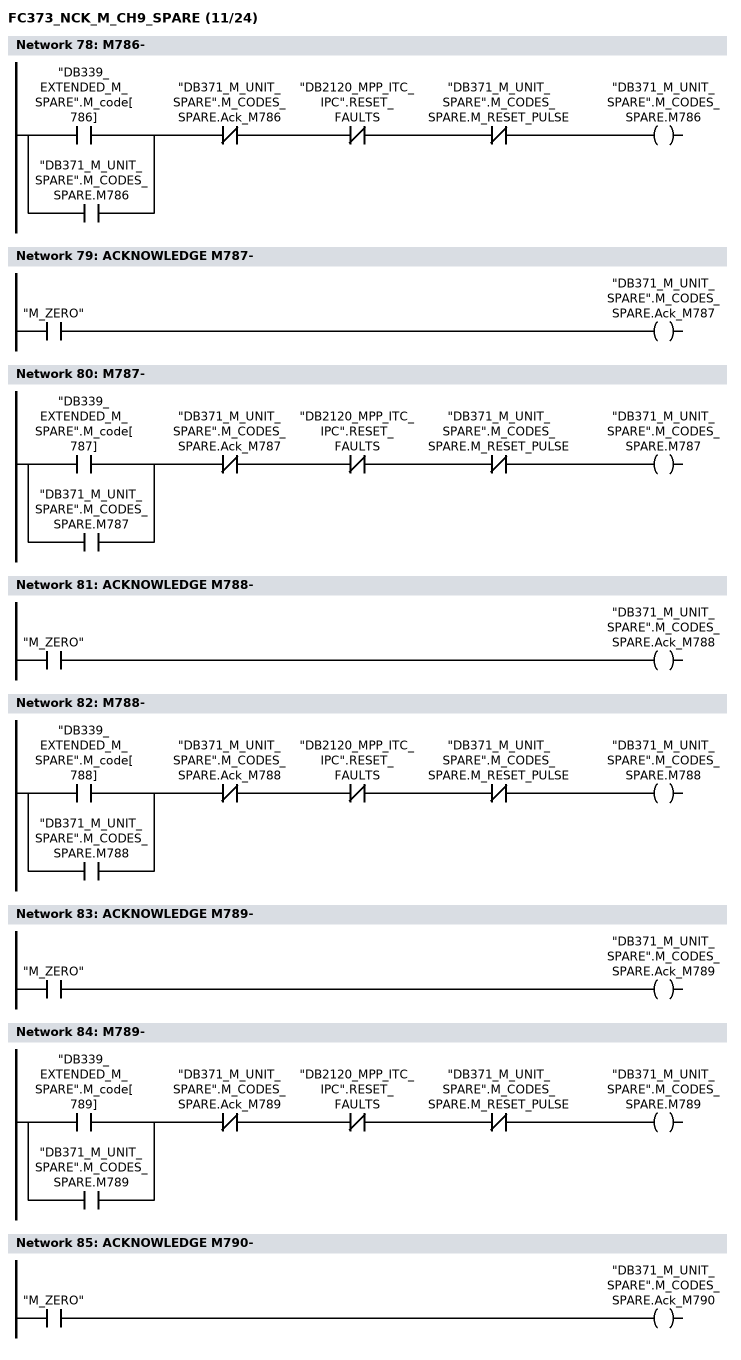
   RUNG wire#powerrail
      Contact( "DB339_EXTENDED_M_SPARE".M_code[786] )
      wire#w1
      I_Contact( "DB371_M_UNIT_SPARE".M_CODES_SPARE.Ack_M786 )
      I_Contact( "DB2120_MPP_ITC_IPC".RESET_FAULTS )
      I_Contact( "DB371_M_UNIT_SPARE".M_CODES_SPARE.M_RESET_PULSE )
      Coil( "DB371_M_UNIT_SPARE".M_CODES_SPARE.M786 )
   END_RUNG
   RUNG wire#powerrail
      Contact( "DB371_M_UNIT_SPARE".M_CODES_SPARE.M786 )
   END_RUNG wire#w1
   // the same network as SCL:
   "DB371_M_UNIT_SPARE".M_CODES_SPARE.M786 := ("DB339_EXTENDED_M_SPARE".M_code[786] OR "DB371_M_UNIT_SPARE".M_CODES_SPARE.M786) AND NOT "DB371_M_UNIT_SPARE".M_CODES_SPARE.Ack_M786 AND NOT "DB2120_MPP_ITC_IPC".RESET_FAULTS AND NOT "DB371_M_UNIT_SPARE".M_CODES_SPARE.M_RESET_PULSE;
END_REGION

REGION Network 79: ACKNOWLEDGE M787-
   RUNG wire#powerrail
      Contact( "M_ZERO" )
      Coil( "DB371_M_UNIT_SPARE".M_CODES_SPARE.Ack_M787 )
   END_RUNG
   // the same network as SCL:
   "DB371_M_UNIT_SPARE".M_CODES_SPARE.Ack_M787 := "M_ZERO";
END_REGION

REGION Network 80: M787-
   RUNG wire#powerrail
      Contact( "DB339_EXTENDED_M_SPARE".M_code[787] )
      wire#w1
      I_Contact( "DB371_M_UNIT_SPARE".M_CODES_SPARE.Ack_M787 )
      I_Contact( "DB2120_MPP_ITC_IPC".RESET_FAULTS )
      I_Contact( "DB371_M_UNIT_SPARE".M_CODES_SPARE.M_RESET_PULSE )
      Coil( "DB371_M_UNIT_SPARE".M_CODES_SPARE.M787 )
   END_RUNG
   RUNG wire#powerrail
      Contact( "DB371_M_UNIT_SPARE".M_CODES_SPARE.M787 )
   END_RUNG wire#w1
   // the same network as SCL:
   "DB371_M_UNIT_SPARE".M_CODES_SPARE.M787 := ("DB339_EXTENDED_M_SPARE".M_code[787] OR "DB371_M_UNIT_SPARE".M_CODES_SPARE.M787) AND NOT "DB371_M_UNIT_SPARE".M_CODES_SPARE.Ack_M787 AND NOT "DB2120_MPP_ITC_IPC".RESET_FAULTS AND NOT "DB371_M_UNIT_SPARE".M_CODES_SPARE.M_RESET_PULSE;
END_REGION

REGION Network 81: ACKNOWLEDGE M788-
   RUNG wire#powerrail
      Contact( "M_ZERO" )
      Coil( "DB371_M_UNIT_SPARE".M_CODES_SPARE.Ack_M788 )
   END_RUNG
   // the same network as SCL:
   "DB371_M_UNIT_SPARE".M_CODES_SPARE.Ack_M788 := "M_ZERO";
END_REGION

REGION Network 82: M788-
   RUNG wire#powerrail
      Contact( "DB339_EXTENDED_M_SPARE".M_code[788] )
      wire#w1
      I_Contact( "DB371_M_UNIT_SPARE".M_CODES_SPARE.Ack_M788 )
      I_Contact( "DB2120_MPP_ITC_IPC".RESET_FAULTS )
      I_Contact( "DB371_M_UNIT_SPARE".M_CODES_SPARE.M_RESET_PULSE )
      Coil( "DB371_M_UNIT_SPARE".M_CODES_SPARE.M788 )
   END_RUNG
   RUNG wire#powerrail
      Contact( "DB371_M_UNIT_SPARE".M_CODES_SPARE.M788 )
   END_RUNG wire#w1
   // the same network as SCL:
   "DB371_M_UNIT_SPARE".M_CODES_SPARE.M788 := ("DB339_EXTENDED_M_SPARE".M_code[788] OR "DB371_M_UNIT_SPARE".M_CODES_SPARE.M788) AND NOT "DB371_M_UNIT_SPARE".M_CODES_SPARE.Ack_M788 AND NOT "DB2120_MPP_ITC_IPC".RESET_FAULTS AND NOT "DB371_M_UNIT_SPARE".M_CODES_SPARE.M_RESET_PULSE;
END_REGION

REGION Network 83: ACKNOWLEDGE M789-
   RUNG wire#powerrail
      Contact( "M_ZERO" )
      Coil( "DB371_M_UNIT_SPARE".M_CODES_SPARE.Ack_M789 )
   END_RUNG
   // the same network as SCL:
   "DB371_M_UNIT_SPARE".M_CODES_SPARE.Ack_M789 := "M_ZERO";
END_REGION

REGION Network 84: M789-
   RUNG wire#powerrail
      Contact( "DB339_EXTENDED_M_SPARE".M_code[789] )
      wire#w1
      I_Contact( "DB371_M_UNIT_SPARE".M_CODES_SPARE.Ack_M789 )
      I_Contact( "DB2120_MPP_ITC_IPC".RESET_FAULTS )
      I_Contact( "DB371_M_UNIT_SPARE".M_CODES_SPARE.M_RESET_PULSE )
      Coil( "DB371_M_UNIT_SPARE".M_CODES_SPARE.M789 )
   END_RUNG
   RUNG wire#powerrail
      Contact( "DB371_M_UNIT_SPARE".M_CODES_SPARE.M789 )
   END_RUNG wire#w1
   // the same network as SCL:
   "DB371_M_UNIT_SPARE".M_CODES_SPARE.M789 := ("DB339_EXTENDED_M_SPARE".M_code[789] OR "DB371_M_UNIT_SPARE".M_CODES_SPARE.M789) AND NOT "DB371_M_UNIT_SPARE".M_CODES_SPARE.Ack_M789 AND NOT "DB2120_MPP_ITC_IPC".RESET_FAULTS AND NOT "DB371_M_UNIT_SPARE".M_CODES_SPARE.M_RESET_PULSE;
END_REGION

REGION Network 85: ACKNOWLEDGE M790-
   RUNG wire#powerrail
      Contact( "M_ZERO" )
      Coil( "DB371_M_UNIT_SPARE".M_CODES_SPARE.Ack_M790 )
   END_RUNG
   // the same network as SCL:
   "DB371_M_UNIT_SPARE".M_CODES_SPARE.Ack_M790 := "M_ZERO";
END_REGION

REGION Network 86: M790-
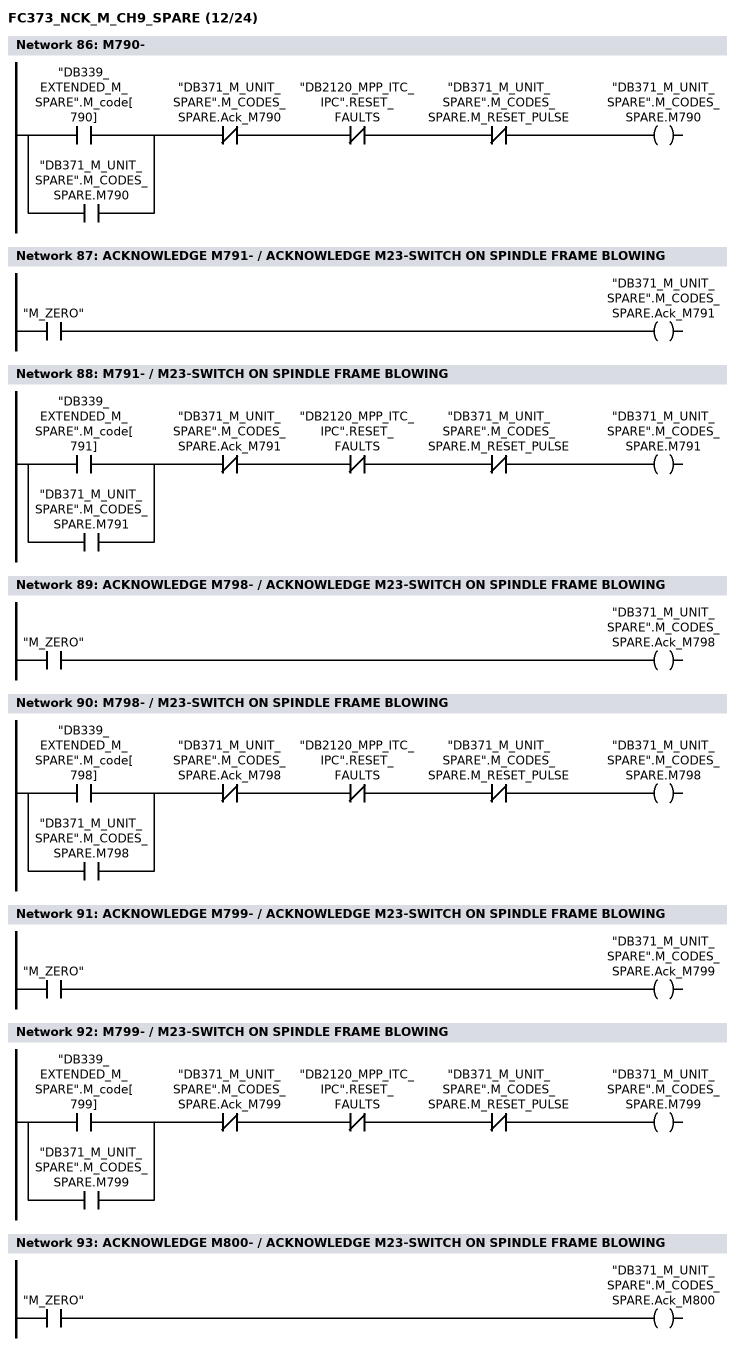
   RUNG wire#powerrail
      Contact( "DB339_EXTENDED_M_SPARE".M_code[790] )
      wire#w1
      I_Contact( "DB371_M_UNIT_SPARE".M_CODES_SPARE.Ack_M790 )
      I_Contact( "DB2120_MPP_ITC_IPC".RESET_FAULTS )
      I_Contact( "DB371_M_UNIT_SPARE".M_CODES_SPARE.M_RESET_PULSE )
      Coil( "DB371_M_UNIT_SPARE".M_CODES_SPARE.M790 )
   END_RUNG
   RUNG wire#powerrail
      Contact( "DB371_M_UNIT_SPARE".M_CODES_SPARE.M790 )
   END_RUNG wire#w1
   // the same network as SCL:
   "DB371_M_UNIT_SPARE".M_CODES_SPARE.M790 := ("DB339_EXTENDED_M_SPARE".M_code[790] OR "DB371_M_UNIT_SPARE".M_CODES_SPARE.M790) AND NOT "DB371_M_UNIT_SPARE".M_CODES_SPARE.Ack_M790 AND NOT "DB2120_MPP_ITC_IPC".RESET_FAULTS AND NOT "DB371_M_UNIT_SPARE".M_CODES_SPARE.M_RESET_PULSE;
END_REGION

REGION Network 87: ACKNOWLEDGE M791- / ACKNOWLEDGE M23-SWITCH ON SPINDLE FRAME BLOWING
   RUNG wire#powerrail
      Contact( "M_ZERO" )
      Coil( "DB371_M_UNIT_SPARE".M_CODES_SPARE.Ack_M791 )
   END_RUNG
   // the same network as SCL:
   "DB371_M_UNIT_SPARE".M_CODES_SPARE.Ack_M791 := "M_ZERO";
END_REGION

REGION Network 88: M791- / M23-SWITCH ON SPINDLE FRAME BLOWING
   RUNG wire#powerrail
      Contact( "DB339_EXTENDED_M_SPARE".M_code[791] )
      wire#w1
      I_Contact( "DB371_M_UNIT_SPARE".M_CODES_SPARE.Ack_M791 )
      I_Contact( "DB2120_MPP_ITC_IPC".RESET_FAULTS )
      I_Contact( "DB371_M_UNIT_SPARE".M_CODES_SPARE.M_RESET_PULSE )
      Coil( "DB371_M_UNIT_SPARE".M_CODES_SPARE.M791 )
   END_RUNG
   RUNG wire#powerrail
      Contact( "DB371_M_UNIT_SPARE".M_CODES_SPARE.M791 )
   END_RUNG wire#w1
   // the same network as SCL:
   "DB371_M_UNIT_SPARE".M_CODES_SPARE.M791 := ("DB339_EXTENDED_M_SPARE".M_code[791] OR "DB371_M_UNIT_SPARE".M_CODES_SPARE.M791) AND NOT "DB371_M_UNIT_SPARE".M_CODES_SPARE.Ack_M791 AND NOT "DB2120_MPP_ITC_IPC".RESET_FAULTS AND NOT "DB371_M_UNIT_SPARE".M_CODES_SPARE.M_RESET_PULSE;
END_REGION

REGION Network 89: ACKNOWLEDGE M798- / ACKNOWLEDGE M23-SWITCH ON SPINDLE FRAME BLOWING
   RUNG wire#powerrail
      Contact( "M_ZERO" )
      Coil( "DB371_M_UNIT_SPARE".M_CODES_SPARE.Ack_M798 )
   END_RUNG
   // the same network as SCL:
   "DB371_M_UNIT_SPARE".M_CODES_SPARE.Ack_M798 := "M_ZERO";
END_REGION

REGION Network 90: M798- / M23-SWITCH ON SPINDLE FRAME BLOWING
   RUNG wire#powerrail
      Contact( "DB339_EXTENDED_M_SPARE".M_code[798] )
      wire#w1
      I_Contact( "DB371_M_UNIT_SPARE".M_CODES_SPARE.Ack_M798 )
      I_Contact( "DB2120_MPP_ITC_IPC".RESET_FAULTS )
      I_Contact( "DB371_M_UNIT_SPARE".M_CODES_SPARE.M_RESET_PULSE )
      Coil( "DB371_M_UNIT_SPARE".M_CODES_SPARE.M798 )
   END_RUNG
   RUNG wire#powerrail
      Contact( "DB371_M_UNIT_SPARE".M_CODES_SPARE.M798 )
   END_RUNG wire#w1
   // the same network as SCL:
   "DB371_M_UNIT_SPARE".M_CODES_SPARE.M798 := ("DB339_EXTENDED_M_SPARE".M_code[798] OR "DB371_M_UNIT_SPARE".M_CODES_SPARE.M798) AND NOT "DB371_M_UNIT_SPARE".M_CODES_SPARE.Ack_M798 AND NOT "DB2120_MPP_ITC_IPC".RESET_FAULTS AND NOT "DB371_M_UNIT_SPARE".M_CODES_SPARE.M_RESET_PULSE;
END_REGION

REGION Network 91: ACKNOWLEDGE M799- / ACKNOWLEDGE M23-SWITCH ON SPINDLE FRAME BLOWING
   RUNG wire#powerrail
      Contact( "M_ZERO" )
      Coil( "DB371_M_UNIT_SPARE".M_CODES_SPARE.Ack_M799 )
   END_RUNG
   // the same network as SCL:
   "DB371_M_UNIT_SPARE".M_CODES_SPARE.Ack_M799 := "M_ZERO";
END_REGION

REGION Network 92: M799- / M23-SWITCH ON SPINDLE FRAME BLOWING
   RUNG wire#powerrail
      Contact( "DB339_EXTENDED_M_SPARE".M_code[799] )
      wire#w1
      I_Contact( "DB371_M_UNIT_SPARE".M_CODES_SPARE.Ack_M799 )
      I_Contact( "DB2120_MPP_ITC_IPC".RESET_FAULTS )
      I_Contact( "DB371_M_UNIT_SPARE".M_CODES_SPARE.M_RESET_PULSE )
      Coil( "DB371_M_UNIT_SPARE".M_CODES_SPARE.M799 )
   END_RUNG
   RUNG wire#powerrail
      Contact( "DB371_M_UNIT_SPARE".M_CODES_SPARE.M799 )
   END_RUNG wire#w1
   // the same network as SCL:
   "DB371_M_UNIT_SPARE".M_CODES_SPARE.M799 := ("DB339_EXTENDED_M_SPARE".M_code[799] OR "DB371_M_UNIT_SPARE".M_CODES_SPARE.M799) AND NOT "DB371_M_UNIT_SPARE".M_CODES_SPARE.Ack_M799 AND NOT "DB2120_MPP_ITC_IPC".RESET_FAULTS AND NOT "DB371_M_UNIT_SPARE".M_CODES_SPARE.M_RESET_PULSE;
END_REGION

REGION Network 93: ACKNOWLEDGE M800- / ACKNOWLEDGE M23-SWITCH ON SPINDLE FRAME BLOWING
   RUNG wire#powerrail
      Contact( "M_ZERO" )
      Coil( "DB371_M_UNIT_SPARE".M_CODES_SPARE.Ack_M800 )
   END_RUNG
   // the same network as SCL:
   "DB371_M_UNIT_SPARE".M_CODES_SPARE.Ack_M800 := "M_ZERO";
END_REGION

REGION Network 94: M800- / M23-SWITCH ON SPINDLE FRAME BLOWING
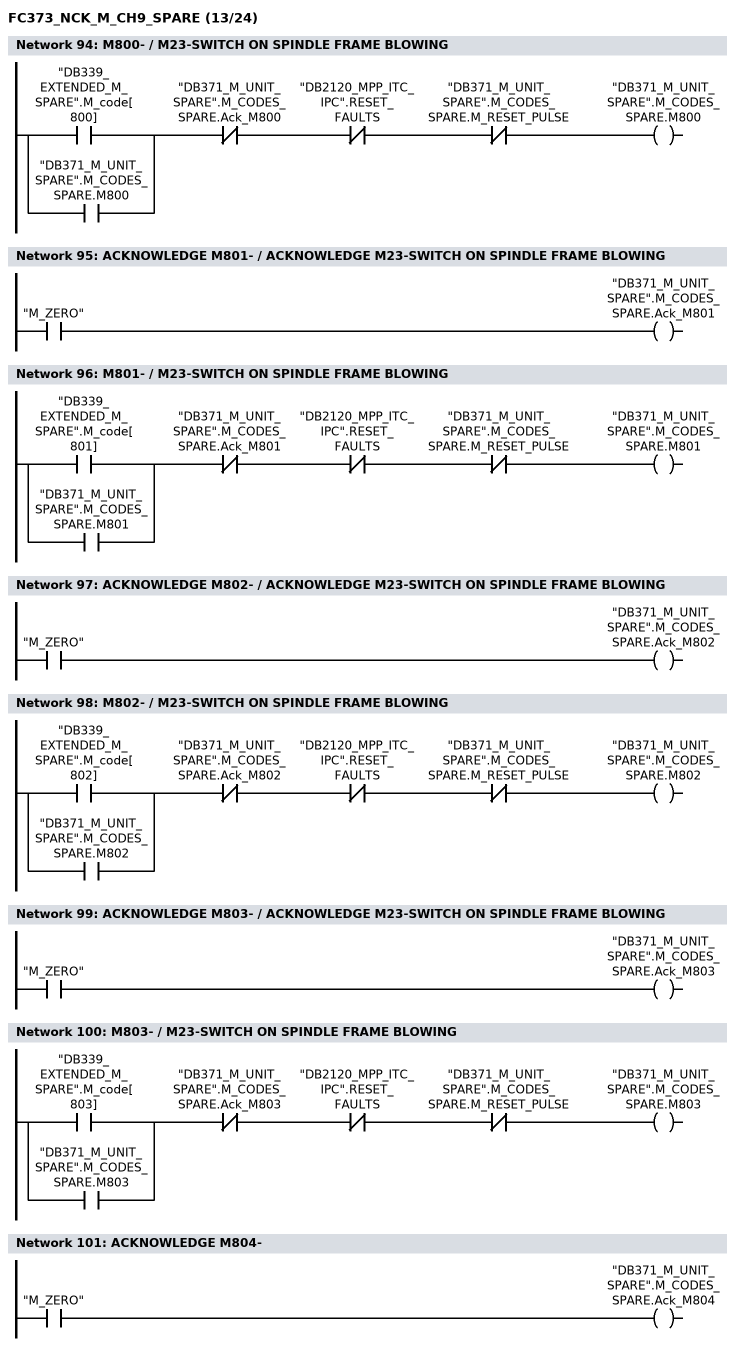
   RUNG wire#powerrail
      Contact( "DB339_EXTENDED_M_SPARE".M_code[800] )
      wire#w1
      I_Contact( "DB371_M_UNIT_SPARE".M_CODES_SPARE.Ack_M800 )
      I_Contact( "DB2120_MPP_ITC_IPC".RESET_FAULTS )
      I_Contact( "DB371_M_UNIT_SPARE".M_CODES_SPARE.M_RESET_PULSE )
      Coil( "DB371_M_UNIT_SPARE".M_CODES_SPARE.M800 )
   END_RUNG
   RUNG wire#powerrail
      Contact( "DB371_M_UNIT_SPARE".M_CODES_SPARE.M800 )
   END_RUNG wire#w1
   // the same network as SCL:
   "DB371_M_UNIT_SPARE".M_CODES_SPARE.M800 := ("DB339_EXTENDED_M_SPARE".M_code[800] OR "DB371_M_UNIT_SPARE".M_CODES_SPARE.M800) AND NOT "DB371_M_UNIT_SPARE".M_CODES_SPARE.Ack_M800 AND NOT "DB2120_MPP_ITC_IPC".RESET_FAULTS AND NOT "DB371_M_UNIT_SPARE".M_CODES_SPARE.M_RESET_PULSE;
END_REGION

REGION Network 95: ACKNOWLEDGE M801- / ACKNOWLEDGE M23-SWITCH ON SPINDLE FRAME BLOWING
   RUNG wire#powerrail
      Contact( "M_ZERO" )
      Coil( "DB371_M_UNIT_SPARE".M_CODES_SPARE.Ack_M801 )
   END_RUNG
   // the same network as SCL:
   "DB371_M_UNIT_SPARE".M_CODES_SPARE.Ack_M801 := "M_ZERO";
END_REGION

REGION Network 96: M801- / M23-SWITCH ON SPINDLE FRAME BLOWING
   RUNG wire#powerrail
      Contact( "DB339_EXTENDED_M_SPARE".M_code[801] )
      wire#w1
      I_Contact( "DB371_M_UNIT_SPARE".M_CODES_SPARE.Ack_M801 )
      I_Contact( "DB2120_MPP_ITC_IPC".RESET_FAULTS )
      I_Contact( "DB371_M_UNIT_SPARE".M_CODES_SPARE.M_RESET_PULSE )
      Coil( "DB371_M_UNIT_SPARE".M_CODES_SPARE.M801 )
   END_RUNG
   RUNG wire#powerrail
      Contact( "DB371_M_UNIT_SPARE".M_CODES_SPARE.M801 )
   END_RUNG wire#w1
   // the same network as SCL:
   "DB371_M_UNIT_SPARE".M_CODES_SPARE.M801 := ("DB339_EXTENDED_M_SPARE".M_code[801] OR "DB371_M_UNIT_SPARE".M_CODES_SPARE.M801) AND NOT "DB371_M_UNIT_SPARE".M_CODES_SPARE.Ack_M801 AND NOT "DB2120_MPP_ITC_IPC".RESET_FAULTS AND NOT "DB371_M_UNIT_SPARE".M_CODES_SPARE.M_RESET_PULSE;
END_REGION

REGION Network 97: ACKNOWLEDGE M802- / ACKNOWLEDGE M23-SWITCH ON SPINDLE FRAME BLOWING
   RUNG wire#powerrail
      Contact( "M_ZERO" )
      Coil( "DB371_M_UNIT_SPARE".M_CODES_SPARE.Ack_M802 )
   END_RUNG
   // the same network as SCL:
   "DB371_M_UNIT_SPARE".M_CODES_SPARE.Ack_M802 := "M_ZERO";
END_REGION

REGION Network 98: M802- / M23-SWITCH ON SPINDLE FRAME BLOWING
   RUNG wire#powerrail
      Contact( "DB339_EXTENDED_M_SPARE".M_code[802] )
      wire#w1
      I_Contact( "DB371_M_UNIT_SPARE".M_CODES_SPARE.Ack_M802 )
      I_Contact( "DB2120_MPP_ITC_IPC".RESET_FAULTS )
      I_Contact( "DB371_M_UNIT_SPARE".M_CODES_SPARE.M_RESET_PULSE )
      Coil( "DB371_M_UNIT_SPARE".M_CODES_SPARE.M802 )
   END_RUNG
   RUNG wire#powerrail
      Contact( "DB371_M_UNIT_SPARE".M_CODES_SPARE.M802 )
   END_RUNG wire#w1
   // the same network as SCL:
   "DB371_M_UNIT_SPARE".M_CODES_SPARE.M802 := ("DB339_EXTENDED_M_SPARE".M_code[802] OR "DB371_M_UNIT_SPARE".M_CODES_SPARE.M802) AND NOT "DB371_M_UNIT_SPARE".M_CODES_SPARE.Ack_M802 AND NOT "DB2120_MPP_ITC_IPC".RESET_FAULTS AND NOT "DB371_M_UNIT_SPARE".M_CODES_SPARE.M_RESET_PULSE;
END_REGION

REGION Network 99: ACKNOWLEDGE M803- / ACKNOWLEDGE M23-SWITCH ON SPINDLE FRAME BLOWING
   RUNG wire#powerrail
      Contact( "M_ZERO" )
      Coil( "DB371_M_UNIT_SPARE".M_CODES_SPARE.Ack_M803 )
   END_RUNG
   // the same network as SCL:
   "DB371_M_UNIT_SPARE".M_CODES_SPARE.Ack_M803 := "M_ZERO";
END_REGION

REGION Network 100: M803- / M23-SWITCH ON SPINDLE FRAME BLOWING
   RUNG wire#powerrail
      Contact( "DB339_EXTENDED_M_SPARE".M_code[803] )
      wire#w1
      I_Contact( "DB371_M_UNIT_SPARE".M_CODES_SPARE.Ack_M803 )
      I_Contact( "DB2120_MPP_ITC_IPC".RESET_FAULTS )
      I_Contact( "DB371_M_UNIT_SPARE".M_CODES_SPARE.M_RESET_PULSE )
      Coil( "DB371_M_UNIT_SPARE".M_CODES_SPARE.M803 )
   END_RUNG
   RUNG wire#powerrail
      Contact( "DB371_M_UNIT_SPARE".M_CODES_SPARE.M803 )
   END_RUNG wire#w1
   // the same network as SCL:
   "DB371_M_UNIT_SPARE".M_CODES_SPARE.M803 := ("DB339_EXTENDED_M_SPARE".M_code[803] OR "DB371_M_UNIT_SPARE".M_CODES_SPARE.M803) AND NOT "DB371_M_UNIT_SPARE".M_CODES_SPARE.Ack_M803 AND NOT "DB2120_MPP_ITC_IPC".RESET_FAULTS AND NOT "DB371_M_UNIT_SPARE".M_CODES_SPARE.M_RESET_PULSE;
END_REGION

REGION Network 101: ACKNOWLEDGE M804-
   RUNG wire#powerrail
      Contact( "M_ZERO" )
      Coil( "DB371_M_UNIT_SPARE".M_CODES_SPARE.Ack_M804 )
   END_RUNG
   // the same network as SCL:
   "DB371_M_UNIT_SPARE".M_CODES_SPARE.Ack_M804 := "M_ZERO";
END_REGION

REGION Network 102: M804-
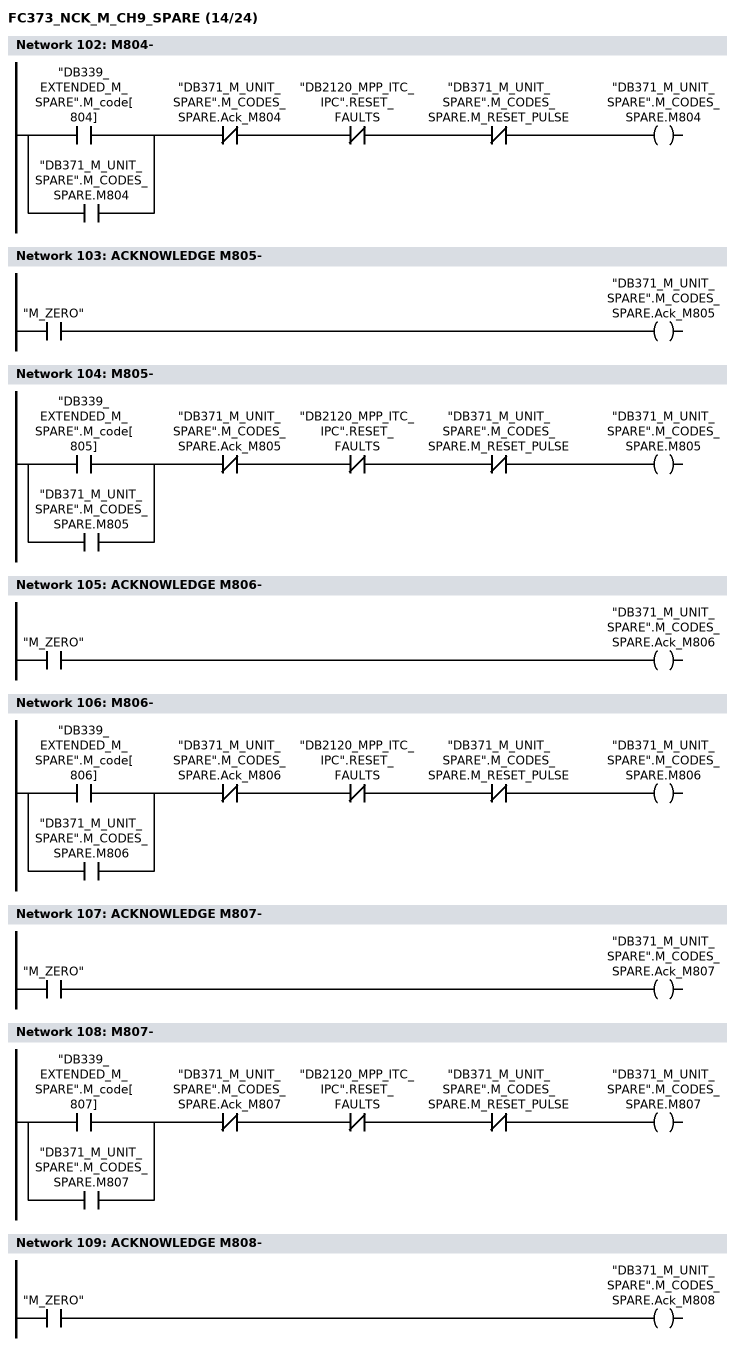
   RUNG wire#powerrail
      Contact( "DB339_EXTENDED_M_SPARE".M_code[804] )
      wire#w1
      I_Contact( "DB371_M_UNIT_SPARE".M_CODES_SPARE.Ack_M804 )
      I_Contact( "DB2120_MPP_ITC_IPC".RESET_FAULTS )
      I_Contact( "DB371_M_UNIT_SPARE".M_CODES_SPARE.M_RESET_PULSE )
      Coil( "DB371_M_UNIT_SPARE".M_CODES_SPARE.M804 )
   END_RUNG
   RUNG wire#powerrail
      Contact( "DB371_M_UNIT_SPARE".M_CODES_SPARE.M804 )
   END_RUNG wire#w1
   // the same network as SCL:
   "DB371_M_UNIT_SPARE".M_CODES_SPARE.M804 := ("DB339_EXTENDED_M_SPARE".M_code[804] OR "DB371_M_UNIT_SPARE".M_CODES_SPARE.M804) AND NOT "DB371_M_UNIT_SPARE".M_CODES_SPARE.Ack_M804 AND NOT "DB2120_MPP_ITC_IPC".RESET_FAULTS AND NOT "DB371_M_UNIT_SPARE".M_CODES_SPARE.M_RESET_PULSE;
END_REGION

REGION Network 103: ACKNOWLEDGE M805-
   RUNG wire#powerrail
      Contact( "M_ZERO" )
      Coil( "DB371_M_UNIT_SPARE".M_CODES_SPARE.Ack_M805 )
   END_RUNG
   // the same network as SCL:
   "DB371_M_UNIT_SPARE".M_CODES_SPARE.Ack_M805 := "M_ZERO";
END_REGION

REGION Network 104: M805-
   RUNG wire#powerrail
      Contact( "DB339_EXTENDED_M_SPARE".M_code[805] )
      wire#w1
      I_Contact( "DB371_M_UNIT_SPARE".M_CODES_SPARE.Ack_M805 )
      I_Contact( "DB2120_MPP_ITC_IPC".RESET_FAULTS )
      I_Contact( "DB371_M_UNIT_SPARE".M_CODES_SPARE.M_RESET_PULSE )
      Coil( "DB371_M_UNIT_SPARE".M_CODES_SPARE.M805 )
   END_RUNG
   RUNG wire#powerrail
      Contact( "DB371_M_UNIT_SPARE".M_CODES_SPARE.M805 )
   END_RUNG wire#w1
   // the same network as SCL:
   "DB371_M_UNIT_SPARE".M_CODES_SPARE.M805 := ("DB339_EXTENDED_M_SPARE".M_code[805] OR "DB371_M_UNIT_SPARE".M_CODES_SPARE.M805) AND NOT "DB371_M_UNIT_SPARE".M_CODES_SPARE.Ack_M805 AND NOT "DB2120_MPP_ITC_IPC".RESET_FAULTS AND NOT "DB371_M_UNIT_SPARE".M_CODES_SPARE.M_RESET_PULSE;
END_REGION

REGION Network 105: ACKNOWLEDGE M806-
   RUNG wire#powerrail
      Contact( "M_ZERO" )
      Coil( "DB371_M_UNIT_SPARE".M_CODES_SPARE.Ack_M806 )
   END_RUNG
   // the same network as SCL:
   "DB371_M_UNIT_SPARE".M_CODES_SPARE.Ack_M806 := "M_ZERO";
END_REGION

REGION Network 106: M806-
   RUNG wire#powerrail
      Contact( "DB339_EXTENDED_M_SPARE".M_code[806] )
      wire#w1
      I_Contact( "DB371_M_UNIT_SPARE".M_CODES_SPARE.Ack_M806 )
      I_Contact( "DB2120_MPP_ITC_IPC".RESET_FAULTS )
      I_Contact( "DB371_M_UNIT_SPARE".M_CODES_SPARE.M_RESET_PULSE )
      Coil( "DB371_M_UNIT_SPARE".M_CODES_SPARE.M806 )
   END_RUNG
   RUNG wire#powerrail
      Contact( "DB371_M_UNIT_SPARE".M_CODES_SPARE.M806 )
   END_RUNG wire#w1
   // the same network as SCL:
   "DB371_M_UNIT_SPARE".M_CODES_SPARE.M806 := ("DB339_EXTENDED_M_SPARE".M_code[806] OR "DB371_M_UNIT_SPARE".M_CODES_SPARE.M806) AND NOT "DB371_M_UNIT_SPARE".M_CODES_SPARE.Ack_M806 AND NOT "DB2120_MPP_ITC_IPC".RESET_FAULTS AND NOT "DB371_M_UNIT_SPARE".M_CODES_SPARE.M_RESET_PULSE;
END_REGION

REGION Network 107: ACKNOWLEDGE M807-
   RUNG wire#powerrail
      Contact( "M_ZERO" )
      Coil( "DB371_M_UNIT_SPARE".M_CODES_SPARE.Ack_M807 )
   END_RUNG
   // the same network as SCL:
   "DB371_M_UNIT_SPARE".M_CODES_SPARE.Ack_M807 := "M_ZERO";
END_REGION

REGION Network 108: M807-
   RUNG wire#powerrail
      Contact( "DB339_EXTENDED_M_SPARE".M_code[807] )
      wire#w1
      I_Contact( "DB371_M_UNIT_SPARE".M_CODES_SPARE.Ack_M807 )
      I_Contact( "DB2120_MPP_ITC_IPC".RESET_FAULTS )
      I_Contact( "DB371_M_UNIT_SPARE".M_CODES_SPARE.M_RESET_PULSE )
      Coil( "DB371_M_UNIT_SPARE".M_CODES_SPARE.M807 )
   END_RUNG
   RUNG wire#powerrail
      Contact( "DB371_M_UNIT_SPARE".M_CODES_SPARE.M807 )
   END_RUNG wire#w1
   // the same network as SCL:
   "DB371_M_UNIT_SPARE".M_CODES_SPARE.M807 := ("DB339_EXTENDED_M_SPARE".M_code[807] OR "DB371_M_UNIT_SPARE".M_CODES_SPARE.M807) AND NOT "DB371_M_UNIT_SPARE".M_CODES_SPARE.Ack_M807 AND NOT "DB2120_MPP_ITC_IPC".RESET_FAULTS AND NOT "DB371_M_UNIT_SPARE".M_CODES_SPARE.M_RESET_PULSE;
END_REGION

REGION Network 109: ACKNOWLEDGE M808-
   RUNG wire#powerrail
      Contact( "M_ZERO" )
      Coil( "DB371_M_UNIT_SPARE".M_CODES_SPARE.Ack_M808 )
   END_RUNG
   // the same network as SCL:
   "DB371_M_UNIT_SPARE".M_CODES_SPARE.Ack_M808 := "M_ZERO";
END_REGION

REGION Network 110: M808-
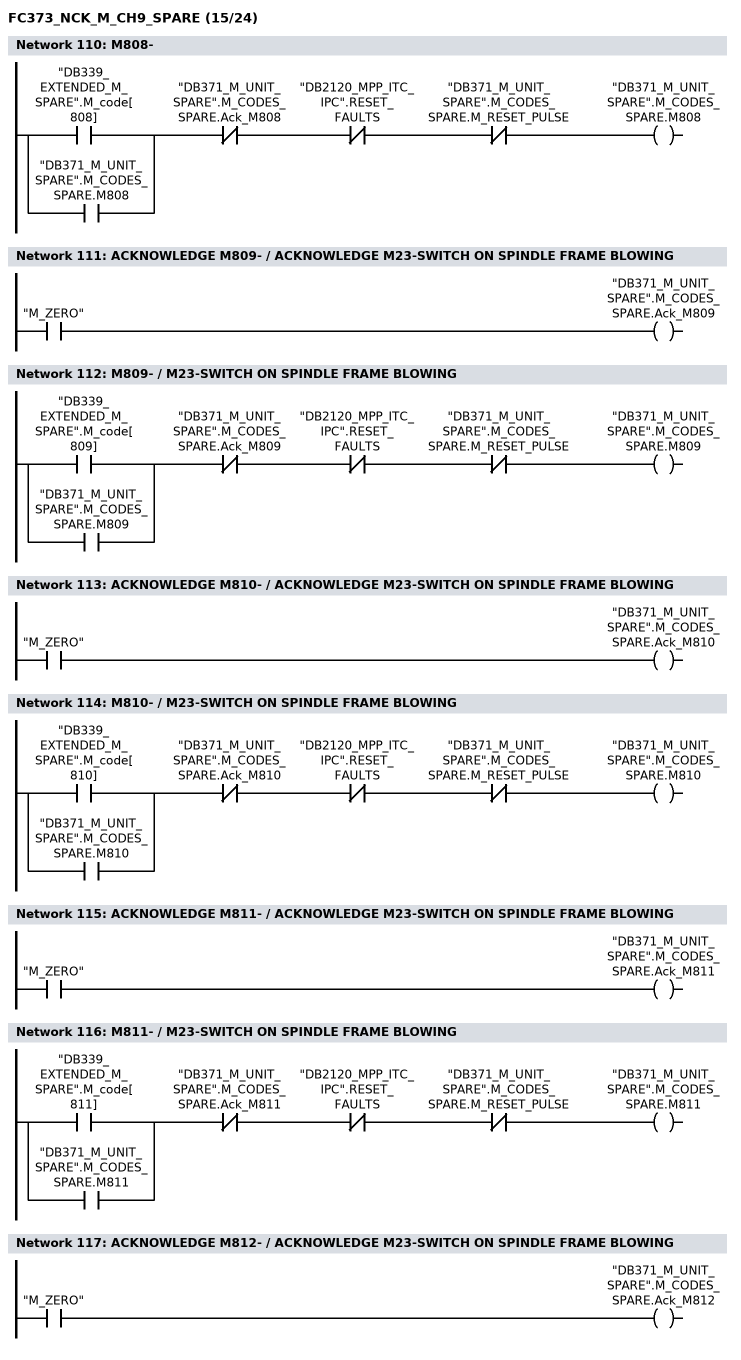
   RUNG wire#powerrail
      Contact( "DB339_EXTENDED_M_SPARE".M_code[808] )
      wire#w1
      I_Contact( "DB371_M_UNIT_SPARE".M_CODES_SPARE.Ack_M808 )
      I_Contact( "DB2120_MPP_ITC_IPC".RESET_FAULTS )
      I_Contact( "DB371_M_UNIT_SPARE".M_CODES_SPARE.M_RESET_PULSE )
      Coil( "DB371_M_UNIT_SPARE".M_CODES_SPARE.M808 )
   END_RUNG
   RUNG wire#powerrail
      Contact( "DB371_M_UNIT_SPARE".M_CODES_SPARE.M808 )
   END_RUNG wire#w1
   // the same network as SCL:
   "DB371_M_UNIT_SPARE".M_CODES_SPARE.M808 := ("DB339_EXTENDED_M_SPARE".M_code[808] OR "DB371_M_UNIT_SPARE".M_CODES_SPARE.M808) AND NOT "DB371_M_UNIT_SPARE".M_CODES_SPARE.Ack_M808 AND NOT "DB2120_MPP_ITC_IPC".RESET_FAULTS AND NOT "DB371_M_UNIT_SPARE".M_CODES_SPARE.M_RESET_PULSE;
END_REGION

REGION Network 111: ACKNOWLEDGE M809- / ACKNOWLEDGE M23-SWITCH ON SPINDLE FRAME BLOWING
   RUNG wire#powerrail
      Contact( "M_ZERO" )
      Coil( "DB371_M_UNIT_SPARE".M_CODES_SPARE.Ack_M809 )
   END_RUNG
   // the same network as SCL:
   "DB371_M_UNIT_SPARE".M_CODES_SPARE.Ack_M809 := "M_ZERO";
END_REGION

REGION Network 112: M809- / M23-SWITCH ON SPINDLE FRAME BLOWING
   RUNG wire#powerrail
      Contact( "DB339_EXTENDED_M_SPARE".M_code[809] )
      wire#w1
      I_Contact( "DB371_M_UNIT_SPARE".M_CODES_SPARE.Ack_M809 )
      I_Contact( "DB2120_MPP_ITC_IPC".RESET_FAULTS )
      I_Contact( "DB371_M_UNIT_SPARE".M_CODES_SPARE.M_RESET_PULSE )
      Coil( "DB371_M_UNIT_SPARE".M_CODES_SPARE.M809 )
   END_RUNG
   RUNG wire#powerrail
      Contact( "DB371_M_UNIT_SPARE".M_CODES_SPARE.M809 )
   END_RUNG wire#w1
   // the same network as SCL:
   "DB371_M_UNIT_SPARE".M_CODES_SPARE.M809 := ("DB339_EXTENDED_M_SPARE".M_code[809] OR "DB371_M_UNIT_SPARE".M_CODES_SPARE.M809) AND NOT "DB371_M_UNIT_SPARE".M_CODES_SPARE.Ack_M809 AND NOT "DB2120_MPP_ITC_IPC".RESET_FAULTS AND NOT "DB371_M_UNIT_SPARE".M_CODES_SPARE.M_RESET_PULSE;
END_REGION

REGION Network 113: ACKNOWLEDGE M810- / ACKNOWLEDGE M23-SWITCH ON SPINDLE FRAME BLOWING
   RUNG wire#powerrail
      Contact( "M_ZERO" )
      Coil( "DB371_M_UNIT_SPARE".M_CODES_SPARE.Ack_M810 )
   END_RUNG
   // the same network as SCL:
   "DB371_M_UNIT_SPARE".M_CODES_SPARE.Ack_M810 := "M_ZERO";
END_REGION

REGION Network 114: M810- / M23-SWITCH ON SPINDLE FRAME BLOWING
   RUNG wire#powerrail
      Contact( "DB339_EXTENDED_M_SPARE".M_code[810] )
      wire#w1
      I_Contact( "DB371_M_UNIT_SPARE".M_CODES_SPARE.Ack_M810 )
      I_Contact( "DB2120_MPP_ITC_IPC".RESET_FAULTS )
      I_Contact( "DB371_M_UNIT_SPARE".M_CODES_SPARE.M_RESET_PULSE )
      Coil( "DB371_M_UNIT_SPARE".M_CODES_SPARE.M810 )
   END_RUNG
   RUNG wire#powerrail
      Contact( "DB371_M_UNIT_SPARE".M_CODES_SPARE.M810 )
   END_RUNG wire#w1
   // the same network as SCL:
   "DB371_M_UNIT_SPARE".M_CODES_SPARE.M810 := ("DB339_EXTENDED_M_SPARE".M_code[810] OR "DB371_M_UNIT_SPARE".M_CODES_SPARE.M810) AND NOT "DB371_M_UNIT_SPARE".M_CODES_SPARE.Ack_M810 AND NOT "DB2120_MPP_ITC_IPC".RESET_FAULTS AND NOT "DB371_M_UNIT_SPARE".M_CODES_SPARE.M_RESET_PULSE;
END_REGION

REGION Network 115: ACKNOWLEDGE M811- / ACKNOWLEDGE M23-SWITCH ON SPINDLE FRAME BLOWING
   RUNG wire#powerrail
      Contact( "M_ZERO" )
      Coil( "DB371_M_UNIT_SPARE".M_CODES_SPARE.Ack_M811 )
   END_RUNG
   // the same network as SCL:
   "DB371_M_UNIT_SPARE".M_CODES_SPARE.Ack_M811 := "M_ZERO";
END_REGION

REGION Network 116: M811- / M23-SWITCH ON SPINDLE FRAME BLOWING
   RUNG wire#powerrail
      Contact( "DB339_EXTENDED_M_SPARE".M_code[811] )
      wire#w1
      I_Contact( "DB371_M_UNIT_SPARE".M_CODES_SPARE.Ack_M811 )
      I_Contact( "DB2120_MPP_ITC_IPC".RESET_FAULTS )
      I_Contact( "DB371_M_UNIT_SPARE".M_CODES_SPARE.M_RESET_PULSE )
      Coil( "DB371_M_UNIT_SPARE".M_CODES_SPARE.M811 )
   END_RUNG
   RUNG wire#powerrail
      Contact( "DB371_M_UNIT_SPARE".M_CODES_SPARE.M811 )
   END_RUNG wire#w1
   // the same network as SCL:
   "DB371_M_UNIT_SPARE".M_CODES_SPARE.M811 := ("DB339_EXTENDED_M_SPARE".M_code[811] OR "DB371_M_UNIT_SPARE".M_CODES_SPARE.M811) AND NOT "DB371_M_UNIT_SPARE".M_CODES_SPARE.Ack_M811 AND NOT "DB2120_MPP_ITC_IPC".RESET_FAULTS AND NOT "DB371_M_UNIT_SPARE".M_CODES_SPARE.M_RESET_PULSE;
END_REGION

REGION Network 117: ACKNOWLEDGE M812- / ACKNOWLEDGE M23-SWITCH ON SPINDLE FRAME BLOWING
   RUNG wire#powerrail
      Contact( "M_ZERO" )
      Coil( "DB371_M_UNIT_SPARE".M_CODES_SPARE.Ack_M812 )
   END_RUNG
   // the same network as SCL:
   "DB371_M_UNIT_SPARE".M_CODES_SPARE.Ack_M812 := "M_ZERO";
END_REGION

REGION Network 118: M812- / M23-SWITCH ON SPINDLE FRAME BLOWING
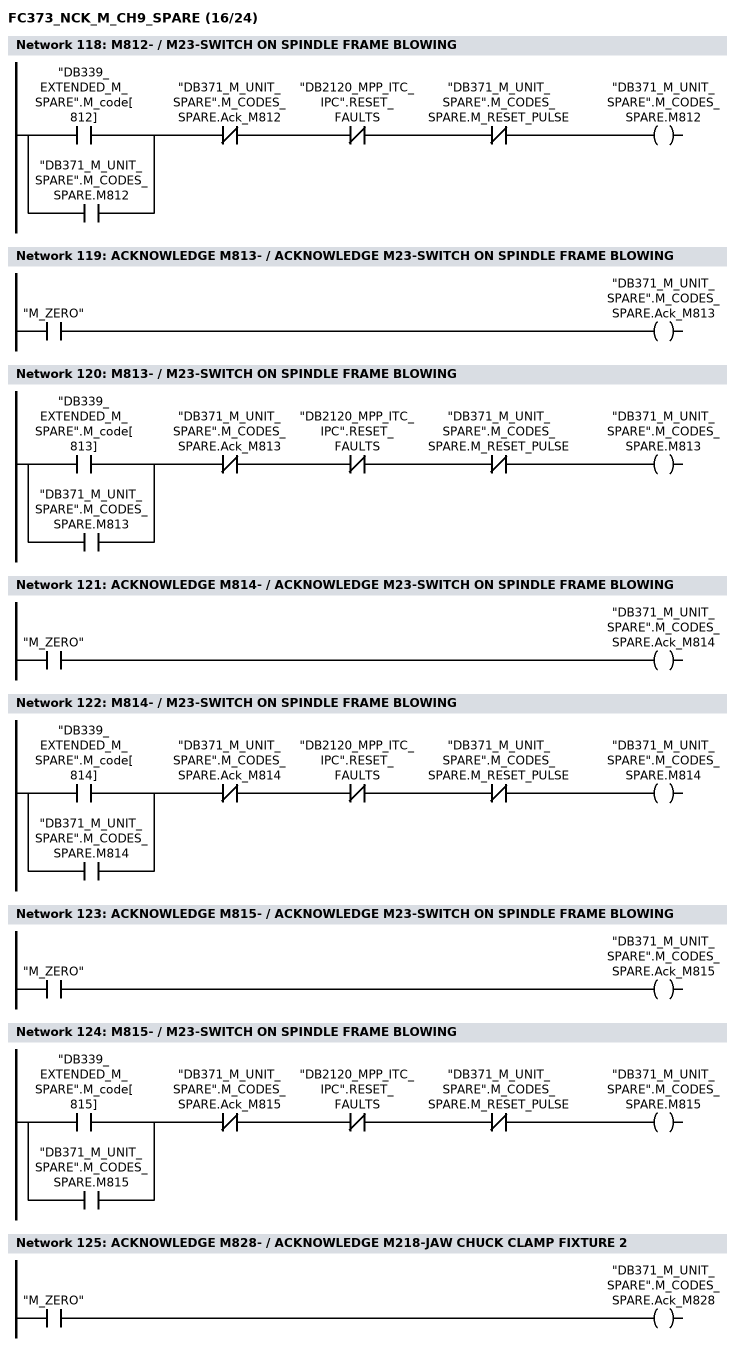
   RUNG wire#powerrail
      Contact( "DB339_EXTENDED_M_SPARE".M_code[812] )
      wire#w1
      I_Contact( "DB371_M_UNIT_SPARE".M_CODES_SPARE.Ack_M812 )
      I_Contact( "DB2120_MPP_ITC_IPC".RESET_FAULTS )
      I_Contact( "DB371_M_UNIT_SPARE".M_CODES_SPARE.M_RESET_PULSE )
      Coil( "DB371_M_UNIT_SPARE".M_CODES_SPARE.M812 )
   END_RUNG
   RUNG wire#powerrail
      Contact( "DB371_M_UNIT_SPARE".M_CODES_SPARE.M812 )
   END_RUNG wire#w1
   // the same network as SCL:
   "DB371_M_UNIT_SPARE".M_CODES_SPARE.M812 := ("DB339_EXTENDED_M_SPARE".M_code[812] OR "DB371_M_UNIT_SPARE".M_CODES_SPARE.M812) AND NOT "DB371_M_UNIT_SPARE".M_CODES_SPARE.Ack_M812 AND NOT "DB2120_MPP_ITC_IPC".RESET_FAULTS AND NOT "DB371_M_UNIT_SPARE".M_CODES_SPARE.M_RESET_PULSE;
END_REGION

REGION Network 119: ACKNOWLEDGE M813- / ACKNOWLEDGE M23-SWITCH ON SPINDLE FRAME BLOWING
   RUNG wire#powerrail
      Contact( "M_ZERO" )
      Coil( "DB371_M_UNIT_SPARE".M_CODES_SPARE.Ack_M813 )
   END_RUNG
   // the same network as SCL:
   "DB371_M_UNIT_SPARE".M_CODES_SPARE.Ack_M813 := "M_ZERO";
END_REGION

REGION Network 120: M813- / M23-SWITCH ON SPINDLE FRAME BLOWING
   RUNG wire#powerrail
      Contact( "DB339_EXTENDED_M_SPARE".M_code[813] )
      wire#w1
      I_Contact( "DB371_M_UNIT_SPARE".M_CODES_SPARE.Ack_M813 )
      I_Contact( "DB2120_MPP_ITC_IPC".RESET_FAULTS )
      I_Contact( "DB371_M_UNIT_SPARE".M_CODES_SPARE.M_RESET_PULSE )
      Coil( "DB371_M_UNIT_SPARE".M_CODES_SPARE.M813 )
   END_RUNG
   RUNG wire#powerrail
      Contact( "DB371_M_UNIT_SPARE".M_CODES_SPARE.M813 )
   END_RUNG wire#w1
   // the same network as SCL:
   "DB371_M_UNIT_SPARE".M_CODES_SPARE.M813 := ("DB339_EXTENDED_M_SPARE".M_code[813] OR "DB371_M_UNIT_SPARE".M_CODES_SPARE.M813) AND NOT "DB371_M_UNIT_SPARE".M_CODES_SPARE.Ack_M813 AND NOT "DB2120_MPP_ITC_IPC".RESET_FAULTS AND NOT "DB371_M_UNIT_SPARE".M_CODES_SPARE.M_RESET_PULSE;
END_REGION

REGION Network 121: ACKNOWLEDGE M814- / ACKNOWLEDGE M23-SWITCH ON SPINDLE FRAME BLOWING
   RUNG wire#powerrail
      Contact( "M_ZERO" )
      Coil( "DB371_M_UNIT_SPARE".M_CODES_SPARE.Ack_M814 )
   END_RUNG
   // the same network as SCL:
   "DB371_M_UNIT_SPARE".M_CODES_SPARE.Ack_M814 := "M_ZERO";
END_REGION

REGION Network 122: M814- / M23-SWITCH ON SPINDLE FRAME BLOWING
   RUNG wire#powerrail
      Contact( "DB339_EXTENDED_M_SPARE".M_code[814] )
      wire#w1
      I_Contact( "DB371_M_UNIT_SPARE".M_CODES_SPARE.Ack_M814 )
      I_Contact( "DB2120_MPP_ITC_IPC".RESET_FAULTS )
      I_Contact( "DB371_M_UNIT_SPARE".M_CODES_SPARE.M_RESET_PULSE )
      Coil( "DB371_M_UNIT_SPARE".M_CODES_SPARE.M814 )
   END_RUNG
   RUNG wire#powerrail
      Contact( "DB371_M_UNIT_SPARE".M_CODES_SPARE.M814 )
   END_RUNG wire#w1
   // the same network as SCL:
   "DB371_M_UNIT_SPARE".M_CODES_SPARE.M814 := ("DB339_EXTENDED_M_SPARE".M_code[814] OR "DB371_M_UNIT_SPARE".M_CODES_SPARE.M814) AND NOT "DB371_M_UNIT_SPARE".M_CODES_SPARE.Ack_M814 AND NOT "DB2120_MPP_ITC_IPC".RESET_FAULTS AND NOT "DB371_M_UNIT_SPARE".M_CODES_SPARE.M_RESET_PULSE;
END_REGION

REGION Network 123: ACKNOWLEDGE M815- / ACKNOWLEDGE M23-SWITCH ON SPINDLE FRAME BLOWING
   RUNG wire#powerrail
      Contact( "M_ZERO" )
      Coil( "DB371_M_UNIT_SPARE".M_CODES_SPARE.Ack_M815 )
   END_RUNG
   // the same network as SCL:
   "DB371_M_UNIT_SPARE".M_CODES_SPARE.Ack_M815 := "M_ZERO";
END_REGION

REGION Network 124: M815- / M23-SWITCH ON SPINDLE FRAME BLOWING
   RUNG wire#powerrail
      Contact( "DB339_EXTENDED_M_SPARE".M_code[815] )
      wire#w1
      I_Contact( "DB371_M_UNIT_SPARE".M_CODES_SPARE.Ack_M815 )
      I_Contact( "DB2120_MPP_ITC_IPC".RESET_FAULTS )
      I_Contact( "DB371_M_UNIT_SPARE".M_CODES_SPARE.M_RESET_PULSE )
      Coil( "DB371_M_UNIT_SPARE".M_CODES_SPARE.M815 )
   END_RUNG
   RUNG wire#powerrail
      Contact( "DB371_M_UNIT_SPARE".M_CODES_SPARE.M815 )
   END_RUNG wire#w1
   // the same network as SCL:
   "DB371_M_UNIT_SPARE".M_CODES_SPARE.M815 := ("DB339_EXTENDED_M_SPARE".M_code[815] OR "DB371_M_UNIT_SPARE".M_CODES_SPARE.M815) AND NOT "DB371_M_UNIT_SPARE".M_CODES_SPARE.Ack_M815 AND NOT "DB2120_MPP_ITC_IPC".RESET_FAULTS AND NOT "DB371_M_UNIT_SPARE".M_CODES_SPARE.M_RESET_PULSE;
END_REGION

REGION Network 125: ACKNOWLEDGE M828- / ACKNOWLEDGE M218-JAW CHUCK CLAMP FIXTURE 2
   RUNG wire#powerrail
      Contact( "M_ZERO" )
      Coil( "DB371_M_UNIT_SPARE".M_CODES_SPARE.Ack_M828 )
   END_RUNG
   // the same network as SCL:
   "DB371_M_UNIT_SPARE".M_CODES_SPARE.Ack_M828 := "M_ZERO";
END_REGION

REGION Network 126: M828- / M218-JAW CHUCK CLAMP FIXTURE 2
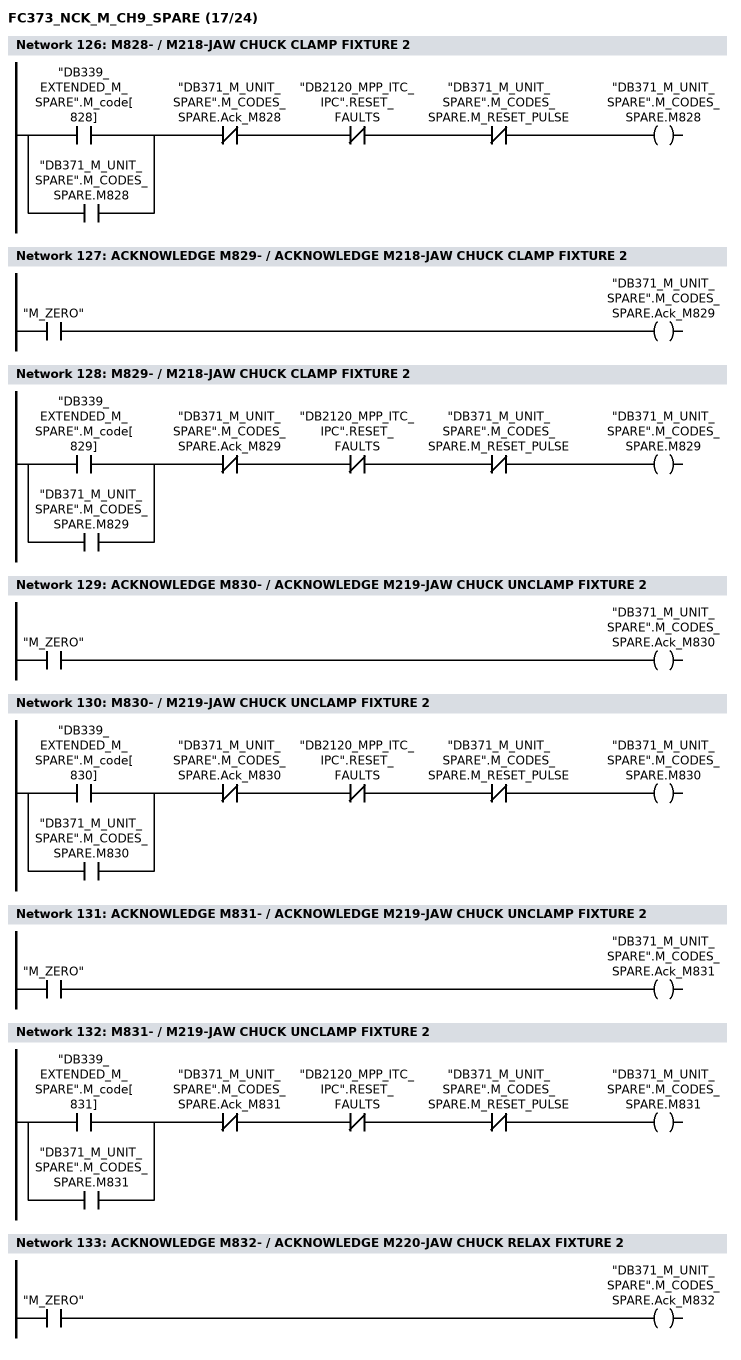
   RUNG wire#powerrail
      Contact( "DB339_EXTENDED_M_SPARE".M_code[828] )
      wire#w1
      I_Contact( "DB371_M_UNIT_SPARE".M_CODES_SPARE.Ack_M828 )
      I_Contact( "DB2120_MPP_ITC_IPC".RESET_FAULTS )
      I_Contact( "DB371_M_UNIT_SPARE".M_CODES_SPARE.M_RESET_PULSE )
      Coil( "DB371_M_UNIT_SPARE".M_CODES_SPARE.M828 )
   END_RUNG
   RUNG wire#powerrail
      Contact( "DB371_M_UNIT_SPARE".M_CODES_SPARE.M828 )
   END_RUNG wire#w1
   // the same network as SCL:
   "DB371_M_UNIT_SPARE".M_CODES_SPARE.M828 := ("DB339_EXTENDED_M_SPARE".M_code[828] OR "DB371_M_UNIT_SPARE".M_CODES_SPARE.M828) AND NOT "DB371_M_UNIT_SPARE".M_CODES_SPARE.Ack_M828 AND NOT "DB2120_MPP_ITC_IPC".RESET_FAULTS AND NOT "DB371_M_UNIT_SPARE".M_CODES_SPARE.M_RESET_PULSE;
END_REGION

REGION Network 127: ACKNOWLEDGE M829- / ACKNOWLEDGE M218-JAW CHUCK CLAMP FIXTURE 2
   RUNG wire#powerrail
      Contact( "M_ZERO" )
      Coil( "DB371_M_UNIT_SPARE".M_CODES_SPARE.Ack_M829 )
   END_RUNG
   // the same network as SCL:
   "DB371_M_UNIT_SPARE".M_CODES_SPARE.Ack_M829 := "M_ZERO";
END_REGION

REGION Network 128: M829- / M218-JAW CHUCK CLAMP FIXTURE 2
   RUNG wire#powerrail
      Contact( "DB339_EXTENDED_M_SPARE".M_code[829] )
      wire#w1
      I_Contact( "DB371_M_UNIT_SPARE".M_CODES_SPARE.Ack_M829 )
      I_Contact( "DB2120_MPP_ITC_IPC".RESET_FAULTS )
      I_Contact( "DB371_M_UNIT_SPARE".M_CODES_SPARE.M_RESET_PULSE )
      Coil( "DB371_M_UNIT_SPARE".M_CODES_SPARE.M829 )
   END_RUNG
   RUNG wire#powerrail
      Contact( "DB371_M_UNIT_SPARE".M_CODES_SPARE.M829 )
   END_RUNG wire#w1
   // the same network as SCL:
   "DB371_M_UNIT_SPARE".M_CODES_SPARE.M829 := ("DB339_EXTENDED_M_SPARE".M_code[829] OR "DB371_M_UNIT_SPARE".M_CODES_SPARE.M829) AND NOT "DB371_M_UNIT_SPARE".M_CODES_SPARE.Ack_M829 AND NOT "DB2120_MPP_ITC_IPC".RESET_FAULTS AND NOT "DB371_M_UNIT_SPARE".M_CODES_SPARE.M_RESET_PULSE;
END_REGION

REGION Network 129: ACKNOWLEDGE M830- / ACKNOWLEDGE M219-JAW CHUCK UNCLAMP FIXTURE 2
   RUNG wire#powerrail
      Contact( "M_ZERO" )
      Coil( "DB371_M_UNIT_SPARE".M_CODES_SPARE.Ack_M830 )
   END_RUNG
   // the same network as SCL:
   "DB371_M_UNIT_SPARE".M_CODES_SPARE.Ack_M830 := "M_ZERO";
END_REGION

REGION Network 130: M830- / M219-JAW CHUCK UNCLAMP FIXTURE 2
   RUNG wire#powerrail
      Contact( "DB339_EXTENDED_M_SPARE".M_code[830] )
      wire#w1
      I_Contact( "DB371_M_UNIT_SPARE".M_CODES_SPARE.Ack_M830 )
      I_Contact( "DB2120_MPP_ITC_IPC".RESET_FAULTS )
      I_Contact( "DB371_M_UNIT_SPARE".M_CODES_SPARE.M_RESET_PULSE )
      Coil( "DB371_M_UNIT_SPARE".M_CODES_SPARE.M830 )
   END_RUNG
   RUNG wire#powerrail
      Contact( "DB371_M_UNIT_SPARE".M_CODES_SPARE.M830 )
   END_RUNG wire#w1
   // the same network as SCL:
   "DB371_M_UNIT_SPARE".M_CODES_SPARE.M830 := ("DB339_EXTENDED_M_SPARE".M_code[830] OR "DB371_M_UNIT_SPARE".M_CODES_SPARE.M830) AND NOT "DB371_M_UNIT_SPARE".M_CODES_SPARE.Ack_M830 AND NOT "DB2120_MPP_ITC_IPC".RESET_FAULTS AND NOT "DB371_M_UNIT_SPARE".M_CODES_SPARE.M_RESET_PULSE;
END_REGION

REGION Network 131: ACKNOWLEDGE M831- / ACKNOWLEDGE M219-JAW CHUCK UNCLAMP FIXTURE 2
   RUNG wire#powerrail
      Contact( "M_ZERO" )
      Coil( "DB371_M_UNIT_SPARE".M_CODES_SPARE.Ack_M831 )
   END_RUNG
   // the same network as SCL:
   "DB371_M_UNIT_SPARE".M_CODES_SPARE.Ack_M831 := "M_ZERO";
END_REGION

REGION Network 132: M831- / M219-JAW CHUCK UNCLAMP FIXTURE 2
   RUNG wire#powerrail
      Contact( "DB339_EXTENDED_M_SPARE".M_code[831] )
      wire#w1
      I_Contact( "DB371_M_UNIT_SPARE".M_CODES_SPARE.Ack_M831 )
      I_Contact( "DB2120_MPP_ITC_IPC".RESET_FAULTS )
      I_Contact( "DB371_M_UNIT_SPARE".M_CODES_SPARE.M_RESET_PULSE )
      Coil( "DB371_M_UNIT_SPARE".M_CODES_SPARE.M831 )
   END_RUNG
   RUNG wire#powerrail
      Contact( "DB371_M_UNIT_SPARE".M_CODES_SPARE.M831 )
   END_RUNG wire#w1
   // the same network as SCL:
   "DB371_M_UNIT_SPARE".M_CODES_SPARE.M831 := ("DB339_EXTENDED_M_SPARE".M_code[831] OR "DB371_M_UNIT_SPARE".M_CODES_SPARE.M831) AND NOT "DB371_M_UNIT_SPARE".M_CODES_SPARE.Ack_M831 AND NOT "DB2120_MPP_ITC_IPC".RESET_FAULTS AND NOT "DB371_M_UNIT_SPARE".M_CODES_SPARE.M_RESET_PULSE;
END_REGION

REGION Network 133: ACKNOWLEDGE M832- / ACKNOWLEDGE M220-JAW CHUCK RELAX FIXTURE 2
   RUNG wire#powerrail
      Contact( "M_ZERO" )
      Coil( "DB371_M_UNIT_SPARE".M_CODES_SPARE.Ack_M832 )
   END_RUNG
   // the same network as SCL:
   "DB371_M_UNIT_SPARE".M_CODES_SPARE.Ack_M832 := "M_ZERO";
END_REGION

REGION Network 134: M832- / M220-JAW CHUCK RELAX FIXTURE 2
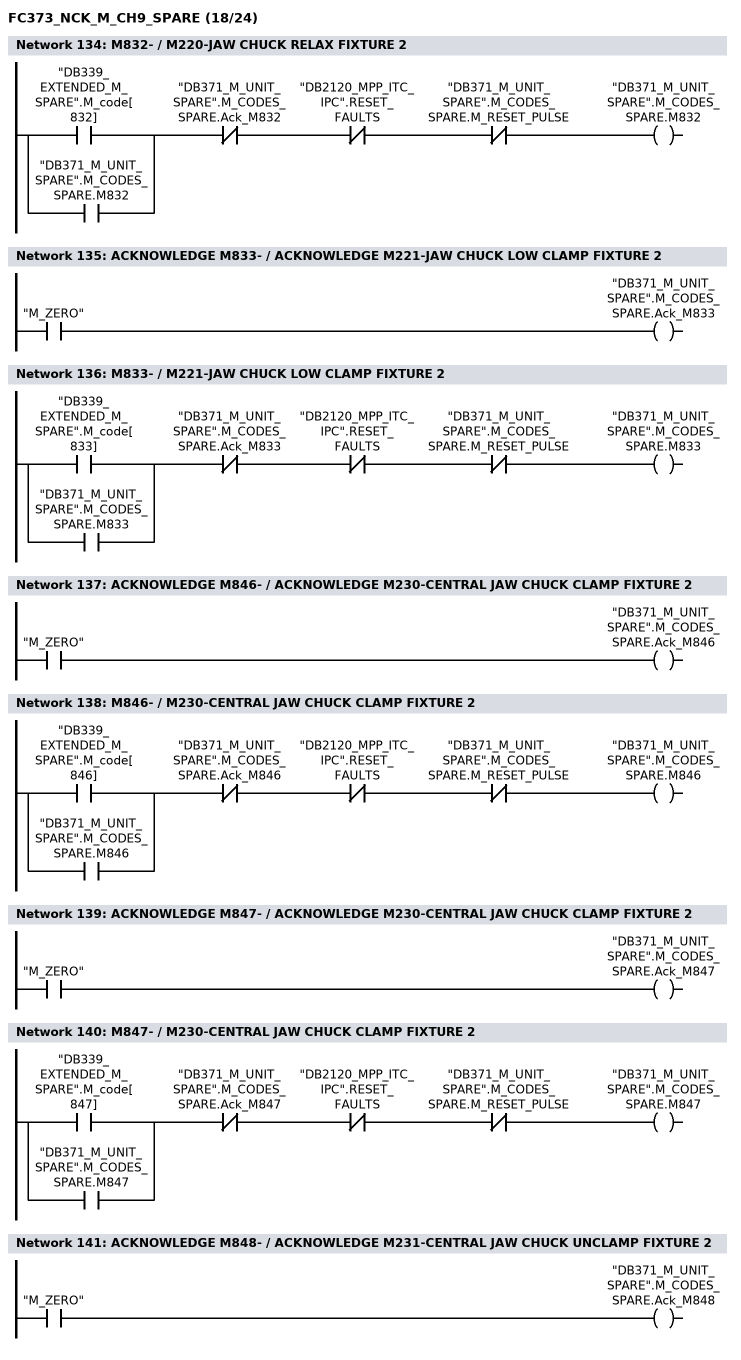
   RUNG wire#powerrail
      Contact( "DB339_EXTENDED_M_SPARE".M_code[832] )
      wire#w1
      I_Contact( "DB371_M_UNIT_SPARE".M_CODES_SPARE.Ack_M832 )
      I_Contact( "DB2120_MPP_ITC_IPC".RESET_FAULTS )
      I_Contact( "DB371_M_UNIT_SPARE".M_CODES_SPARE.M_RESET_PULSE )
      Coil( "DB371_M_UNIT_SPARE".M_CODES_SPARE.M832 )
   END_RUNG
   RUNG wire#powerrail
      Contact( "DB371_M_UNIT_SPARE".M_CODES_SPARE.M832 )
   END_RUNG wire#w1
   // the same network as SCL:
   "DB371_M_UNIT_SPARE".M_CODES_SPARE.M832 := ("DB339_EXTENDED_M_SPARE".M_code[832] OR "DB371_M_UNIT_SPARE".M_CODES_SPARE.M832) AND NOT "DB371_M_UNIT_SPARE".M_CODES_SPARE.Ack_M832 AND NOT "DB2120_MPP_ITC_IPC".RESET_FAULTS AND NOT "DB371_M_UNIT_SPARE".M_CODES_SPARE.M_RESET_PULSE;
END_REGION

REGION Network 135: ACKNOWLEDGE M833- / ACKNOWLEDGE M221-JAW CHUCK LOW CLAMP FIXTURE 2
   RUNG wire#powerrail
      Contact( "M_ZERO" )
      Coil( "DB371_M_UNIT_SPARE".M_CODES_SPARE.Ack_M833 )
   END_RUNG
   // the same network as SCL:
   "DB371_M_UNIT_SPARE".M_CODES_SPARE.Ack_M833 := "M_ZERO";
END_REGION

REGION Network 136: M833- / M221-JAW CHUCK LOW CLAMP FIXTURE 2
   RUNG wire#powerrail
      Contact( "DB339_EXTENDED_M_SPARE".M_code[833] )
      wire#w1
      I_Contact( "DB371_M_UNIT_SPARE".M_CODES_SPARE.Ack_M833 )
      I_Contact( "DB2120_MPP_ITC_IPC".RESET_FAULTS )
      I_Contact( "DB371_M_UNIT_SPARE".M_CODES_SPARE.M_RESET_PULSE )
      Coil( "DB371_M_UNIT_SPARE".M_CODES_SPARE.M833 )
   END_RUNG
   RUNG wire#powerrail
      Contact( "DB371_M_UNIT_SPARE".M_CODES_SPARE.M833 )
   END_RUNG wire#w1
   // the same network as SCL:
   "DB371_M_UNIT_SPARE".M_CODES_SPARE.M833 := ("DB339_EXTENDED_M_SPARE".M_code[833] OR "DB371_M_UNIT_SPARE".M_CODES_SPARE.M833) AND NOT "DB371_M_UNIT_SPARE".M_CODES_SPARE.Ack_M833 AND NOT "DB2120_MPP_ITC_IPC".RESET_FAULTS AND NOT "DB371_M_UNIT_SPARE".M_CODES_SPARE.M_RESET_PULSE;
END_REGION

REGION Network 137: ACKNOWLEDGE M846- / ACKNOWLEDGE M230-CENTRAL JAW CHUCK CLAMP FIXTURE 2
   RUNG wire#powerrail
      Contact( "M_ZERO" )
      Coil( "DB371_M_UNIT_SPARE".M_CODES_SPARE.Ack_M846 )
   END_RUNG
   // the same network as SCL:
   "DB371_M_UNIT_SPARE".M_CODES_SPARE.Ack_M846 := "M_ZERO";
END_REGION

REGION Network 138: M846- / M230-CENTRAL JAW CHUCK CLAMP FIXTURE 2
   RUNG wire#powerrail
      Contact( "DB339_EXTENDED_M_SPARE".M_code[846] )
      wire#w1
      I_Contact( "DB371_M_UNIT_SPARE".M_CODES_SPARE.Ack_M846 )
      I_Contact( "DB2120_MPP_ITC_IPC".RESET_FAULTS )
      I_Contact( "DB371_M_UNIT_SPARE".M_CODES_SPARE.M_RESET_PULSE )
      Coil( "DB371_M_UNIT_SPARE".M_CODES_SPARE.M846 )
   END_RUNG
   RUNG wire#powerrail
      Contact( "DB371_M_UNIT_SPARE".M_CODES_SPARE.M846 )
   END_RUNG wire#w1
   // the same network as SCL:
   "DB371_M_UNIT_SPARE".M_CODES_SPARE.M846 := ("DB339_EXTENDED_M_SPARE".M_code[846] OR "DB371_M_UNIT_SPARE".M_CODES_SPARE.M846) AND NOT "DB371_M_UNIT_SPARE".M_CODES_SPARE.Ack_M846 AND NOT "DB2120_MPP_ITC_IPC".RESET_FAULTS AND NOT "DB371_M_UNIT_SPARE".M_CODES_SPARE.M_RESET_PULSE;
END_REGION

REGION Network 139: ACKNOWLEDGE M847- / ACKNOWLEDGE M230-CENTRAL JAW CHUCK CLAMP FIXTURE 2
   RUNG wire#powerrail
      Contact( "M_ZERO" )
      Coil( "DB371_M_UNIT_SPARE".M_CODES_SPARE.Ack_M847 )
   END_RUNG
   // the same network as SCL:
   "DB371_M_UNIT_SPARE".M_CODES_SPARE.Ack_M847 := "M_ZERO";
END_REGION

REGION Network 140: M847- / M230-CENTRAL JAW CHUCK CLAMP FIXTURE 2
   RUNG wire#powerrail
      Contact( "DB339_EXTENDED_M_SPARE".M_code[847] )
      wire#w1
      I_Contact( "DB371_M_UNIT_SPARE".M_CODES_SPARE.Ack_M847 )
      I_Contact( "DB2120_MPP_ITC_IPC".RESET_FAULTS )
      I_Contact( "DB371_M_UNIT_SPARE".M_CODES_SPARE.M_RESET_PULSE )
      Coil( "DB371_M_UNIT_SPARE".M_CODES_SPARE.M847 )
   END_RUNG
   RUNG wire#powerrail
      Contact( "DB371_M_UNIT_SPARE".M_CODES_SPARE.M847 )
   END_RUNG wire#w1
   // the same network as SCL:
   "DB371_M_UNIT_SPARE".M_CODES_SPARE.M847 := ("DB339_EXTENDED_M_SPARE".M_code[847] OR "DB371_M_UNIT_SPARE".M_CODES_SPARE.M847) AND NOT "DB371_M_UNIT_SPARE".M_CODES_SPARE.Ack_M847 AND NOT "DB2120_MPP_ITC_IPC".RESET_FAULTS AND NOT "DB371_M_UNIT_SPARE".M_CODES_SPARE.M_RESET_PULSE;
END_REGION

REGION Network 141: ACKNOWLEDGE M848- / ACKNOWLEDGE M231-CENTRAL JAW CHUCK UNCLAMP FIXTURE 2
   RUNG wire#powerrail
      Contact( "M_ZERO" )
      Coil( "DB371_M_UNIT_SPARE".M_CODES_SPARE.Ack_M848 )
   END_RUNG
   // the same network as SCL:
   "DB371_M_UNIT_SPARE".M_CODES_SPARE.Ack_M848 := "M_ZERO";
END_REGION

REGION Network 142: M848- / M231-CENTRAL JAW CHUCK UNCLAMP FIXTURE 2
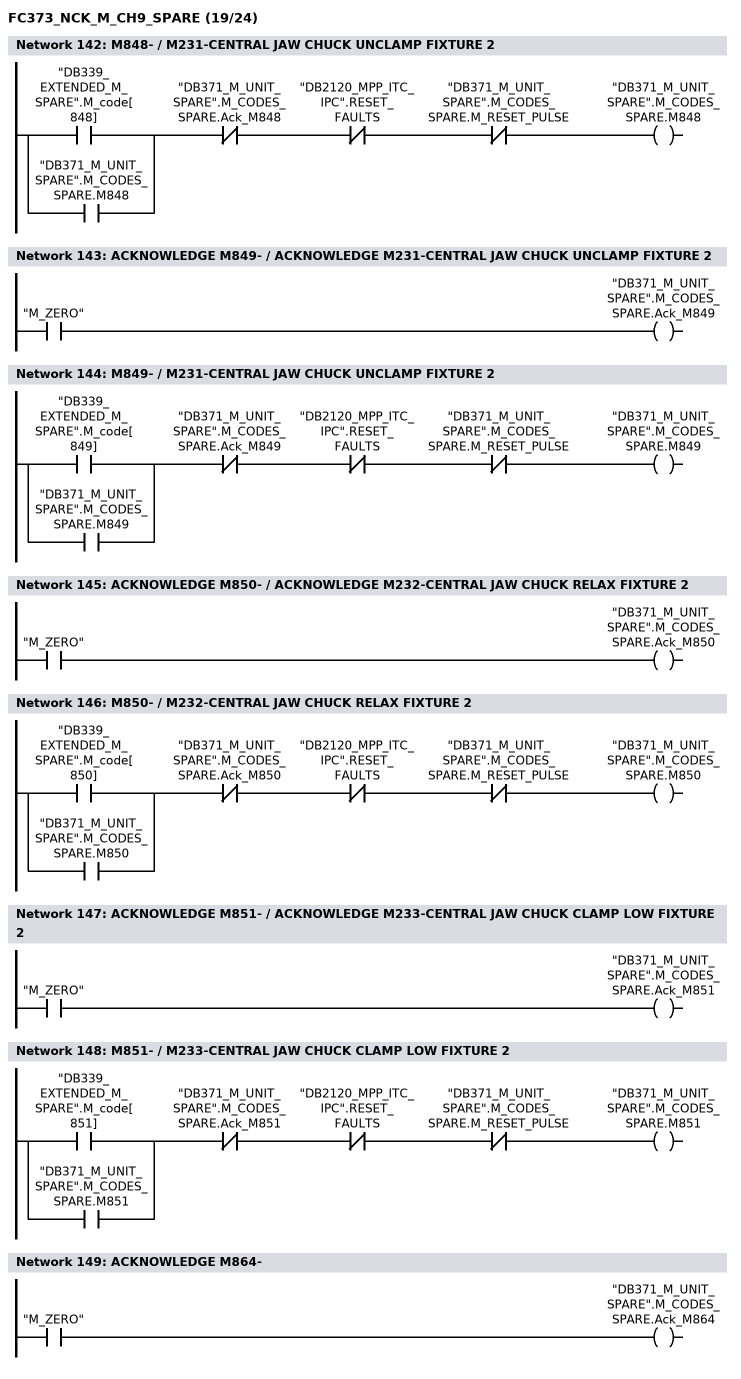
   RUNG wire#powerrail
      Contact( "DB339_EXTENDED_M_SPARE".M_code[848] )
      wire#w1
      I_Contact( "DB371_M_UNIT_SPARE".M_CODES_SPARE.Ack_M848 )
      I_Contact( "DB2120_MPP_ITC_IPC".RESET_FAULTS )
      I_Contact( "DB371_M_UNIT_SPARE".M_CODES_SPARE.M_RESET_PULSE )
      Coil( "DB371_M_UNIT_SPARE".M_CODES_SPARE.M848 )
   END_RUNG
   RUNG wire#powerrail
      Contact( "DB371_M_UNIT_SPARE".M_CODES_SPARE.M848 )
   END_RUNG wire#w1
   // the same network as SCL:
   "DB371_M_UNIT_SPARE".M_CODES_SPARE.M848 := ("DB339_EXTENDED_M_SPARE".M_code[848] OR "DB371_M_UNIT_SPARE".M_CODES_SPARE.M848) AND NOT "DB371_M_UNIT_SPARE".M_CODES_SPARE.Ack_M848 AND NOT "DB2120_MPP_ITC_IPC".RESET_FAULTS AND NOT "DB371_M_UNIT_SPARE".M_CODES_SPARE.M_RESET_PULSE;
END_REGION

REGION Network 143: ACKNOWLEDGE M849- / ACKNOWLEDGE M231-CENTRAL JAW CHUCK UNCLAMP FIXTURE 2
   RUNG wire#powerrail
      Contact( "M_ZERO" )
      Coil( "DB371_M_UNIT_SPARE".M_CODES_SPARE.Ack_M849 )
   END_RUNG
   // the same network as SCL:
   "DB371_M_UNIT_SPARE".M_CODES_SPARE.Ack_M849 := "M_ZERO";
END_REGION

REGION Network 144: M849- / M231-CENTRAL JAW CHUCK UNCLAMP FIXTURE 2
   RUNG wire#powerrail
      Contact( "DB339_EXTENDED_M_SPARE".M_code[849] )
      wire#w1
      I_Contact( "DB371_M_UNIT_SPARE".M_CODES_SPARE.Ack_M849 )
      I_Contact( "DB2120_MPP_ITC_IPC".RESET_FAULTS )
      I_Contact( "DB371_M_UNIT_SPARE".M_CODES_SPARE.M_RESET_PULSE )
      Coil( "DB371_M_UNIT_SPARE".M_CODES_SPARE.M849 )
   END_RUNG
   RUNG wire#powerrail
      Contact( "DB371_M_UNIT_SPARE".M_CODES_SPARE.M849 )
   END_RUNG wire#w1
   // the same network as SCL:
   "DB371_M_UNIT_SPARE".M_CODES_SPARE.M849 := ("DB339_EXTENDED_M_SPARE".M_code[849] OR "DB371_M_UNIT_SPARE".M_CODES_SPARE.M849) AND NOT "DB371_M_UNIT_SPARE".M_CODES_SPARE.Ack_M849 AND NOT "DB2120_MPP_ITC_IPC".RESET_FAULTS AND NOT "DB371_M_UNIT_SPARE".M_CODES_SPARE.M_RESET_PULSE;
END_REGION

REGION Network 145: ACKNOWLEDGE M850- / ACKNOWLEDGE M232-CENTRAL JAW CHUCK RELAX FIXTURE 2
   RUNG wire#powerrail
      Contact( "M_ZERO" )
      Coil( "DB371_M_UNIT_SPARE".M_CODES_SPARE.Ack_M850 )
   END_RUNG
   // the same network as SCL:
   "DB371_M_UNIT_SPARE".M_CODES_SPARE.Ack_M850 := "M_ZERO";
END_REGION

REGION Network 146: M850- / M232-CENTRAL JAW CHUCK RELAX FIXTURE 2
   RUNG wire#powerrail
      Contact( "DB339_EXTENDED_M_SPARE".M_code[850] )
      wire#w1
      I_Contact( "DB371_M_UNIT_SPARE".M_CODES_SPARE.Ack_M850 )
      I_Contact( "DB2120_MPP_ITC_IPC".RESET_FAULTS )
      I_Contact( "DB371_M_UNIT_SPARE".M_CODES_SPARE.M_RESET_PULSE )
      Coil( "DB371_M_UNIT_SPARE".M_CODES_SPARE.M850 )
   END_RUNG
   RUNG wire#powerrail
      Contact( "DB371_M_UNIT_SPARE".M_CODES_SPARE.M850 )
   END_RUNG wire#w1
   // the same network as SCL:
   "DB371_M_UNIT_SPARE".M_CODES_SPARE.M850 := ("DB339_EXTENDED_M_SPARE".M_code[850] OR "DB371_M_UNIT_SPARE".M_CODES_SPARE.M850) AND NOT "DB371_M_UNIT_SPARE".M_CODES_SPARE.Ack_M850 AND NOT "DB2120_MPP_ITC_IPC".RESET_FAULTS AND NOT "DB371_M_UNIT_SPARE".M_CODES_SPARE.M_RESET_PULSE;
END_REGION

REGION Network 147: ACKNOWLEDGE M851- / ACKNOWLEDGE M233-CENTRAL JAW CHUCK CLAMP LOW FIXTURE 2
   RUNG wire#powerrail
      Contact( "M_ZERO" )
      Coil( "DB371_M_UNIT_SPARE".M_CODES_SPARE.Ack_M851 )
   END_RUNG
   // the same network as SCL:
   "DB371_M_UNIT_SPARE".M_CODES_SPARE.Ack_M851 := "M_ZERO";
END_REGION

REGION Network 148: M851- / M233-CENTRAL JAW CHUCK CLAMP LOW FIXTURE 2
   RUNG wire#powerrail
      Contact( "DB339_EXTENDED_M_SPARE".M_code[851] )
      wire#w1
      I_Contact( "DB371_M_UNIT_SPARE".M_CODES_SPARE.Ack_M851 )
      I_Contact( "DB2120_MPP_ITC_IPC".RESET_FAULTS )
      I_Contact( "DB371_M_UNIT_SPARE".M_CODES_SPARE.M_RESET_PULSE )
      Coil( "DB371_M_UNIT_SPARE".M_CODES_SPARE.M851 )
   END_RUNG
   RUNG wire#powerrail
      Contact( "DB371_M_UNIT_SPARE".M_CODES_SPARE.M851 )
   END_RUNG wire#w1
   // the same network as SCL:
   "DB371_M_UNIT_SPARE".M_CODES_SPARE.M851 := ("DB339_EXTENDED_M_SPARE".M_code[851] OR "DB371_M_UNIT_SPARE".M_CODES_SPARE.M851) AND NOT "DB371_M_UNIT_SPARE".M_CODES_SPARE.Ack_M851 AND NOT "DB2120_MPP_ITC_IPC".RESET_FAULTS AND NOT "DB371_M_UNIT_SPARE".M_CODES_SPARE.M_RESET_PULSE;
END_REGION

REGION Network 149: ACKNOWLEDGE M864-
   RUNG wire#powerrail
      Contact( "M_ZERO" )
      Coil( "DB371_M_UNIT_SPARE".M_CODES_SPARE.Ack_M864 )
   END_RUNG
   // the same network as SCL:
   "DB371_M_UNIT_SPARE".M_CODES_SPARE.Ack_M864 := "M_ZERO";
END_REGION

REGION Network 150: M864-
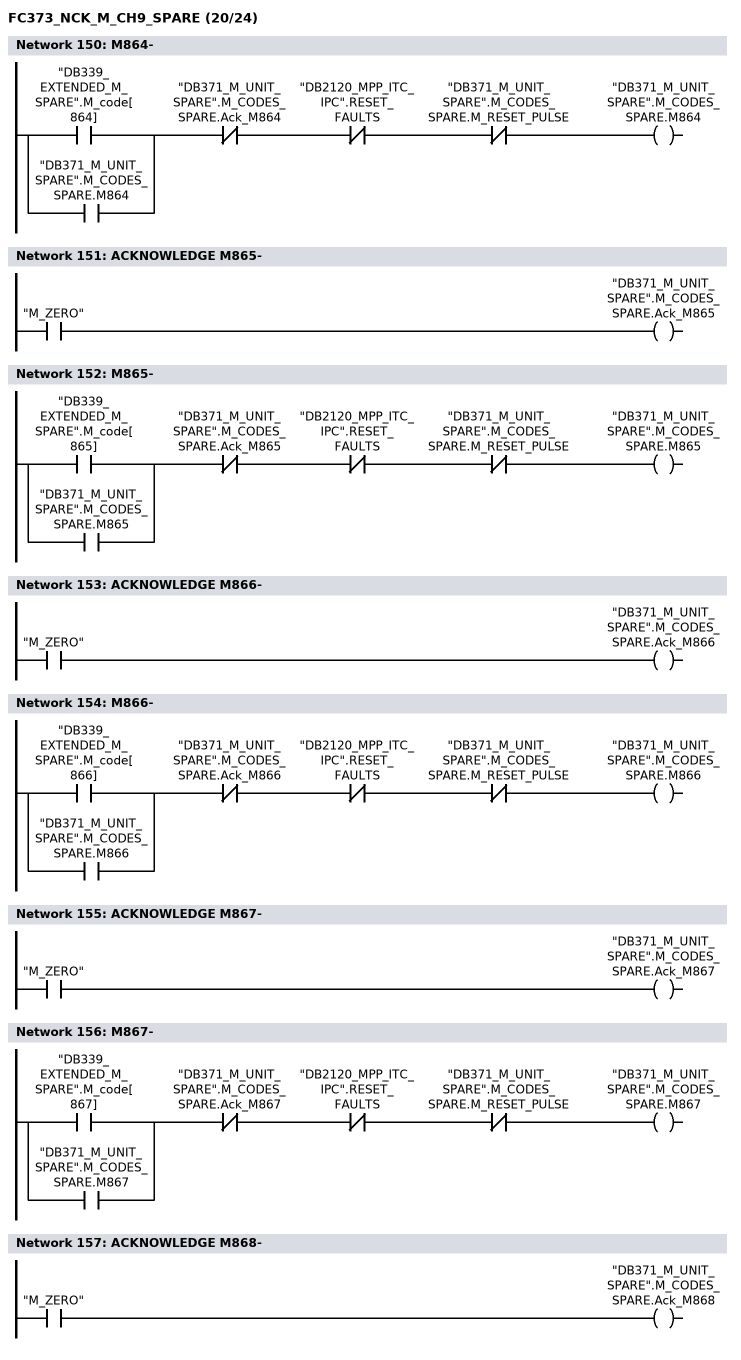
   RUNG wire#powerrail
      Contact( "DB339_EXTENDED_M_SPARE".M_code[864] )
      wire#w1
      I_Contact( "DB371_M_UNIT_SPARE".M_CODES_SPARE.Ack_M864 )
      I_Contact( "DB2120_MPP_ITC_IPC".RESET_FAULTS )
      I_Contact( "DB371_M_UNIT_SPARE".M_CODES_SPARE.M_RESET_PULSE )
      Coil( "DB371_M_UNIT_SPARE".M_CODES_SPARE.M864 )
   END_RUNG
   RUNG wire#powerrail
      Contact( "DB371_M_UNIT_SPARE".M_CODES_SPARE.M864 )
   END_RUNG wire#w1
   // the same network as SCL:
   "DB371_M_UNIT_SPARE".M_CODES_SPARE.M864 := ("DB339_EXTENDED_M_SPARE".M_code[864] OR "DB371_M_UNIT_SPARE".M_CODES_SPARE.M864) AND NOT "DB371_M_UNIT_SPARE".M_CODES_SPARE.Ack_M864 AND NOT "DB2120_MPP_ITC_IPC".RESET_FAULTS AND NOT "DB371_M_UNIT_SPARE".M_CODES_SPARE.M_RESET_PULSE;
END_REGION

REGION Network 151: ACKNOWLEDGE M865-
   RUNG wire#powerrail
      Contact( "M_ZERO" )
      Coil( "DB371_M_UNIT_SPARE".M_CODES_SPARE.Ack_M865 )
   END_RUNG
   // the same network as SCL:
   "DB371_M_UNIT_SPARE".M_CODES_SPARE.Ack_M865 := "M_ZERO";
END_REGION

REGION Network 152: M865-
   RUNG wire#powerrail
      Contact( "DB339_EXTENDED_M_SPARE".M_code[865] )
      wire#w1
      I_Contact( "DB371_M_UNIT_SPARE".M_CODES_SPARE.Ack_M865 )
      I_Contact( "DB2120_MPP_ITC_IPC".RESET_FAULTS )
      I_Contact( "DB371_M_UNIT_SPARE".M_CODES_SPARE.M_RESET_PULSE )
      Coil( "DB371_M_UNIT_SPARE".M_CODES_SPARE.M865 )
   END_RUNG
   RUNG wire#powerrail
      Contact( "DB371_M_UNIT_SPARE".M_CODES_SPARE.M865 )
   END_RUNG wire#w1
   // the same network as SCL:
   "DB371_M_UNIT_SPARE".M_CODES_SPARE.M865 := ("DB339_EXTENDED_M_SPARE".M_code[865] OR "DB371_M_UNIT_SPARE".M_CODES_SPARE.M865) AND NOT "DB371_M_UNIT_SPARE".M_CODES_SPARE.Ack_M865 AND NOT "DB2120_MPP_ITC_IPC".RESET_FAULTS AND NOT "DB371_M_UNIT_SPARE".M_CODES_SPARE.M_RESET_PULSE;
END_REGION

REGION Network 153: ACKNOWLEDGE M866-
   RUNG wire#powerrail
      Contact( "M_ZERO" )
      Coil( "DB371_M_UNIT_SPARE".M_CODES_SPARE.Ack_M866 )
   END_RUNG
   // the same network as SCL:
   "DB371_M_UNIT_SPARE".M_CODES_SPARE.Ack_M866 := "M_ZERO";
END_REGION

REGION Network 154: M866-
   RUNG wire#powerrail
      Contact( "DB339_EXTENDED_M_SPARE".M_code[866] )
      wire#w1
      I_Contact( "DB371_M_UNIT_SPARE".M_CODES_SPARE.Ack_M866 )
      I_Contact( "DB2120_MPP_ITC_IPC".RESET_FAULTS )
      I_Contact( "DB371_M_UNIT_SPARE".M_CODES_SPARE.M_RESET_PULSE )
      Coil( "DB371_M_UNIT_SPARE".M_CODES_SPARE.M866 )
   END_RUNG
   RUNG wire#powerrail
      Contact( "DB371_M_UNIT_SPARE".M_CODES_SPARE.M866 )
   END_RUNG wire#w1
   // the same network as SCL:
   "DB371_M_UNIT_SPARE".M_CODES_SPARE.M866 := ("DB339_EXTENDED_M_SPARE".M_code[866] OR "DB371_M_UNIT_SPARE".M_CODES_SPARE.M866) AND NOT "DB371_M_UNIT_SPARE".M_CODES_SPARE.Ack_M866 AND NOT "DB2120_MPP_ITC_IPC".RESET_FAULTS AND NOT "DB371_M_UNIT_SPARE".M_CODES_SPARE.M_RESET_PULSE;
END_REGION

REGION Network 155: ACKNOWLEDGE M867-
   RUNG wire#powerrail
      Contact( "M_ZERO" )
      Coil( "DB371_M_UNIT_SPARE".M_CODES_SPARE.Ack_M867 )
   END_RUNG
   // the same network as SCL:
   "DB371_M_UNIT_SPARE".M_CODES_SPARE.Ack_M867 := "M_ZERO";
END_REGION

REGION Network 156: M867-
   RUNG wire#powerrail
      Contact( "DB339_EXTENDED_M_SPARE".M_code[867] )
      wire#w1
      I_Contact( "DB371_M_UNIT_SPARE".M_CODES_SPARE.Ack_M867 )
      I_Contact( "DB2120_MPP_ITC_IPC".RESET_FAULTS )
      I_Contact( "DB371_M_UNIT_SPARE".M_CODES_SPARE.M_RESET_PULSE )
      Coil( "DB371_M_UNIT_SPARE".M_CODES_SPARE.M867 )
   END_RUNG
   RUNG wire#powerrail
      Contact( "DB371_M_UNIT_SPARE".M_CODES_SPARE.M867 )
   END_RUNG wire#w1
   // the same network as SCL:
   "DB371_M_UNIT_SPARE".M_CODES_SPARE.M867 := ("DB339_EXTENDED_M_SPARE".M_code[867] OR "DB371_M_UNIT_SPARE".M_CODES_SPARE.M867) AND NOT "DB371_M_UNIT_SPARE".M_CODES_SPARE.Ack_M867 AND NOT "DB2120_MPP_ITC_IPC".RESET_FAULTS AND NOT "DB371_M_UNIT_SPARE".M_CODES_SPARE.M_RESET_PULSE;
END_REGION

REGION Network 157: ACKNOWLEDGE M868-
   RUNG wire#powerrail
      Contact( "M_ZERO" )
      Coil( "DB371_M_UNIT_SPARE".M_CODES_SPARE.Ack_M868 )
   END_RUNG
   // the same network as SCL:
   "DB371_M_UNIT_SPARE".M_CODES_SPARE.Ack_M868 := "M_ZERO";
END_REGION

REGION Network 158: M868-
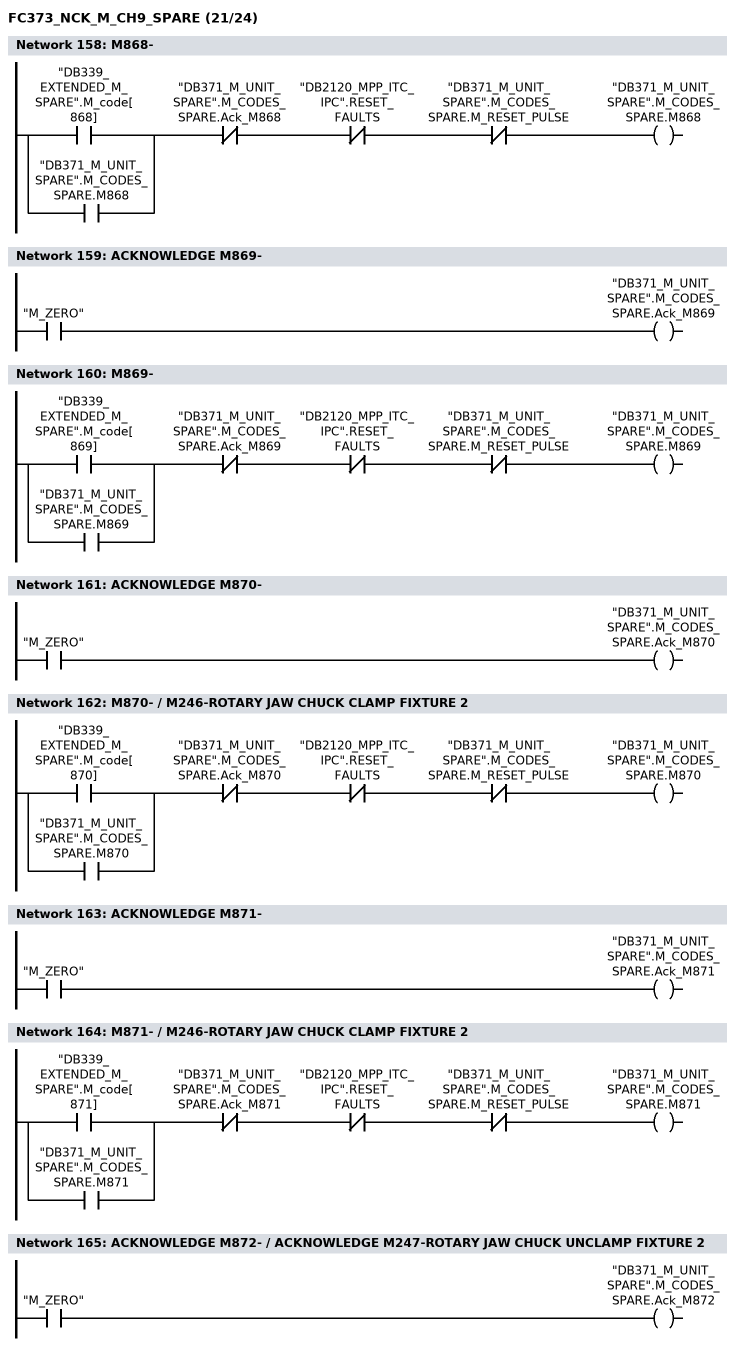
   RUNG wire#powerrail
      Contact( "DB339_EXTENDED_M_SPARE".M_code[868] )
      wire#w1
      I_Contact( "DB371_M_UNIT_SPARE".M_CODES_SPARE.Ack_M868 )
      I_Contact( "DB2120_MPP_ITC_IPC".RESET_FAULTS )
      I_Contact( "DB371_M_UNIT_SPARE".M_CODES_SPARE.M_RESET_PULSE )
      Coil( "DB371_M_UNIT_SPARE".M_CODES_SPARE.M868 )
   END_RUNG
   RUNG wire#powerrail
      Contact( "DB371_M_UNIT_SPARE".M_CODES_SPARE.M868 )
   END_RUNG wire#w1
   // the same network as SCL:
   "DB371_M_UNIT_SPARE".M_CODES_SPARE.M868 := ("DB339_EXTENDED_M_SPARE".M_code[868] OR "DB371_M_UNIT_SPARE".M_CODES_SPARE.M868) AND NOT "DB371_M_UNIT_SPARE".M_CODES_SPARE.Ack_M868 AND NOT "DB2120_MPP_ITC_IPC".RESET_FAULTS AND NOT "DB371_M_UNIT_SPARE".M_CODES_SPARE.M_RESET_PULSE;
END_REGION

REGION Network 159: ACKNOWLEDGE M869-
   RUNG wire#powerrail
      Contact( "M_ZERO" )
      Coil( "DB371_M_UNIT_SPARE".M_CODES_SPARE.Ack_M869 )
   END_RUNG
   // the same network as SCL:
   "DB371_M_UNIT_SPARE".M_CODES_SPARE.Ack_M869 := "M_ZERO";
END_REGION

REGION Network 160: M869-
   RUNG wire#powerrail
      Contact( "DB339_EXTENDED_M_SPARE".M_code[869] )
      wire#w1
      I_Contact( "DB371_M_UNIT_SPARE".M_CODES_SPARE.Ack_M869 )
      I_Contact( "DB2120_MPP_ITC_IPC".RESET_FAULTS )
      I_Contact( "DB371_M_UNIT_SPARE".M_CODES_SPARE.M_RESET_PULSE )
      Coil( "DB371_M_UNIT_SPARE".M_CODES_SPARE.M869 )
   END_RUNG
   RUNG wire#powerrail
      Contact( "DB371_M_UNIT_SPARE".M_CODES_SPARE.M869 )
   END_RUNG wire#w1
   // the same network as SCL:
   "DB371_M_UNIT_SPARE".M_CODES_SPARE.M869 := ("DB339_EXTENDED_M_SPARE".M_code[869] OR "DB371_M_UNIT_SPARE".M_CODES_SPARE.M869) AND NOT "DB371_M_UNIT_SPARE".M_CODES_SPARE.Ack_M869 AND NOT "DB2120_MPP_ITC_IPC".RESET_FAULTS AND NOT "DB371_M_UNIT_SPARE".M_CODES_SPARE.M_RESET_PULSE;
END_REGION

REGION Network 161: ACKNOWLEDGE M870-
   RUNG wire#powerrail
      Contact( "M_ZERO" )
      Coil( "DB371_M_UNIT_SPARE".M_CODES_SPARE.Ack_M870 )
   END_RUNG
   // the same network as SCL:
   "DB371_M_UNIT_SPARE".M_CODES_SPARE.Ack_M870 := "M_ZERO";
END_REGION

REGION Network 162: M870- / M246-ROTARY JAW CHUCK CLAMP FIXTURE 2
   RUNG wire#powerrail
      Contact( "DB339_EXTENDED_M_SPARE".M_code[870] )
      wire#w1
      I_Contact( "DB371_M_UNIT_SPARE".M_CODES_SPARE.Ack_M870 )
      I_Contact( "DB2120_MPP_ITC_IPC".RESET_FAULTS )
      I_Contact( "DB371_M_UNIT_SPARE".M_CODES_SPARE.M_RESET_PULSE )
      Coil( "DB371_M_UNIT_SPARE".M_CODES_SPARE.M870 )
   END_RUNG
   RUNG wire#powerrail
      Contact( "DB371_M_UNIT_SPARE".M_CODES_SPARE.M870 )
   END_RUNG wire#w1
   // the same network as SCL:
   "DB371_M_UNIT_SPARE".M_CODES_SPARE.M870 := ("DB339_EXTENDED_M_SPARE".M_code[870] OR "DB371_M_UNIT_SPARE".M_CODES_SPARE.M870) AND NOT "DB371_M_UNIT_SPARE".M_CODES_SPARE.Ack_M870 AND NOT "DB2120_MPP_ITC_IPC".RESET_FAULTS AND NOT "DB371_M_UNIT_SPARE".M_CODES_SPARE.M_RESET_PULSE;
END_REGION

REGION Network 163: ACKNOWLEDGE M871-
   RUNG wire#powerrail
      Contact( "M_ZERO" )
      Coil( "DB371_M_UNIT_SPARE".M_CODES_SPARE.Ack_M871 )
   END_RUNG
   // the same network as SCL:
   "DB371_M_UNIT_SPARE".M_CODES_SPARE.Ack_M871 := "M_ZERO";
END_REGION

REGION Network 164: M871- / M246-ROTARY JAW CHUCK CLAMP FIXTURE 2
   RUNG wire#powerrail
      Contact( "DB339_EXTENDED_M_SPARE".M_code[871] )
      wire#w1
      I_Contact( "DB371_M_UNIT_SPARE".M_CODES_SPARE.Ack_M871 )
      I_Contact( "DB2120_MPP_ITC_IPC".RESET_FAULTS )
      I_Contact( "DB371_M_UNIT_SPARE".M_CODES_SPARE.M_RESET_PULSE )
      Coil( "DB371_M_UNIT_SPARE".M_CODES_SPARE.M871 )
   END_RUNG
   RUNG wire#powerrail
      Contact( "DB371_M_UNIT_SPARE".M_CODES_SPARE.M871 )
   END_RUNG wire#w1
   // the same network as SCL:
   "DB371_M_UNIT_SPARE".M_CODES_SPARE.M871 := ("DB339_EXTENDED_M_SPARE".M_code[871] OR "DB371_M_UNIT_SPARE".M_CODES_SPARE.M871) AND NOT "DB371_M_UNIT_SPARE".M_CODES_SPARE.Ack_M871 AND NOT "DB2120_MPP_ITC_IPC".RESET_FAULTS AND NOT "DB371_M_UNIT_SPARE".M_CODES_SPARE.M_RESET_PULSE;
END_REGION

REGION Network 165: ACKNOWLEDGE M872- / ACKNOWLEDGE M247-ROTARY JAW CHUCK UNCLAMP FIXTURE 2
   RUNG wire#powerrail
      Contact( "M_ZERO" )
      Coil( "DB371_M_UNIT_SPARE".M_CODES_SPARE.Ack_M872 )
   END_RUNG
   // the same network as SCL:
   "DB371_M_UNIT_SPARE".M_CODES_SPARE.Ack_M872 := "M_ZERO";
END_REGION

REGION Network 166: M872- / M247-ROTARY JAW CHUCK UNCLAMP FIXTURE 2
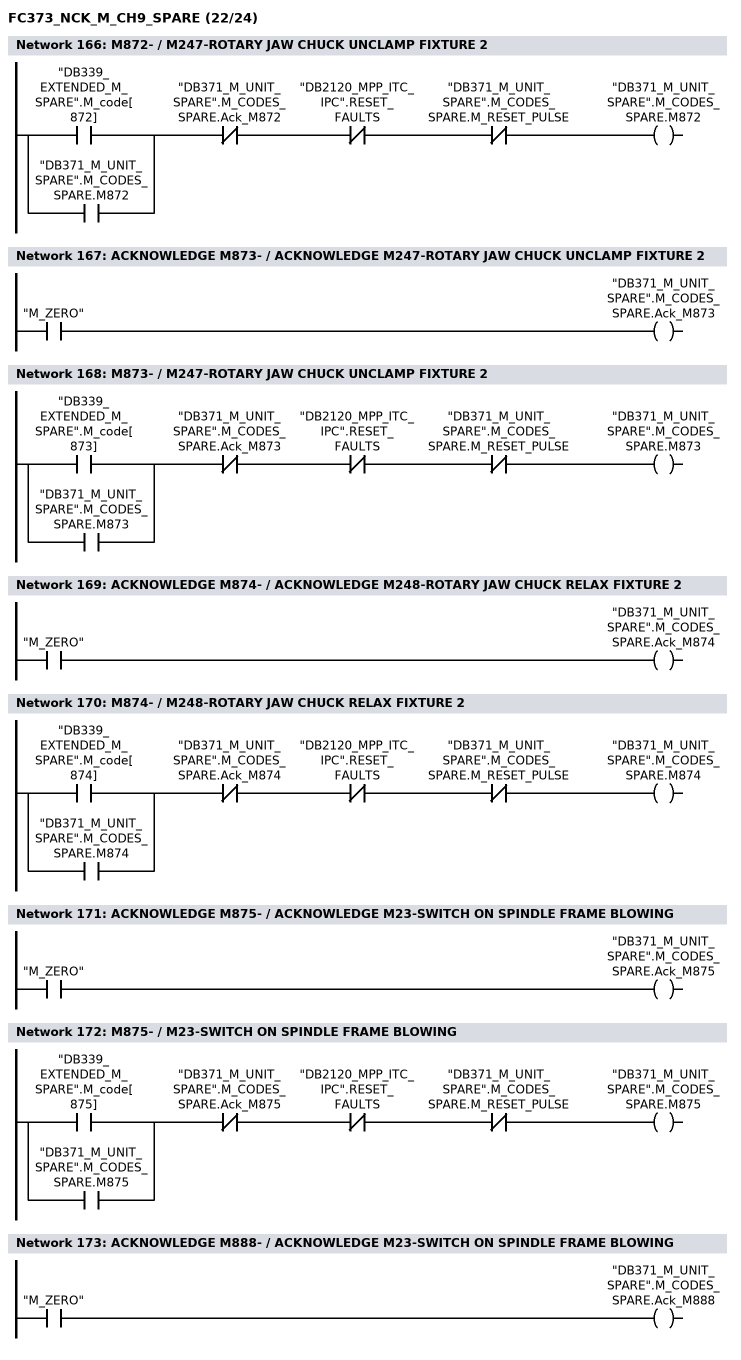
   RUNG wire#powerrail
      Contact( "DB339_EXTENDED_M_SPARE".M_code[872] )
      wire#w1
      I_Contact( "DB371_M_UNIT_SPARE".M_CODES_SPARE.Ack_M872 )
      I_Contact( "DB2120_MPP_ITC_IPC".RESET_FAULTS )
      I_Contact( "DB371_M_UNIT_SPARE".M_CODES_SPARE.M_RESET_PULSE )
      Coil( "DB371_M_UNIT_SPARE".M_CODES_SPARE.M872 )
   END_RUNG
   RUNG wire#powerrail
      Contact( "DB371_M_UNIT_SPARE".M_CODES_SPARE.M872 )
   END_RUNG wire#w1
   // the same network as SCL:
   "DB371_M_UNIT_SPARE".M_CODES_SPARE.M872 := ("DB339_EXTENDED_M_SPARE".M_code[872] OR "DB371_M_UNIT_SPARE".M_CODES_SPARE.M872) AND NOT "DB371_M_UNIT_SPARE".M_CODES_SPARE.Ack_M872 AND NOT "DB2120_MPP_ITC_IPC".RESET_FAULTS AND NOT "DB371_M_UNIT_SPARE".M_CODES_SPARE.M_RESET_PULSE;
END_REGION

REGION Network 167: ACKNOWLEDGE M873- / ACKNOWLEDGE M247-ROTARY JAW CHUCK UNCLAMP FIXTURE 2
   RUNG wire#powerrail
      Contact( "M_ZERO" )
      Coil( "DB371_M_UNIT_SPARE".M_CODES_SPARE.Ack_M873 )
   END_RUNG
   // the same network as SCL:
   "DB371_M_UNIT_SPARE".M_CODES_SPARE.Ack_M873 := "M_ZERO";
END_REGION

REGION Network 168: M873- / M247-ROTARY JAW CHUCK UNCLAMP FIXTURE 2
   RUNG wire#powerrail
      Contact( "DB339_EXTENDED_M_SPARE".M_code[873] )
      wire#w1
      I_Contact( "DB371_M_UNIT_SPARE".M_CODES_SPARE.Ack_M873 )
      I_Contact( "DB2120_MPP_ITC_IPC".RESET_FAULTS )
      I_Contact( "DB371_M_UNIT_SPARE".M_CODES_SPARE.M_RESET_PULSE )
      Coil( "DB371_M_UNIT_SPARE".M_CODES_SPARE.M873 )
   END_RUNG
   RUNG wire#powerrail
      Contact( "DB371_M_UNIT_SPARE".M_CODES_SPARE.M873 )
   END_RUNG wire#w1
   // the same network as SCL:
   "DB371_M_UNIT_SPARE".M_CODES_SPARE.M873 := ("DB339_EXTENDED_M_SPARE".M_code[873] OR "DB371_M_UNIT_SPARE".M_CODES_SPARE.M873) AND NOT "DB371_M_UNIT_SPARE".M_CODES_SPARE.Ack_M873 AND NOT "DB2120_MPP_ITC_IPC".RESET_FAULTS AND NOT "DB371_M_UNIT_SPARE".M_CODES_SPARE.M_RESET_PULSE;
END_REGION

REGION Network 169: ACKNOWLEDGE M874- / ACKNOWLEDGE M248-ROTARY JAW CHUCK RELAX FIXTURE 2
   RUNG wire#powerrail
      Contact( "M_ZERO" )
      Coil( "DB371_M_UNIT_SPARE".M_CODES_SPARE.Ack_M874 )
   END_RUNG
   // the same network as SCL:
   "DB371_M_UNIT_SPARE".M_CODES_SPARE.Ack_M874 := "M_ZERO";
END_REGION

REGION Network 170: M874- / M248-ROTARY JAW CHUCK RELAX FIXTURE 2
   RUNG wire#powerrail
      Contact( "DB339_EXTENDED_M_SPARE".M_code[874] )
      wire#w1
      I_Contact( "DB371_M_UNIT_SPARE".M_CODES_SPARE.Ack_M874 )
      I_Contact( "DB2120_MPP_ITC_IPC".RESET_FAULTS )
      I_Contact( "DB371_M_UNIT_SPARE".M_CODES_SPARE.M_RESET_PULSE )
      Coil( "DB371_M_UNIT_SPARE".M_CODES_SPARE.M874 )
   END_RUNG
   RUNG wire#powerrail
      Contact( "DB371_M_UNIT_SPARE".M_CODES_SPARE.M874 )
   END_RUNG wire#w1
   // the same network as SCL:
   "DB371_M_UNIT_SPARE".M_CODES_SPARE.M874 := ("DB339_EXTENDED_M_SPARE".M_code[874] OR "DB371_M_UNIT_SPARE".M_CODES_SPARE.M874) AND NOT "DB371_M_UNIT_SPARE".M_CODES_SPARE.Ack_M874 AND NOT "DB2120_MPP_ITC_IPC".RESET_FAULTS AND NOT "DB371_M_UNIT_SPARE".M_CODES_SPARE.M_RESET_PULSE;
END_REGION

REGION Network 171: ACKNOWLEDGE M875- / ACKNOWLEDGE M23-SWITCH ON SPINDLE FRAME BLOWING
   RUNG wire#powerrail
      Contact( "M_ZERO" )
      Coil( "DB371_M_UNIT_SPARE".M_CODES_SPARE.Ack_M875 )
   END_RUNG
   // the same network as SCL:
   "DB371_M_UNIT_SPARE".M_CODES_SPARE.Ack_M875 := "M_ZERO";
END_REGION

